(* IEC 61131-3 sources: IEC61131-3-CDSV3/Regular Expressions/src/20 Program Organization Units/Unicode, 1 file *)

(* ---- FuUnicodeCodepointCaseConvert.pou ---- *)
(*#-#-#-#-#-#-#-#-#-#---Declaration---#-#-#-#-#-#-#-#-#-#-#-#-#*)

// Converts the given Unicode odepoint to the lowercase or uppercase codepoint (the opposite casing).
// If there is no codepoint mapping, then it will return 0.
{attribute 'qualified_only'}
FUNCTION FuUnicodeCodepointCaseConvert : DWORD
VAR_INPUT
    dwCodepoint: DWORD;
END_VAR
(*#-#-#-#-#-#-#-#-#-#---Implementation---#-#-#-#-#-#-#-#-#-#-#-#-#*)

FuUnicodeCodepointCaseConvert := 0;

// The following code has been generated from Unicode's UnicodeData.txt file
CASE dwCodepoint OF
    65:
        FuUnicodeCodepointCaseConvert := 97;
        RETURN;
    66:
        FuUnicodeCodepointCaseConvert := 98;
        RETURN;
    67:
        FuUnicodeCodepointCaseConvert := 99;
        RETURN;
    68:
        FuUnicodeCodepointCaseConvert := 100;
        RETURN;
    69:
        FuUnicodeCodepointCaseConvert := 101;
        RETURN;
    70:
        FuUnicodeCodepointCaseConvert := 102;
        RETURN;
    71:
        FuUnicodeCodepointCaseConvert := 103;
        RETURN;
    72:
        FuUnicodeCodepointCaseConvert := 104;
        RETURN;
    73:
        FuUnicodeCodepointCaseConvert := 105;
        RETURN;
    74:
        FuUnicodeCodepointCaseConvert := 106;
        RETURN;
    75:
        FuUnicodeCodepointCaseConvert := 107;
        RETURN;
    76:
        FuUnicodeCodepointCaseConvert := 108;
        RETURN;
    77:
        FuUnicodeCodepointCaseConvert := 109;
        RETURN;
    78:
        FuUnicodeCodepointCaseConvert := 110;
        RETURN;
    79:
        FuUnicodeCodepointCaseConvert := 111;
        RETURN;
    80:
        FuUnicodeCodepointCaseConvert := 112;
        RETURN;
    81:
        FuUnicodeCodepointCaseConvert := 113;
        RETURN;
    82:
        FuUnicodeCodepointCaseConvert := 114;
        RETURN;
    83:
        FuUnicodeCodepointCaseConvert := 115;
        RETURN;
    84:
        FuUnicodeCodepointCaseConvert := 116;
        RETURN;
    85:
        FuUnicodeCodepointCaseConvert := 117;
        RETURN;
    86:
        FuUnicodeCodepointCaseConvert := 118;
        RETURN;
    87:
        FuUnicodeCodepointCaseConvert := 119;
        RETURN;
    88:
        FuUnicodeCodepointCaseConvert := 120;
        RETURN;
    89:
        FuUnicodeCodepointCaseConvert := 121;
        RETURN;
    90:
        FuUnicodeCodepointCaseConvert := 122;
        RETURN;
    97:
        FuUnicodeCodepointCaseConvert := 65;
        RETURN;
    98:
        FuUnicodeCodepointCaseConvert := 66;
        RETURN;
    99:
        FuUnicodeCodepointCaseConvert := 67;
        RETURN;
    100:
        FuUnicodeCodepointCaseConvert := 68;
        RETURN;
    101:
        FuUnicodeCodepointCaseConvert := 69;
        RETURN;
    102:
        FuUnicodeCodepointCaseConvert := 70;
        RETURN;
    103:
        FuUnicodeCodepointCaseConvert := 71;
        RETURN;
    104:
        FuUnicodeCodepointCaseConvert := 72;
        RETURN;
    105:
        FuUnicodeCodepointCaseConvert := 73;
        RETURN;
    106:
        FuUnicodeCodepointCaseConvert := 74;
        RETURN;
    107:
        FuUnicodeCodepointCaseConvert := 75;
        RETURN;
    108:
        FuUnicodeCodepointCaseConvert := 76;
        RETURN;
    109:
        FuUnicodeCodepointCaseConvert := 77;
        RETURN;
    110:
        FuUnicodeCodepointCaseConvert := 78;
        RETURN;
    111:
        FuUnicodeCodepointCaseConvert := 79;
        RETURN;
    112:
        FuUnicodeCodepointCaseConvert := 80;
        RETURN;
    113:
        FuUnicodeCodepointCaseConvert := 81;
        RETURN;
    114:
        FuUnicodeCodepointCaseConvert := 82;
        RETURN;
    115:
        FuUnicodeCodepointCaseConvert := 83;
        RETURN;
    116:
        FuUnicodeCodepointCaseConvert := 84;
        RETURN;
    117:
        FuUnicodeCodepointCaseConvert := 85;
        RETURN;
    118:
        FuUnicodeCodepointCaseConvert := 86;
        RETURN;
    119:
        FuUnicodeCodepointCaseConvert := 87;
        RETURN;
    120:
        FuUnicodeCodepointCaseConvert := 88;
        RETURN;
    121:
        FuUnicodeCodepointCaseConvert := 89;
        RETURN;
    122:
        FuUnicodeCodepointCaseConvert := 90;
        RETURN;
    181:
        FuUnicodeCodepointCaseConvert := 924;
        RETURN;
    192:
        FuUnicodeCodepointCaseConvert := 224;
        RETURN;
    193:
        FuUnicodeCodepointCaseConvert := 225;
        RETURN;
    194:
        FuUnicodeCodepointCaseConvert := 226;
        RETURN;
    195:
        FuUnicodeCodepointCaseConvert := 227;
        RETURN;
    196:
        FuUnicodeCodepointCaseConvert := 228;
        RETURN;
    197:
        FuUnicodeCodepointCaseConvert := 229;
        RETURN;
    198:
        FuUnicodeCodepointCaseConvert := 230;
        RETURN;
    199:
        FuUnicodeCodepointCaseConvert := 231;
        RETURN;
    200:
        FuUnicodeCodepointCaseConvert := 232;
        RETURN;
    201:
        FuUnicodeCodepointCaseConvert := 233;
        RETURN;
    202:
        FuUnicodeCodepointCaseConvert := 234;
        RETURN;
    203:
        FuUnicodeCodepointCaseConvert := 235;
        RETURN;
    204:
        FuUnicodeCodepointCaseConvert := 236;
        RETURN;
    205:
        FuUnicodeCodepointCaseConvert := 237;
        RETURN;
    206:
        FuUnicodeCodepointCaseConvert := 238;
        RETURN;
    207:
        FuUnicodeCodepointCaseConvert := 239;
        RETURN;
    208:
        FuUnicodeCodepointCaseConvert := 240;
        RETURN;
    209:
        FuUnicodeCodepointCaseConvert := 241;
        RETURN;
    210:
        FuUnicodeCodepointCaseConvert := 242;
        RETURN;
    211:
        FuUnicodeCodepointCaseConvert := 243;
        RETURN;
    212:
        FuUnicodeCodepointCaseConvert := 244;
        RETURN;
    213:
        FuUnicodeCodepointCaseConvert := 245;
        RETURN;
    214:
        FuUnicodeCodepointCaseConvert := 246;
        RETURN;
    216:
        FuUnicodeCodepointCaseConvert := 248;
        RETURN;
    217:
        FuUnicodeCodepointCaseConvert := 249;
        RETURN;
    218:
        FuUnicodeCodepointCaseConvert := 250;
        RETURN;
    219:
        FuUnicodeCodepointCaseConvert := 251;
        RETURN;
    220:
        FuUnicodeCodepointCaseConvert := 252;
        RETURN;
    221:
        FuUnicodeCodepointCaseConvert := 253;
        RETURN;
    222:
        FuUnicodeCodepointCaseConvert := 254;
        RETURN;
    224:
        FuUnicodeCodepointCaseConvert := 192;
        RETURN;
    225:
        FuUnicodeCodepointCaseConvert := 193;
        RETURN;
    226:
        FuUnicodeCodepointCaseConvert := 194;
        RETURN;
    227:
        FuUnicodeCodepointCaseConvert := 195;
        RETURN;
    228:
        FuUnicodeCodepointCaseConvert := 196;
        RETURN;
    229:
        FuUnicodeCodepointCaseConvert := 197;
        RETURN;
    230:
        FuUnicodeCodepointCaseConvert := 198;
        RETURN;
    231:
        FuUnicodeCodepointCaseConvert := 199;
        RETURN;
    232:
        FuUnicodeCodepointCaseConvert := 200;
        RETURN;
    233:
        FuUnicodeCodepointCaseConvert := 201;
        RETURN;
    234:
        FuUnicodeCodepointCaseConvert := 202;
        RETURN;
    235:
        FuUnicodeCodepointCaseConvert := 203;
        RETURN;
    236:
        FuUnicodeCodepointCaseConvert := 204;
        RETURN;
    237:
        FuUnicodeCodepointCaseConvert := 205;
        RETURN;
    238:
        FuUnicodeCodepointCaseConvert := 206;
        RETURN;
    239:
        FuUnicodeCodepointCaseConvert := 207;
        RETURN;
    240:
        FuUnicodeCodepointCaseConvert := 208;
        RETURN;
    241:
        FuUnicodeCodepointCaseConvert := 209;
        RETURN;
    242:
        FuUnicodeCodepointCaseConvert := 210;
        RETURN;
    243:
        FuUnicodeCodepointCaseConvert := 211;
        RETURN;
    244:
        FuUnicodeCodepointCaseConvert := 212;
        RETURN;
    245:
        FuUnicodeCodepointCaseConvert := 213;
        RETURN;
    246:
        FuUnicodeCodepointCaseConvert := 214;
        RETURN;
    248:
        FuUnicodeCodepointCaseConvert := 216;
        RETURN;
    249:
        FuUnicodeCodepointCaseConvert := 217;
        RETURN;
    250:
        FuUnicodeCodepointCaseConvert := 218;
        RETURN;
    251:
        FuUnicodeCodepointCaseConvert := 219;
        RETURN;
    252:
        FuUnicodeCodepointCaseConvert := 220;
        RETURN;
    253:
        FuUnicodeCodepointCaseConvert := 221;
        RETURN;
    254:
        FuUnicodeCodepointCaseConvert := 222;
        RETURN;
    255:
        FuUnicodeCodepointCaseConvert := 376;
        RETURN;
    256:
        FuUnicodeCodepointCaseConvert := 257;
        RETURN;
    257:
        FuUnicodeCodepointCaseConvert := 256;
        RETURN;
    258:
        FuUnicodeCodepointCaseConvert := 259;
        RETURN;
    259:
        FuUnicodeCodepointCaseConvert := 258;
        RETURN;
    260:
        FuUnicodeCodepointCaseConvert := 261;
        RETURN;
    261:
        FuUnicodeCodepointCaseConvert := 260;
        RETURN;
    262:
        FuUnicodeCodepointCaseConvert := 263;
        RETURN;
    263:
        FuUnicodeCodepointCaseConvert := 262;
        RETURN;
    264:
        FuUnicodeCodepointCaseConvert := 265;
        RETURN;
    265:
        FuUnicodeCodepointCaseConvert := 264;
        RETURN;
    266:
        FuUnicodeCodepointCaseConvert := 267;
        RETURN;
    267:
        FuUnicodeCodepointCaseConvert := 266;
        RETURN;
    268:
        FuUnicodeCodepointCaseConvert := 269;
        RETURN;
    269:
        FuUnicodeCodepointCaseConvert := 268;
        RETURN;
    270:
        FuUnicodeCodepointCaseConvert := 271;
        RETURN;
    271:
        FuUnicodeCodepointCaseConvert := 270;
        RETURN;
    272:
        FuUnicodeCodepointCaseConvert := 273;
        RETURN;
    273:
        FuUnicodeCodepointCaseConvert := 272;
        RETURN;
    274:
        FuUnicodeCodepointCaseConvert := 275;
        RETURN;
    275:
        FuUnicodeCodepointCaseConvert := 274;
        RETURN;
    276:
        FuUnicodeCodepointCaseConvert := 277;
        RETURN;
    277:
        FuUnicodeCodepointCaseConvert := 276;
        RETURN;
    278:
        FuUnicodeCodepointCaseConvert := 279;
        RETURN;
    279:
        FuUnicodeCodepointCaseConvert := 278;
        RETURN;
    280:
        FuUnicodeCodepointCaseConvert := 281;
        RETURN;
    281:
        FuUnicodeCodepointCaseConvert := 280;
        RETURN;
    282:
        FuUnicodeCodepointCaseConvert := 283;
        RETURN;
    283:
        FuUnicodeCodepointCaseConvert := 282;
        RETURN;
    284:
        FuUnicodeCodepointCaseConvert := 285;
        RETURN;
    285:
        FuUnicodeCodepointCaseConvert := 284;
        RETURN;
    286:
        FuUnicodeCodepointCaseConvert := 287;
        RETURN;
    287:
        FuUnicodeCodepointCaseConvert := 286;
        RETURN;
    288:
        FuUnicodeCodepointCaseConvert := 289;
        RETURN;
    289:
        FuUnicodeCodepointCaseConvert := 288;
        RETURN;
    290:
        FuUnicodeCodepointCaseConvert := 291;
        RETURN;
    291:
        FuUnicodeCodepointCaseConvert := 290;
        RETURN;
    292:
        FuUnicodeCodepointCaseConvert := 293;
        RETURN;
    293:
        FuUnicodeCodepointCaseConvert := 292;
        RETURN;
    294:
        FuUnicodeCodepointCaseConvert := 295;
        RETURN;
    295:
        FuUnicodeCodepointCaseConvert := 294;
        RETURN;
    296:
        FuUnicodeCodepointCaseConvert := 297;
        RETURN;
    297:
        FuUnicodeCodepointCaseConvert := 296;
        RETURN;
    298:
        FuUnicodeCodepointCaseConvert := 299;
        RETURN;
    299:
        FuUnicodeCodepointCaseConvert := 298;
        RETURN;
    300:
        FuUnicodeCodepointCaseConvert := 301;
        RETURN;
    301:
        FuUnicodeCodepointCaseConvert := 300;
        RETURN;
    302:
        FuUnicodeCodepointCaseConvert := 303;
        RETURN;
    303:
        FuUnicodeCodepointCaseConvert := 302;
        RETURN;
    304:
        FuUnicodeCodepointCaseConvert := 105;
        RETURN;
    305:
        FuUnicodeCodepointCaseConvert := 73;
        RETURN;
    306:
        FuUnicodeCodepointCaseConvert := 307;
        RETURN;
    307:
        FuUnicodeCodepointCaseConvert := 306;
        RETURN;
    308:
        FuUnicodeCodepointCaseConvert := 309;
        RETURN;
    309:
        FuUnicodeCodepointCaseConvert := 308;
        RETURN;
    310:
        FuUnicodeCodepointCaseConvert := 311;
        RETURN;
    311:
        FuUnicodeCodepointCaseConvert := 310;
        RETURN;
    313:
        FuUnicodeCodepointCaseConvert := 314;
        RETURN;
    314:
        FuUnicodeCodepointCaseConvert := 313;
        RETURN;
    315:
        FuUnicodeCodepointCaseConvert := 316;
        RETURN;
    316:
        FuUnicodeCodepointCaseConvert := 315;
        RETURN;
    317:
        FuUnicodeCodepointCaseConvert := 318;
        RETURN;
    318:
        FuUnicodeCodepointCaseConvert := 317;
        RETURN;
    319:
        FuUnicodeCodepointCaseConvert := 320;
        RETURN;
    320:
        FuUnicodeCodepointCaseConvert := 319;
        RETURN;
    321:
        FuUnicodeCodepointCaseConvert := 322;
        RETURN;
    322:
        FuUnicodeCodepointCaseConvert := 321;
        RETURN;
    323:
        FuUnicodeCodepointCaseConvert := 324;
        RETURN;
    324:
        FuUnicodeCodepointCaseConvert := 323;
        RETURN;
    325:
        FuUnicodeCodepointCaseConvert := 326;
        RETURN;
    326:
        FuUnicodeCodepointCaseConvert := 325;
        RETURN;
    327:
        FuUnicodeCodepointCaseConvert := 328;
        RETURN;
    328:
        FuUnicodeCodepointCaseConvert := 327;
        RETURN;
    330:
        FuUnicodeCodepointCaseConvert := 331;
        RETURN;
    331:
        FuUnicodeCodepointCaseConvert := 330;
        RETURN;
    332:
        FuUnicodeCodepointCaseConvert := 333;
        RETURN;
    333:
        FuUnicodeCodepointCaseConvert := 332;
        RETURN;
    334:
        FuUnicodeCodepointCaseConvert := 335;
        RETURN;
    335:
        FuUnicodeCodepointCaseConvert := 334;
        RETURN;
    336:
        FuUnicodeCodepointCaseConvert := 337;
        RETURN;
    337:
        FuUnicodeCodepointCaseConvert := 336;
        RETURN;
    338:
        FuUnicodeCodepointCaseConvert := 339;
        RETURN;
    339:
        FuUnicodeCodepointCaseConvert := 338;
        RETURN;
    340:
        FuUnicodeCodepointCaseConvert := 341;
        RETURN;
    341:
        FuUnicodeCodepointCaseConvert := 340;
        RETURN;
    342:
        FuUnicodeCodepointCaseConvert := 343;
        RETURN;
    343:
        FuUnicodeCodepointCaseConvert := 342;
        RETURN;
    344:
        FuUnicodeCodepointCaseConvert := 345;
        RETURN;
    345:
        FuUnicodeCodepointCaseConvert := 344;
        RETURN;
    346:
        FuUnicodeCodepointCaseConvert := 347;
        RETURN;
    347:
        FuUnicodeCodepointCaseConvert := 346;
        RETURN;
    348:
        FuUnicodeCodepointCaseConvert := 349;
        RETURN;
    349:
        FuUnicodeCodepointCaseConvert := 348;
        RETURN;
    350:
        FuUnicodeCodepointCaseConvert := 351;
        RETURN;
    351:
        FuUnicodeCodepointCaseConvert := 350;
        RETURN;
    352:
        FuUnicodeCodepointCaseConvert := 353;
        RETURN;
    353:
        FuUnicodeCodepointCaseConvert := 352;
        RETURN;
    354:
        FuUnicodeCodepointCaseConvert := 355;
        RETURN;
    355:
        FuUnicodeCodepointCaseConvert := 354;
        RETURN;
    356:
        FuUnicodeCodepointCaseConvert := 357;
        RETURN;
    357:
        FuUnicodeCodepointCaseConvert := 356;
        RETURN;
    358:
        FuUnicodeCodepointCaseConvert := 359;
        RETURN;
    359:
        FuUnicodeCodepointCaseConvert := 358;
        RETURN;
    360:
        FuUnicodeCodepointCaseConvert := 361;
        RETURN;
    361:
        FuUnicodeCodepointCaseConvert := 360;
        RETURN;
    362:
        FuUnicodeCodepointCaseConvert := 363;
        RETURN;
    363:
        FuUnicodeCodepointCaseConvert := 362;
        RETURN;
    364:
        FuUnicodeCodepointCaseConvert := 365;
        RETURN;
    365:
        FuUnicodeCodepointCaseConvert := 364;
        RETURN;
    366:
        FuUnicodeCodepointCaseConvert := 367;
        RETURN;
    367:
        FuUnicodeCodepointCaseConvert := 366;
        RETURN;
    368:
        FuUnicodeCodepointCaseConvert := 369;
        RETURN;
    369:
        FuUnicodeCodepointCaseConvert := 368;
        RETURN;
    370:
        FuUnicodeCodepointCaseConvert := 371;
        RETURN;
    371:
        FuUnicodeCodepointCaseConvert := 370;
        RETURN;
    372:
        FuUnicodeCodepointCaseConvert := 373;
        RETURN;
    373:
        FuUnicodeCodepointCaseConvert := 372;
        RETURN;
    374:
        FuUnicodeCodepointCaseConvert := 375;
        RETURN;
    375:
        FuUnicodeCodepointCaseConvert := 374;
        RETURN;
    376:
        FuUnicodeCodepointCaseConvert := 255;
        RETURN;
    377:
        FuUnicodeCodepointCaseConvert := 378;
        RETURN;
    378:
        FuUnicodeCodepointCaseConvert := 377;
        RETURN;
    379:
        FuUnicodeCodepointCaseConvert := 380;
        RETURN;
    380:
        FuUnicodeCodepointCaseConvert := 379;
        RETURN;
    381:
        FuUnicodeCodepointCaseConvert := 382;
        RETURN;
    382:
        FuUnicodeCodepointCaseConvert := 381;
        RETURN;
    383:
        FuUnicodeCodepointCaseConvert := 83;
        RETURN;
    384:
        FuUnicodeCodepointCaseConvert := 579;
        RETURN;
    385:
        FuUnicodeCodepointCaseConvert := 595;
        RETURN;
    386:
        FuUnicodeCodepointCaseConvert := 387;
        RETURN;
    387:
        FuUnicodeCodepointCaseConvert := 386;
        RETURN;
    388:
        FuUnicodeCodepointCaseConvert := 389;
        RETURN;
    389:
        FuUnicodeCodepointCaseConvert := 388;
        RETURN;
    390:
        FuUnicodeCodepointCaseConvert := 596;
        RETURN;
    391:
        FuUnicodeCodepointCaseConvert := 392;
        RETURN;
    392:
        FuUnicodeCodepointCaseConvert := 391;
        RETURN;
    393:
        FuUnicodeCodepointCaseConvert := 598;
        RETURN;
    394:
        FuUnicodeCodepointCaseConvert := 599;
        RETURN;
    395:
        FuUnicodeCodepointCaseConvert := 396;
        RETURN;
    396:
        FuUnicodeCodepointCaseConvert := 395;
        RETURN;
    398:
        FuUnicodeCodepointCaseConvert := 477;
        RETURN;
    399:
        FuUnicodeCodepointCaseConvert := 601;
        RETURN;
    400:
        FuUnicodeCodepointCaseConvert := 603;
        RETURN;
    401:
        FuUnicodeCodepointCaseConvert := 402;
        RETURN;
    402:
        FuUnicodeCodepointCaseConvert := 401;
        RETURN;
    403:
        FuUnicodeCodepointCaseConvert := 608;
        RETURN;
    404:
        FuUnicodeCodepointCaseConvert := 611;
        RETURN;
    405:
        FuUnicodeCodepointCaseConvert := 502;
        RETURN;
    406:
        FuUnicodeCodepointCaseConvert := 617;
        RETURN;
    407:
        FuUnicodeCodepointCaseConvert := 616;
        RETURN;
    408:
        FuUnicodeCodepointCaseConvert := 409;
        RETURN;
    409:
        FuUnicodeCodepointCaseConvert := 408;
        RETURN;
    410:
        FuUnicodeCodepointCaseConvert := 573;
        RETURN;
    412:
        FuUnicodeCodepointCaseConvert := 623;
        RETURN;
    413:
        FuUnicodeCodepointCaseConvert := 626;
        RETURN;
    414:
        FuUnicodeCodepointCaseConvert := 544;
        RETURN;
    415:
        FuUnicodeCodepointCaseConvert := 629;
        RETURN;
    416:
        FuUnicodeCodepointCaseConvert := 417;
        RETURN;
    417:
        FuUnicodeCodepointCaseConvert := 416;
        RETURN;
    418:
        FuUnicodeCodepointCaseConvert := 419;
        RETURN;
    419:
        FuUnicodeCodepointCaseConvert := 418;
        RETURN;
    420:
        FuUnicodeCodepointCaseConvert := 421;
        RETURN;
    421:
        FuUnicodeCodepointCaseConvert := 420;
        RETURN;
    422:
        FuUnicodeCodepointCaseConvert := 640;
        RETURN;
    423:
        FuUnicodeCodepointCaseConvert := 424;
        RETURN;
    424:
        FuUnicodeCodepointCaseConvert := 423;
        RETURN;
    425:
        FuUnicodeCodepointCaseConvert := 643;
        RETURN;
    428:
        FuUnicodeCodepointCaseConvert := 429;
        RETURN;
    429:
        FuUnicodeCodepointCaseConvert := 428;
        RETURN;
    430:
        FuUnicodeCodepointCaseConvert := 648;
        RETURN;
    431:
        FuUnicodeCodepointCaseConvert := 432;
        RETURN;
    432:
        FuUnicodeCodepointCaseConvert := 431;
        RETURN;
    433:
        FuUnicodeCodepointCaseConvert := 650;
        RETURN;
    434:
        FuUnicodeCodepointCaseConvert := 651;
        RETURN;
    435:
        FuUnicodeCodepointCaseConvert := 436;
        RETURN;
    436:
        FuUnicodeCodepointCaseConvert := 435;
        RETURN;
    437:
        FuUnicodeCodepointCaseConvert := 438;
        RETURN;
    438:
        FuUnicodeCodepointCaseConvert := 437;
        RETURN;
    439:
        FuUnicodeCodepointCaseConvert := 658;
        RETURN;
    440:
        FuUnicodeCodepointCaseConvert := 441;
        RETURN;
    441:
        FuUnicodeCodepointCaseConvert := 440;
        RETURN;
    444:
        FuUnicodeCodepointCaseConvert := 445;
        RETURN;
    445:
        FuUnicodeCodepointCaseConvert := 444;
        RETURN;
    447:
        FuUnicodeCodepointCaseConvert := 503;
        RETURN;
    452:
        FuUnicodeCodepointCaseConvert := 453;
        RETURN;
    453:
        FuUnicodeCodepointCaseConvert := 453;
        RETURN;
    454:
        FuUnicodeCodepointCaseConvert := 453;
        RETURN;
    455:
        FuUnicodeCodepointCaseConvert := 456;
        RETURN;
    456:
        FuUnicodeCodepointCaseConvert := 456;
        RETURN;
    457:
        FuUnicodeCodepointCaseConvert := 456;
        RETURN;
    458:
        FuUnicodeCodepointCaseConvert := 459;
        RETURN;
    459:
        FuUnicodeCodepointCaseConvert := 459;
        RETURN;
    460:
        FuUnicodeCodepointCaseConvert := 459;
        RETURN;
    461:
        FuUnicodeCodepointCaseConvert := 462;
        RETURN;
    462:
        FuUnicodeCodepointCaseConvert := 461;
        RETURN;
    463:
        FuUnicodeCodepointCaseConvert := 464;
        RETURN;
    464:
        FuUnicodeCodepointCaseConvert := 463;
        RETURN;
    465:
        FuUnicodeCodepointCaseConvert := 466;
        RETURN;
    466:
        FuUnicodeCodepointCaseConvert := 465;
        RETURN;
    467:
        FuUnicodeCodepointCaseConvert := 468;
        RETURN;
    468:
        FuUnicodeCodepointCaseConvert := 467;
        RETURN;
    469:
        FuUnicodeCodepointCaseConvert := 470;
        RETURN;
    470:
        FuUnicodeCodepointCaseConvert := 469;
        RETURN;
    471:
        FuUnicodeCodepointCaseConvert := 472;
        RETURN;
    472:
        FuUnicodeCodepointCaseConvert := 471;
        RETURN;
    473:
        FuUnicodeCodepointCaseConvert := 474;
        RETURN;
    474:
        FuUnicodeCodepointCaseConvert := 473;
        RETURN;
    475:
        FuUnicodeCodepointCaseConvert := 476;
        RETURN;
    476:
        FuUnicodeCodepointCaseConvert := 475;
        RETURN;
    477:
        FuUnicodeCodepointCaseConvert := 398;
        RETURN;
    478:
        FuUnicodeCodepointCaseConvert := 479;
        RETURN;
    479:
        FuUnicodeCodepointCaseConvert := 478;
        RETURN;
    480:
        FuUnicodeCodepointCaseConvert := 481;
        RETURN;
    481:
        FuUnicodeCodepointCaseConvert := 480;
        RETURN;
    482:
        FuUnicodeCodepointCaseConvert := 483;
        RETURN;
    483:
        FuUnicodeCodepointCaseConvert := 482;
        RETURN;
    484:
        FuUnicodeCodepointCaseConvert := 485;
        RETURN;
    485:
        FuUnicodeCodepointCaseConvert := 484;
        RETURN;
    486:
        FuUnicodeCodepointCaseConvert := 487;
        RETURN;
    487:
        FuUnicodeCodepointCaseConvert := 486;
        RETURN;
    488:
        FuUnicodeCodepointCaseConvert := 489;
        RETURN;
    489:
        FuUnicodeCodepointCaseConvert := 488;
        RETURN;
    490:
        FuUnicodeCodepointCaseConvert := 491;
        RETURN;
    491:
        FuUnicodeCodepointCaseConvert := 490;
        RETURN;
    492:
        FuUnicodeCodepointCaseConvert := 493;
        RETURN;
    493:
        FuUnicodeCodepointCaseConvert := 492;
        RETURN;
    494:
        FuUnicodeCodepointCaseConvert := 495;
        RETURN;
    495:
        FuUnicodeCodepointCaseConvert := 494;
        RETURN;
    497:
        FuUnicodeCodepointCaseConvert := 498;
        RETURN;
    498:
        FuUnicodeCodepointCaseConvert := 498;
        RETURN;
    499:
        FuUnicodeCodepointCaseConvert := 498;
        RETURN;
    500:
        FuUnicodeCodepointCaseConvert := 501;
        RETURN;
    501:
        FuUnicodeCodepointCaseConvert := 500;
        RETURN;
    502:
        FuUnicodeCodepointCaseConvert := 405;
        RETURN;
    503:
        FuUnicodeCodepointCaseConvert := 447;
        RETURN;
    504:
        FuUnicodeCodepointCaseConvert := 505;
        RETURN;
    505:
        FuUnicodeCodepointCaseConvert := 504;
        RETURN;
    506:
        FuUnicodeCodepointCaseConvert := 507;
        RETURN;
    507:
        FuUnicodeCodepointCaseConvert := 506;
        RETURN;
    508:
        FuUnicodeCodepointCaseConvert := 509;
        RETURN;
    509:
        FuUnicodeCodepointCaseConvert := 508;
        RETURN;
    510:
        FuUnicodeCodepointCaseConvert := 511;
        RETURN;
    511:
        FuUnicodeCodepointCaseConvert := 510;
        RETURN;
    512:
        FuUnicodeCodepointCaseConvert := 513;
        RETURN;
    513:
        FuUnicodeCodepointCaseConvert := 512;
        RETURN;
    514:
        FuUnicodeCodepointCaseConvert := 515;
        RETURN;
    515:
        FuUnicodeCodepointCaseConvert := 514;
        RETURN;
    516:
        FuUnicodeCodepointCaseConvert := 517;
        RETURN;
    517:
        FuUnicodeCodepointCaseConvert := 516;
        RETURN;
    518:
        FuUnicodeCodepointCaseConvert := 519;
        RETURN;
    519:
        FuUnicodeCodepointCaseConvert := 518;
        RETURN;
    520:
        FuUnicodeCodepointCaseConvert := 521;
        RETURN;
    521:
        FuUnicodeCodepointCaseConvert := 520;
        RETURN;
    522:
        FuUnicodeCodepointCaseConvert := 523;
        RETURN;
    523:
        FuUnicodeCodepointCaseConvert := 522;
        RETURN;
    524:
        FuUnicodeCodepointCaseConvert := 525;
        RETURN;
    525:
        FuUnicodeCodepointCaseConvert := 524;
        RETURN;
    526:
        FuUnicodeCodepointCaseConvert := 527;
        RETURN;
    527:
        FuUnicodeCodepointCaseConvert := 526;
        RETURN;
    528:
        FuUnicodeCodepointCaseConvert := 529;
        RETURN;
    529:
        FuUnicodeCodepointCaseConvert := 528;
        RETURN;
    530:
        FuUnicodeCodepointCaseConvert := 531;
        RETURN;
    531:
        FuUnicodeCodepointCaseConvert := 530;
        RETURN;
    532:
        FuUnicodeCodepointCaseConvert := 533;
        RETURN;
    533:
        FuUnicodeCodepointCaseConvert := 532;
        RETURN;
    534:
        FuUnicodeCodepointCaseConvert := 535;
        RETURN;
    535:
        FuUnicodeCodepointCaseConvert := 534;
        RETURN;
    536:
        FuUnicodeCodepointCaseConvert := 537;
        RETURN;
    537:
        FuUnicodeCodepointCaseConvert := 536;
        RETURN;
    538:
        FuUnicodeCodepointCaseConvert := 539;
        RETURN;
    539:
        FuUnicodeCodepointCaseConvert := 538;
        RETURN;
    540:
        FuUnicodeCodepointCaseConvert := 541;
        RETURN;
    541:
        FuUnicodeCodepointCaseConvert := 540;
        RETURN;
    542:
        FuUnicodeCodepointCaseConvert := 543;
        RETURN;
    543:
        FuUnicodeCodepointCaseConvert := 542;
        RETURN;
    544:
        FuUnicodeCodepointCaseConvert := 414;
        RETURN;
    546:
        FuUnicodeCodepointCaseConvert := 547;
        RETURN;
    547:
        FuUnicodeCodepointCaseConvert := 546;
        RETURN;
    548:
        FuUnicodeCodepointCaseConvert := 549;
        RETURN;
    549:
        FuUnicodeCodepointCaseConvert := 548;
        RETURN;
    550:
        FuUnicodeCodepointCaseConvert := 551;
        RETURN;
    551:
        FuUnicodeCodepointCaseConvert := 550;
        RETURN;
    552:
        FuUnicodeCodepointCaseConvert := 553;
        RETURN;
    553:
        FuUnicodeCodepointCaseConvert := 552;
        RETURN;
    554:
        FuUnicodeCodepointCaseConvert := 555;
        RETURN;
    555:
        FuUnicodeCodepointCaseConvert := 554;
        RETURN;
    556:
        FuUnicodeCodepointCaseConvert := 557;
        RETURN;
    557:
        FuUnicodeCodepointCaseConvert := 556;
        RETURN;
    558:
        FuUnicodeCodepointCaseConvert := 559;
        RETURN;
    559:
        FuUnicodeCodepointCaseConvert := 558;
        RETURN;
    560:
        FuUnicodeCodepointCaseConvert := 561;
        RETURN;
    561:
        FuUnicodeCodepointCaseConvert := 560;
        RETURN;
    562:
        FuUnicodeCodepointCaseConvert := 563;
        RETURN;
    563:
        FuUnicodeCodepointCaseConvert := 562;
        RETURN;
    570:
        FuUnicodeCodepointCaseConvert := 11365;
        RETURN;
    571:
        FuUnicodeCodepointCaseConvert := 572;
        RETURN;
    572:
        FuUnicodeCodepointCaseConvert := 571;
        RETURN;
    573:
        FuUnicodeCodepointCaseConvert := 410;
        RETURN;
    574:
        FuUnicodeCodepointCaseConvert := 11366;
        RETURN;
    575:
        FuUnicodeCodepointCaseConvert := 11390;
        RETURN;
    576:
        FuUnicodeCodepointCaseConvert := 11391;
        RETURN;
    577:
        FuUnicodeCodepointCaseConvert := 578;
        RETURN;
    578:
        FuUnicodeCodepointCaseConvert := 577;
        RETURN;
    579:
        FuUnicodeCodepointCaseConvert := 384;
        RETURN;
    580:
        FuUnicodeCodepointCaseConvert := 649;
        RETURN;
    581:
        FuUnicodeCodepointCaseConvert := 652;
        RETURN;
    582:
        FuUnicodeCodepointCaseConvert := 583;
        RETURN;
    583:
        FuUnicodeCodepointCaseConvert := 582;
        RETURN;
    584:
        FuUnicodeCodepointCaseConvert := 585;
        RETURN;
    585:
        FuUnicodeCodepointCaseConvert := 584;
        RETURN;
    586:
        FuUnicodeCodepointCaseConvert := 587;
        RETURN;
    587:
        FuUnicodeCodepointCaseConvert := 586;
        RETURN;
    588:
        FuUnicodeCodepointCaseConvert := 589;
        RETURN;
    589:
        FuUnicodeCodepointCaseConvert := 588;
        RETURN;
    590:
        FuUnicodeCodepointCaseConvert := 591;
        RETURN;
    591:
        FuUnicodeCodepointCaseConvert := 590;
        RETURN;
    592:
        FuUnicodeCodepointCaseConvert := 11375;
        RETURN;
    593:
        FuUnicodeCodepointCaseConvert := 11373;
        RETURN;
    594:
        FuUnicodeCodepointCaseConvert := 11376;
        RETURN;
    595:
        FuUnicodeCodepointCaseConvert := 385;
        RETURN;
    596:
        FuUnicodeCodepointCaseConvert := 390;
        RETURN;
    598:
        FuUnicodeCodepointCaseConvert := 393;
        RETURN;
    599:
        FuUnicodeCodepointCaseConvert := 394;
        RETURN;
    601:
        FuUnicodeCodepointCaseConvert := 399;
        RETURN;
    603:
        FuUnicodeCodepointCaseConvert := 400;
        RETURN;
    604:
        FuUnicodeCodepointCaseConvert := 42923;
        RETURN;
    608:
        FuUnicodeCodepointCaseConvert := 403;
        RETURN;
    609:
        FuUnicodeCodepointCaseConvert := 42924;
        RETURN;
    611:
        FuUnicodeCodepointCaseConvert := 404;
        RETURN;
    613:
        FuUnicodeCodepointCaseConvert := 42893;
        RETURN;
    614:
        FuUnicodeCodepointCaseConvert := 42922;
        RETURN;
    616:
        FuUnicodeCodepointCaseConvert := 407;
        RETURN;
    617:
        FuUnicodeCodepointCaseConvert := 406;
        RETURN;
    618:
        FuUnicodeCodepointCaseConvert := 42926;
        RETURN;
    619:
        FuUnicodeCodepointCaseConvert := 11362;
        RETURN;
    620:
        FuUnicodeCodepointCaseConvert := 42925;
        RETURN;
    623:
        FuUnicodeCodepointCaseConvert := 412;
        RETURN;
    625:
        FuUnicodeCodepointCaseConvert := 11374;
        RETURN;
    626:
        FuUnicodeCodepointCaseConvert := 413;
        RETURN;
    629:
        FuUnicodeCodepointCaseConvert := 415;
        RETURN;
    637:
        FuUnicodeCodepointCaseConvert := 11364;
        RETURN;
    640:
        FuUnicodeCodepointCaseConvert := 422;
        RETURN;
    642:
        FuUnicodeCodepointCaseConvert := 42949;
        RETURN;
    643:
        FuUnicodeCodepointCaseConvert := 425;
        RETURN;
    647:
        FuUnicodeCodepointCaseConvert := 42929;
        RETURN;
    648:
        FuUnicodeCodepointCaseConvert := 430;
        RETURN;
    649:
        FuUnicodeCodepointCaseConvert := 580;
        RETURN;
    650:
        FuUnicodeCodepointCaseConvert := 433;
        RETURN;
    651:
        FuUnicodeCodepointCaseConvert := 434;
        RETURN;
    652:
        FuUnicodeCodepointCaseConvert := 581;
        RETURN;
    658:
        FuUnicodeCodepointCaseConvert := 439;
        RETURN;
    669:
        FuUnicodeCodepointCaseConvert := 42930;
        RETURN;
    670:
        FuUnicodeCodepointCaseConvert := 42928;
        RETURN;
    837:
        FuUnicodeCodepointCaseConvert := 921;
        RETURN;
    880:
        FuUnicodeCodepointCaseConvert := 881;
        RETURN;
    881:
        FuUnicodeCodepointCaseConvert := 880;
        RETURN;
    882:
        FuUnicodeCodepointCaseConvert := 883;
        RETURN;
    883:
        FuUnicodeCodepointCaseConvert := 882;
        RETURN;
    886:
        FuUnicodeCodepointCaseConvert := 887;
        RETURN;
    887:
        FuUnicodeCodepointCaseConvert := 886;
        RETURN;
    891:
        FuUnicodeCodepointCaseConvert := 1021;
        RETURN;
    892:
        FuUnicodeCodepointCaseConvert := 1022;
        RETURN;
    893:
        FuUnicodeCodepointCaseConvert := 1023;
        RETURN;
    895:
        FuUnicodeCodepointCaseConvert := 1011;
        RETURN;
    902:
        FuUnicodeCodepointCaseConvert := 940;
        RETURN;
    904:
        FuUnicodeCodepointCaseConvert := 941;
        RETURN;
    905:
        FuUnicodeCodepointCaseConvert := 942;
        RETURN;
    906:
        FuUnicodeCodepointCaseConvert := 943;
        RETURN;
    908:
        FuUnicodeCodepointCaseConvert := 972;
        RETURN;
    910:
        FuUnicodeCodepointCaseConvert := 973;
        RETURN;
    911:
        FuUnicodeCodepointCaseConvert := 974;
        RETURN;
    913:
        FuUnicodeCodepointCaseConvert := 945;
        RETURN;
    914:
        FuUnicodeCodepointCaseConvert := 946;
        RETURN;
    915:
        FuUnicodeCodepointCaseConvert := 947;
        RETURN;
    916:
        FuUnicodeCodepointCaseConvert := 948;
        RETURN;
    917:
        FuUnicodeCodepointCaseConvert := 949;
        RETURN;
    918:
        FuUnicodeCodepointCaseConvert := 950;
        RETURN;
    919:
        FuUnicodeCodepointCaseConvert := 951;
        RETURN;
    920:
        FuUnicodeCodepointCaseConvert := 952;
        RETURN;
    921:
        FuUnicodeCodepointCaseConvert := 953;
        RETURN;
    922:
        FuUnicodeCodepointCaseConvert := 954;
        RETURN;
    923:
        FuUnicodeCodepointCaseConvert := 955;
        RETURN;
    924:
        FuUnicodeCodepointCaseConvert := 956;
        RETURN;
    925:
        FuUnicodeCodepointCaseConvert := 957;
        RETURN;
    926:
        FuUnicodeCodepointCaseConvert := 958;
        RETURN;
    927:
        FuUnicodeCodepointCaseConvert := 959;
        RETURN;
    928:
        FuUnicodeCodepointCaseConvert := 960;
        RETURN;
    929:
        FuUnicodeCodepointCaseConvert := 961;
        RETURN;
    931:
        FuUnicodeCodepointCaseConvert := 963;
        RETURN;
    932:
        FuUnicodeCodepointCaseConvert := 964;
        RETURN;
    933:
        FuUnicodeCodepointCaseConvert := 965;
        RETURN;
    934:
        FuUnicodeCodepointCaseConvert := 966;
        RETURN;
    935:
        FuUnicodeCodepointCaseConvert := 967;
        RETURN;
    936:
        FuUnicodeCodepointCaseConvert := 968;
        RETURN;
    937:
        FuUnicodeCodepointCaseConvert := 969;
        RETURN;
    938:
        FuUnicodeCodepointCaseConvert := 970;
        RETURN;
    939:
        FuUnicodeCodepointCaseConvert := 971;
        RETURN;
    940:
        FuUnicodeCodepointCaseConvert := 902;
        RETURN;
    941:
        FuUnicodeCodepointCaseConvert := 904;
        RETURN;
    942:
        FuUnicodeCodepointCaseConvert := 905;
        RETURN;
    943:
        FuUnicodeCodepointCaseConvert := 906;
        RETURN;
    945:
        FuUnicodeCodepointCaseConvert := 913;
        RETURN;
    946:
        FuUnicodeCodepointCaseConvert := 914;
        RETURN;
    947:
        FuUnicodeCodepointCaseConvert := 915;
        RETURN;
    948:
        FuUnicodeCodepointCaseConvert := 916;
        RETURN;
    949:
        FuUnicodeCodepointCaseConvert := 917;
        RETURN;
    950:
        FuUnicodeCodepointCaseConvert := 918;
        RETURN;
    951:
        FuUnicodeCodepointCaseConvert := 919;
        RETURN;
    952:
        FuUnicodeCodepointCaseConvert := 920;
        RETURN;
    953:
        FuUnicodeCodepointCaseConvert := 921;
        RETURN;
    954:
        FuUnicodeCodepointCaseConvert := 922;
        RETURN;
    955:
        FuUnicodeCodepointCaseConvert := 923;
        RETURN;
    956:
        FuUnicodeCodepointCaseConvert := 924;
        RETURN;
    957:
        FuUnicodeCodepointCaseConvert := 925;
        RETURN;
    958:
        FuUnicodeCodepointCaseConvert := 926;
        RETURN;
    959:
        FuUnicodeCodepointCaseConvert := 927;
        RETURN;
    960:
        FuUnicodeCodepointCaseConvert := 928;
        RETURN;
    961:
        FuUnicodeCodepointCaseConvert := 929;
        RETURN;
    962:
        FuUnicodeCodepointCaseConvert := 931;
        RETURN;
    963:
        FuUnicodeCodepointCaseConvert := 931;
        RETURN;
    964:
        FuUnicodeCodepointCaseConvert := 932;
        RETURN;
    965:
        FuUnicodeCodepointCaseConvert := 933;
        RETURN;
    966:
        FuUnicodeCodepointCaseConvert := 934;
        RETURN;
    967:
        FuUnicodeCodepointCaseConvert := 935;
        RETURN;
    968:
        FuUnicodeCodepointCaseConvert := 936;
        RETURN;
    969:
        FuUnicodeCodepointCaseConvert := 937;
        RETURN;
    970:
        FuUnicodeCodepointCaseConvert := 938;
        RETURN;
    971:
        FuUnicodeCodepointCaseConvert := 939;
        RETURN;
    972:
        FuUnicodeCodepointCaseConvert := 908;
        RETURN;
    973:
        FuUnicodeCodepointCaseConvert := 910;
        RETURN;
    974:
        FuUnicodeCodepointCaseConvert := 911;
        RETURN;
    975:
        FuUnicodeCodepointCaseConvert := 983;
        RETURN;
    976:
        FuUnicodeCodepointCaseConvert := 914;
        RETURN;
    977:
        FuUnicodeCodepointCaseConvert := 920;
        RETURN;
    981:
        FuUnicodeCodepointCaseConvert := 934;
        RETURN;
    982:
        FuUnicodeCodepointCaseConvert := 928;
        RETURN;
    983:
        FuUnicodeCodepointCaseConvert := 975;
        RETURN;
    984:
        FuUnicodeCodepointCaseConvert := 985;
        RETURN;
    985:
        FuUnicodeCodepointCaseConvert := 984;
        RETURN;
    986:
        FuUnicodeCodepointCaseConvert := 987;
        RETURN;
    987:
        FuUnicodeCodepointCaseConvert := 986;
        RETURN;
    988:
        FuUnicodeCodepointCaseConvert := 989;
        RETURN;
    989:
        FuUnicodeCodepointCaseConvert := 988;
        RETURN;
    990:
        FuUnicodeCodepointCaseConvert := 991;
        RETURN;
    991:
        FuUnicodeCodepointCaseConvert := 990;
        RETURN;
    992:
        FuUnicodeCodepointCaseConvert := 993;
        RETURN;
    993:
        FuUnicodeCodepointCaseConvert := 992;
        RETURN;
    994:
        FuUnicodeCodepointCaseConvert := 995;
        RETURN;
    995:
        FuUnicodeCodepointCaseConvert := 994;
        RETURN;
    996:
        FuUnicodeCodepointCaseConvert := 997;
        RETURN;
    997:
        FuUnicodeCodepointCaseConvert := 996;
        RETURN;
    998:
        FuUnicodeCodepointCaseConvert := 999;
        RETURN;
    999:
        FuUnicodeCodepointCaseConvert := 998;
        RETURN;
    1000:
        FuUnicodeCodepointCaseConvert := 1001;
        RETURN;
    1001:
        FuUnicodeCodepointCaseConvert := 1000;
        RETURN;
    1002:
        FuUnicodeCodepointCaseConvert := 1003;
        RETURN;
    1003:
        FuUnicodeCodepointCaseConvert := 1002;
        RETURN;
    1004:
        FuUnicodeCodepointCaseConvert := 1005;
        RETURN;
    1005:
        FuUnicodeCodepointCaseConvert := 1004;
        RETURN;
    1006:
        FuUnicodeCodepointCaseConvert := 1007;
        RETURN;
    1007:
        FuUnicodeCodepointCaseConvert := 1006;
        RETURN;
    1008:
        FuUnicodeCodepointCaseConvert := 922;
        RETURN;
    1009:
        FuUnicodeCodepointCaseConvert := 929;
        RETURN;
    1010:
        FuUnicodeCodepointCaseConvert := 1017;
        RETURN;
    1011:
        FuUnicodeCodepointCaseConvert := 895;
        RETURN;
    1012:
        FuUnicodeCodepointCaseConvert := 952;
        RETURN;
    1013:
        FuUnicodeCodepointCaseConvert := 917;
        RETURN;
    1015:
        FuUnicodeCodepointCaseConvert := 1016;
        RETURN;
    1016:
        FuUnicodeCodepointCaseConvert := 1015;
        RETURN;
    1017:
        FuUnicodeCodepointCaseConvert := 1010;
        RETURN;
    1018:
        FuUnicodeCodepointCaseConvert := 1019;
        RETURN;
    1019:
        FuUnicodeCodepointCaseConvert := 1018;
        RETURN;
    1021:
        FuUnicodeCodepointCaseConvert := 891;
        RETURN;
    1022:
        FuUnicodeCodepointCaseConvert := 892;
        RETURN;
    1023:
        FuUnicodeCodepointCaseConvert := 893;
        RETURN;
    1024:
        FuUnicodeCodepointCaseConvert := 1104;
        RETURN;
    1025:
        FuUnicodeCodepointCaseConvert := 1105;
        RETURN;
    1026:
        FuUnicodeCodepointCaseConvert := 1106;
        RETURN;
    1027:
        FuUnicodeCodepointCaseConvert := 1107;
        RETURN;
    1028:
        FuUnicodeCodepointCaseConvert := 1108;
        RETURN;
    1029:
        FuUnicodeCodepointCaseConvert := 1109;
        RETURN;
    1030:
        FuUnicodeCodepointCaseConvert := 1110;
        RETURN;
    1031:
        FuUnicodeCodepointCaseConvert := 1111;
        RETURN;
    1032:
        FuUnicodeCodepointCaseConvert := 1112;
        RETURN;
    1033:
        FuUnicodeCodepointCaseConvert := 1113;
        RETURN;
    1034:
        FuUnicodeCodepointCaseConvert := 1114;
        RETURN;
    1035:
        FuUnicodeCodepointCaseConvert := 1115;
        RETURN;
    1036:
        FuUnicodeCodepointCaseConvert := 1116;
        RETURN;
    1037:
        FuUnicodeCodepointCaseConvert := 1117;
        RETURN;
    1038:
        FuUnicodeCodepointCaseConvert := 1118;
        RETURN;
    1039:
        FuUnicodeCodepointCaseConvert := 1119;
        RETURN;
    1040:
        FuUnicodeCodepointCaseConvert := 1072;
        RETURN;
    1041:
        FuUnicodeCodepointCaseConvert := 1073;
        RETURN;
    1042:
        FuUnicodeCodepointCaseConvert := 1074;
        RETURN;
    1043:
        FuUnicodeCodepointCaseConvert := 1075;
        RETURN;
    1044:
        FuUnicodeCodepointCaseConvert := 1076;
        RETURN;
    1045:
        FuUnicodeCodepointCaseConvert := 1077;
        RETURN;
    1046:
        FuUnicodeCodepointCaseConvert := 1078;
        RETURN;
    1047:
        FuUnicodeCodepointCaseConvert := 1079;
        RETURN;
    1048:
        FuUnicodeCodepointCaseConvert := 1080;
        RETURN;
    1049:
        FuUnicodeCodepointCaseConvert := 1081;
        RETURN;
    1050:
        FuUnicodeCodepointCaseConvert := 1082;
        RETURN;
    1051:
        FuUnicodeCodepointCaseConvert := 1083;
        RETURN;
    1052:
        FuUnicodeCodepointCaseConvert := 1084;
        RETURN;
    1053:
        FuUnicodeCodepointCaseConvert := 1085;
        RETURN;
    1054:
        FuUnicodeCodepointCaseConvert := 1086;
        RETURN;
    1055:
        FuUnicodeCodepointCaseConvert := 1087;
        RETURN;
    1056:
        FuUnicodeCodepointCaseConvert := 1088;
        RETURN;
    1057:
        FuUnicodeCodepointCaseConvert := 1089;
        RETURN;
    1058:
        FuUnicodeCodepointCaseConvert := 1090;
        RETURN;
    1059:
        FuUnicodeCodepointCaseConvert := 1091;
        RETURN;
    1060:
        FuUnicodeCodepointCaseConvert := 1092;
        RETURN;
    1061:
        FuUnicodeCodepointCaseConvert := 1093;
        RETURN;
    1062:
        FuUnicodeCodepointCaseConvert := 1094;
        RETURN;
    1063:
        FuUnicodeCodepointCaseConvert := 1095;
        RETURN;
    1064:
        FuUnicodeCodepointCaseConvert := 1096;
        RETURN;
    1065:
        FuUnicodeCodepointCaseConvert := 1097;
        RETURN;
    1066:
        FuUnicodeCodepointCaseConvert := 1098;
        RETURN;
    1067:
        FuUnicodeCodepointCaseConvert := 1099;
        RETURN;
    1068:
        FuUnicodeCodepointCaseConvert := 1100;
        RETURN;
    1069:
        FuUnicodeCodepointCaseConvert := 1101;
        RETURN;
    1070:
        FuUnicodeCodepointCaseConvert := 1102;
        RETURN;
    1071:
        FuUnicodeCodepointCaseConvert := 1103;
        RETURN;
    1072:
        FuUnicodeCodepointCaseConvert := 1040;
        RETURN;
    1073:
        FuUnicodeCodepointCaseConvert := 1041;
        RETURN;
    1074:
        FuUnicodeCodepointCaseConvert := 1042;
        RETURN;
    1075:
        FuUnicodeCodepointCaseConvert := 1043;
        RETURN;
    1076:
        FuUnicodeCodepointCaseConvert := 1044;
        RETURN;
    1077:
        FuUnicodeCodepointCaseConvert := 1045;
        RETURN;
    1078:
        FuUnicodeCodepointCaseConvert := 1046;
        RETURN;
    1079:
        FuUnicodeCodepointCaseConvert := 1047;
        RETURN;
    1080:
        FuUnicodeCodepointCaseConvert := 1048;
        RETURN;
    1081:
        FuUnicodeCodepointCaseConvert := 1049;
        RETURN;
    1082:
        FuUnicodeCodepointCaseConvert := 1050;
        RETURN;
    1083:
        FuUnicodeCodepointCaseConvert := 1051;
        RETURN;
    1084:
        FuUnicodeCodepointCaseConvert := 1052;
        RETURN;
    1085:
        FuUnicodeCodepointCaseConvert := 1053;
        RETURN;
    1086:
        FuUnicodeCodepointCaseConvert := 1054;
        RETURN;
    1087:
        FuUnicodeCodepointCaseConvert := 1055;
        RETURN;
    1088:
        FuUnicodeCodepointCaseConvert := 1056;
        RETURN;
    1089:
        FuUnicodeCodepointCaseConvert := 1057;
        RETURN;
    1090:
        FuUnicodeCodepointCaseConvert := 1058;
        RETURN;
    1091:
        FuUnicodeCodepointCaseConvert := 1059;
        RETURN;
    1092:
        FuUnicodeCodepointCaseConvert := 1060;
        RETURN;
    1093:
        FuUnicodeCodepointCaseConvert := 1061;
        RETURN;
    1094:
        FuUnicodeCodepointCaseConvert := 1062;
        RETURN;
    1095:
        FuUnicodeCodepointCaseConvert := 1063;
        RETURN;
    1096:
        FuUnicodeCodepointCaseConvert := 1064;
        RETURN;
    1097:
        FuUnicodeCodepointCaseConvert := 1065;
        RETURN;
    1098:
        FuUnicodeCodepointCaseConvert := 1066;
        RETURN;
    1099:
        FuUnicodeCodepointCaseConvert := 1067;
        RETURN;
    1100:
        FuUnicodeCodepointCaseConvert := 1068;
        RETURN;
    1101:
        FuUnicodeCodepointCaseConvert := 1069;
        RETURN;
    1102:
        FuUnicodeCodepointCaseConvert := 1070;
        RETURN;
    1103:
        FuUnicodeCodepointCaseConvert := 1071;
        RETURN;
    1104:
        FuUnicodeCodepointCaseConvert := 1024;
        RETURN;
    1105:
        FuUnicodeCodepointCaseConvert := 1025;
        RETURN;
    1106:
        FuUnicodeCodepointCaseConvert := 1026;
        RETURN;
    1107:
        FuUnicodeCodepointCaseConvert := 1027;
        RETURN;
    1108:
        FuUnicodeCodepointCaseConvert := 1028;
        RETURN;
    1109:
        FuUnicodeCodepointCaseConvert := 1029;
        RETURN;
    1110:
        FuUnicodeCodepointCaseConvert := 1030;
        RETURN;
    1111:
        FuUnicodeCodepointCaseConvert := 1031;
        RETURN;
    1112:
        FuUnicodeCodepointCaseConvert := 1032;
        RETURN;
    1113:
        FuUnicodeCodepointCaseConvert := 1033;
        RETURN;
    1114:
        FuUnicodeCodepointCaseConvert := 1034;
        RETURN;
    1115:
        FuUnicodeCodepointCaseConvert := 1035;
        RETURN;
    1116:
        FuUnicodeCodepointCaseConvert := 1036;
        RETURN;
    1117:
        FuUnicodeCodepointCaseConvert := 1037;
        RETURN;
    1118:
        FuUnicodeCodepointCaseConvert := 1038;
        RETURN;
    1119:
        FuUnicodeCodepointCaseConvert := 1039;
        RETURN;
    1120:
        FuUnicodeCodepointCaseConvert := 1121;
        RETURN;
    1121:
        FuUnicodeCodepointCaseConvert := 1120;
        RETURN;
    1122:
        FuUnicodeCodepointCaseConvert := 1123;
        RETURN;
    1123:
        FuUnicodeCodepointCaseConvert := 1122;
        RETURN;
    1124:
        FuUnicodeCodepointCaseConvert := 1125;
        RETURN;
    1125:
        FuUnicodeCodepointCaseConvert := 1124;
        RETURN;
    1126:
        FuUnicodeCodepointCaseConvert := 1127;
        RETURN;
    1127:
        FuUnicodeCodepointCaseConvert := 1126;
        RETURN;
    1128:
        FuUnicodeCodepointCaseConvert := 1129;
        RETURN;
    1129:
        FuUnicodeCodepointCaseConvert := 1128;
        RETURN;
    1130:
        FuUnicodeCodepointCaseConvert := 1131;
        RETURN;
    1131:
        FuUnicodeCodepointCaseConvert := 1130;
        RETURN;
    1132:
        FuUnicodeCodepointCaseConvert := 1133;
        RETURN;
    1133:
        FuUnicodeCodepointCaseConvert := 1132;
        RETURN;
    1134:
        FuUnicodeCodepointCaseConvert := 1135;
        RETURN;
    1135:
        FuUnicodeCodepointCaseConvert := 1134;
        RETURN;
    1136:
        FuUnicodeCodepointCaseConvert := 1137;
        RETURN;
    1137:
        FuUnicodeCodepointCaseConvert := 1136;
        RETURN;
    1138:
        FuUnicodeCodepointCaseConvert := 1139;
        RETURN;
    1139:
        FuUnicodeCodepointCaseConvert := 1138;
        RETURN;
    1140:
        FuUnicodeCodepointCaseConvert := 1141;
        RETURN;
    1141:
        FuUnicodeCodepointCaseConvert := 1140;
        RETURN;
    1142:
        FuUnicodeCodepointCaseConvert := 1143;
        RETURN;
    1143:
        FuUnicodeCodepointCaseConvert := 1142;
        RETURN;
    1144:
        FuUnicodeCodepointCaseConvert := 1145;
        RETURN;
    1145:
        FuUnicodeCodepointCaseConvert := 1144;
        RETURN;
    1146:
        FuUnicodeCodepointCaseConvert := 1147;
        RETURN;
    1147:
        FuUnicodeCodepointCaseConvert := 1146;
        RETURN;
    1148:
        FuUnicodeCodepointCaseConvert := 1149;
        RETURN;
    1149:
        FuUnicodeCodepointCaseConvert := 1148;
        RETURN;
    1150:
        FuUnicodeCodepointCaseConvert := 1151;
        RETURN;
    1151:
        FuUnicodeCodepointCaseConvert := 1150;
        RETURN;
    1152:
        FuUnicodeCodepointCaseConvert := 1153;
        RETURN;
    1153:
        FuUnicodeCodepointCaseConvert := 1152;
        RETURN;
    1162:
        FuUnicodeCodepointCaseConvert := 1163;
        RETURN;
    1163:
        FuUnicodeCodepointCaseConvert := 1162;
        RETURN;
    1164:
        FuUnicodeCodepointCaseConvert := 1165;
        RETURN;
    1165:
        FuUnicodeCodepointCaseConvert := 1164;
        RETURN;
    1166:
        FuUnicodeCodepointCaseConvert := 1167;
        RETURN;
    1167:
        FuUnicodeCodepointCaseConvert := 1166;
        RETURN;
    1168:
        FuUnicodeCodepointCaseConvert := 1169;
        RETURN;
    1169:
        FuUnicodeCodepointCaseConvert := 1168;
        RETURN;
    1170:
        FuUnicodeCodepointCaseConvert := 1171;
        RETURN;
    1171:
        FuUnicodeCodepointCaseConvert := 1170;
        RETURN;
    1172:
        FuUnicodeCodepointCaseConvert := 1173;
        RETURN;
    1173:
        FuUnicodeCodepointCaseConvert := 1172;
        RETURN;
    1174:
        FuUnicodeCodepointCaseConvert := 1175;
        RETURN;
    1175:
        FuUnicodeCodepointCaseConvert := 1174;
        RETURN;
    1176:
        FuUnicodeCodepointCaseConvert := 1177;
        RETURN;
    1177:
        FuUnicodeCodepointCaseConvert := 1176;
        RETURN;
    1178:
        FuUnicodeCodepointCaseConvert := 1179;
        RETURN;
    1179:
        FuUnicodeCodepointCaseConvert := 1178;
        RETURN;
    1180:
        FuUnicodeCodepointCaseConvert := 1181;
        RETURN;
    1181:
        FuUnicodeCodepointCaseConvert := 1180;
        RETURN;
    1182:
        FuUnicodeCodepointCaseConvert := 1183;
        RETURN;
    1183:
        FuUnicodeCodepointCaseConvert := 1182;
        RETURN;
    1184:
        FuUnicodeCodepointCaseConvert := 1185;
        RETURN;
    1185:
        FuUnicodeCodepointCaseConvert := 1184;
        RETURN;
    1186:
        FuUnicodeCodepointCaseConvert := 1187;
        RETURN;
    1187:
        FuUnicodeCodepointCaseConvert := 1186;
        RETURN;
    1188:
        FuUnicodeCodepointCaseConvert := 1189;
        RETURN;
    1189:
        FuUnicodeCodepointCaseConvert := 1188;
        RETURN;
    1190:
        FuUnicodeCodepointCaseConvert := 1191;
        RETURN;
    1191:
        FuUnicodeCodepointCaseConvert := 1190;
        RETURN;
    1192:
        FuUnicodeCodepointCaseConvert := 1193;
        RETURN;
    1193:
        FuUnicodeCodepointCaseConvert := 1192;
        RETURN;
    1194:
        FuUnicodeCodepointCaseConvert := 1195;
        RETURN;
    1195:
        FuUnicodeCodepointCaseConvert := 1194;
        RETURN;
    1196:
        FuUnicodeCodepointCaseConvert := 1197;
        RETURN;
    1197:
        FuUnicodeCodepointCaseConvert := 1196;
        RETURN;
    1198:
        FuUnicodeCodepointCaseConvert := 1199;
        RETURN;
    1199:
        FuUnicodeCodepointCaseConvert := 1198;
        RETURN;
    1200:
        FuUnicodeCodepointCaseConvert := 1201;
        RETURN;
    1201:
        FuUnicodeCodepointCaseConvert := 1200;
        RETURN;
    1202:
        FuUnicodeCodepointCaseConvert := 1203;
        RETURN;
    1203:
        FuUnicodeCodepointCaseConvert := 1202;
        RETURN;
    1204:
        FuUnicodeCodepointCaseConvert := 1205;
        RETURN;
    1205:
        FuUnicodeCodepointCaseConvert := 1204;
        RETURN;
    1206:
        FuUnicodeCodepointCaseConvert := 1207;
        RETURN;
    1207:
        FuUnicodeCodepointCaseConvert := 1206;
        RETURN;
    1208:
        FuUnicodeCodepointCaseConvert := 1209;
        RETURN;
    1209:
        FuUnicodeCodepointCaseConvert := 1208;
        RETURN;
    1210:
        FuUnicodeCodepointCaseConvert := 1211;
        RETURN;
    1211:
        FuUnicodeCodepointCaseConvert := 1210;
        RETURN;
    1212:
        FuUnicodeCodepointCaseConvert := 1213;
        RETURN;
    1213:
        FuUnicodeCodepointCaseConvert := 1212;
        RETURN;
    1214:
        FuUnicodeCodepointCaseConvert := 1215;
        RETURN;
    1215:
        FuUnicodeCodepointCaseConvert := 1214;
        RETURN;
    1216:
        FuUnicodeCodepointCaseConvert := 1231;
        RETURN;
    1217:
        FuUnicodeCodepointCaseConvert := 1218;
        RETURN;
    1218:
        FuUnicodeCodepointCaseConvert := 1217;
        RETURN;
    1219:
        FuUnicodeCodepointCaseConvert := 1220;
        RETURN;
    1220:
        FuUnicodeCodepointCaseConvert := 1219;
        RETURN;
    1221:
        FuUnicodeCodepointCaseConvert := 1222;
        RETURN;
    1222:
        FuUnicodeCodepointCaseConvert := 1221;
        RETURN;
    1223:
        FuUnicodeCodepointCaseConvert := 1224;
        RETURN;
    1224:
        FuUnicodeCodepointCaseConvert := 1223;
        RETURN;
    1225:
        FuUnicodeCodepointCaseConvert := 1226;
        RETURN;
    1226:
        FuUnicodeCodepointCaseConvert := 1225;
        RETURN;
    1227:
        FuUnicodeCodepointCaseConvert := 1228;
        RETURN;
    1228:
        FuUnicodeCodepointCaseConvert := 1227;
        RETURN;
    1229:
        FuUnicodeCodepointCaseConvert := 1230;
        RETURN;
    1230:
        FuUnicodeCodepointCaseConvert := 1229;
        RETURN;
    1231:
        FuUnicodeCodepointCaseConvert := 1216;
        RETURN;
    1232:
        FuUnicodeCodepointCaseConvert := 1233;
        RETURN;
    1233:
        FuUnicodeCodepointCaseConvert := 1232;
        RETURN;
    1234:
        FuUnicodeCodepointCaseConvert := 1235;
        RETURN;
    1235:
        FuUnicodeCodepointCaseConvert := 1234;
        RETURN;
    1236:
        FuUnicodeCodepointCaseConvert := 1237;
        RETURN;
    1237:
        FuUnicodeCodepointCaseConvert := 1236;
        RETURN;
    1238:
        FuUnicodeCodepointCaseConvert := 1239;
        RETURN;
    1239:
        FuUnicodeCodepointCaseConvert := 1238;
        RETURN;
    1240:
        FuUnicodeCodepointCaseConvert := 1241;
        RETURN;
    1241:
        FuUnicodeCodepointCaseConvert := 1240;
        RETURN;
    1242:
        FuUnicodeCodepointCaseConvert := 1243;
        RETURN;
    1243:
        FuUnicodeCodepointCaseConvert := 1242;
        RETURN;
    1244:
        FuUnicodeCodepointCaseConvert := 1245;
        RETURN;
    1245:
        FuUnicodeCodepointCaseConvert := 1244;
        RETURN;
    1246:
        FuUnicodeCodepointCaseConvert := 1247;
        RETURN;
    1247:
        FuUnicodeCodepointCaseConvert := 1246;
        RETURN;
    1248:
        FuUnicodeCodepointCaseConvert := 1249;
        RETURN;
    1249:
        FuUnicodeCodepointCaseConvert := 1248;
        RETURN;
    1250:
        FuUnicodeCodepointCaseConvert := 1251;
        RETURN;
    1251:
        FuUnicodeCodepointCaseConvert := 1250;
        RETURN;
    1252:
        FuUnicodeCodepointCaseConvert := 1253;
        RETURN;
    1253:
        FuUnicodeCodepointCaseConvert := 1252;
        RETURN;
    1254:
        FuUnicodeCodepointCaseConvert := 1255;
        RETURN;
    1255:
        FuUnicodeCodepointCaseConvert := 1254;
        RETURN;
    1256:
        FuUnicodeCodepointCaseConvert := 1257;
        RETURN;
    1257:
        FuUnicodeCodepointCaseConvert := 1256;
        RETURN;
    1258:
        FuUnicodeCodepointCaseConvert := 1259;
        RETURN;
    1259:
        FuUnicodeCodepointCaseConvert := 1258;
        RETURN;
    1260:
        FuUnicodeCodepointCaseConvert := 1261;
        RETURN;
    1261:
        FuUnicodeCodepointCaseConvert := 1260;
        RETURN;
    1262:
        FuUnicodeCodepointCaseConvert := 1263;
        RETURN;
    1263:
        FuUnicodeCodepointCaseConvert := 1262;
        RETURN;
    1264:
        FuUnicodeCodepointCaseConvert := 1265;
        RETURN;
    1265:
        FuUnicodeCodepointCaseConvert := 1264;
        RETURN;
    1266:
        FuUnicodeCodepointCaseConvert := 1267;
        RETURN;
    1267:
        FuUnicodeCodepointCaseConvert := 1266;
        RETURN;
    1268:
        FuUnicodeCodepointCaseConvert := 1269;
        RETURN;
    1269:
        FuUnicodeCodepointCaseConvert := 1268;
        RETURN;
    1270:
        FuUnicodeCodepointCaseConvert := 1271;
        RETURN;
    1271:
        FuUnicodeCodepointCaseConvert := 1270;
        RETURN;
    1272:
        FuUnicodeCodepointCaseConvert := 1273;
        RETURN;
    1273:
        FuUnicodeCodepointCaseConvert := 1272;
        RETURN;
    1274:
        FuUnicodeCodepointCaseConvert := 1275;
        RETURN;
    1275:
        FuUnicodeCodepointCaseConvert := 1274;
        RETURN;
    1276:
        FuUnicodeCodepointCaseConvert := 1277;
        RETURN;
    1277:
        FuUnicodeCodepointCaseConvert := 1276;
        RETURN;
    1278:
        FuUnicodeCodepointCaseConvert := 1279;
        RETURN;
    1279:
        FuUnicodeCodepointCaseConvert := 1278;
        RETURN;
    1280:
        FuUnicodeCodepointCaseConvert := 1281;
        RETURN;
    1281:
        FuUnicodeCodepointCaseConvert := 1280;
        RETURN;
    1282:
        FuUnicodeCodepointCaseConvert := 1283;
        RETURN;
    1283:
        FuUnicodeCodepointCaseConvert := 1282;
        RETURN;
    1284:
        FuUnicodeCodepointCaseConvert := 1285;
        RETURN;
    1285:
        FuUnicodeCodepointCaseConvert := 1284;
        RETURN;
    1286:
        FuUnicodeCodepointCaseConvert := 1287;
        RETURN;
    1287:
        FuUnicodeCodepointCaseConvert := 1286;
        RETURN;
    1288:
        FuUnicodeCodepointCaseConvert := 1289;
        RETURN;
    1289:
        FuUnicodeCodepointCaseConvert := 1288;
        RETURN;
    1290:
        FuUnicodeCodepointCaseConvert := 1291;
        RETURN;
    1291:
        FuUnicodeCodepointCaseConvert := 1290;
        RETURN;
    1292:
        FuUnicodeCodepointCaseConvert := 1293;
        RETURN;
    1293:
        FuUnicodeCodepointCaseConvert := 1292;
        RETURN;
    1294:
        FuUnicodeCodepointCaseConvert := 1295;
        RETURN;
    1295:
        FuUnicodeCodepointCaseConvert := 1294;
        RETURN;
    1296:
        FuUnicodeCodepointCaseConvert := 1297;
        RETURN;
    1297:
        FuUnicodeCodepointCaseConvert := 1296;
        RETURN;
    1298:
        FuUnicodeCodepointCaseConvert := 1299;
        RETURN;
    1299:
        FuUnicodeCodepointCaseConvert := 1298;
        RETURN;
    1300:
        FuUnicodeCodepointCaseConvert := 1301;
        RETURN;
    1301:
        FuUnicodeCodepointCaseConvert := 1300;
        RETURN;
    1302:
        FuUnicodeCodepointCaseConvert := 1303;
        RETURN;
    1303:
        FuUnicodeCodepointCaseConvert := 1302;
        RETURN;
    1304:
        FuUnicodeCodepointCaseConvert := 1305;
        RETURN;
    1305:
        FuUnicodeCodepointCaseConvert := 1304;
        RETURN;
    1306:
        FuUnicodeCodepointCaseConvert := 1307;
        RETURN;
    1307:
        FuUnicodeCodepointCaseConvert := 1306;
        RETURN;
    1308:
        FuUnicodeCodepointCaseConvert := 1309;
        RETURN;
    1309:
        FuUnicodeCodepointCaseConvert := 1308;
        RETURN;
    1310:
        FuUnicodeCodepointCaseConvert := 1311;
        RETURN;
    1311:
        FuUnicodeCodepointCaseConvert := 1310;
        RETURN;
    1312:
        FuUnicodeCodepointCaseConvert := 1313;
        RETURN;
    1313:
        FuUnicodeCodepointCaseConvert := 1312;
        RETURN;
    1314:
        FuUnicodeCodepointCaseConvert := 1315;
        RETURN;
    1315:
        FuUnicodeCodepointCaseConvert := 1314;
        RETURN;
    1316:
        FuUnicodeCodepointCaseConvert := 1317;
        RETURN;
    1317:
        FuUnicodeCodepointCaseConvert := 1316;
        RETURN;
    1318:
        FuUnicodeCodepointCaseConvert := 1319;
        RETURN;
    1319:
        FuUnicodeCodepointCaseConvert := 1318;
        RETURN;
    1320:
        FuUnicodeCodepointCaseConvert := 1321;
        RETURN;
    1321:
        FuUnicodeCodepointCaseConvert := 1320;
        RETURN;
    1322:
        FuUnicodeCodepointCaseConvert := 1323;
        RETURN;
    1323:
        FuUnicodeCodepointCaseConvert := 1322;
        RETURN;
    1324:
        FuUnicodeCodepointCaseConvert := 1325;
        RETURN;
    1325:
        FuUnicodeCodepointCaseConvert := 1324;
        RETURN;
    1326:
        FuUnicodeCodepointCaseConvert := 1327;
        RETURN;
    1327:
        FuUnicodeCodepointCaseConvert := 1326;
        RETURN;
    1329:
        FuUnicodeCodepointCaseConvert := 1377;
        RETURN;
    1330:
        FuUnicodeCodepointCaseConvert := 1378;
        RETURN;
    1331:
        FuUnicodeCodepointCaseConvert := 1379;
        RETURN;
    1332:
        FuUnicodeCodepointCaseConvert := 1380;
        RETURN;
    1333:
        FuUnicodeCodepointCaseConvert := 1381;
        RETURN;
    1334:
        FuUnicodeCodepointCaseConvert := 1382;
        RETURN;
    1335:
        FuUnicodeCodepointCaseConvert := 1383;
        RETURN;
    1336:
        FuUnicodeCodepointCaseConvert := 1384;
        RETURN;
    1337:
        FuUnicodeCodepointCaseConvert := 1385;
        RETURN;
    1338:
        FuUnicodeCodepointCaseConvert := 1386;
        RETURN;
    1339:
        FuUnicodeCodepointCaseConvert := 1387;
        RETURN;
    1340:
        FuUnicodeCodepointCaseConvert := 1388;
        RETURN;
    1341:
        FuUnicodeCodepointCaseConvert := 1389;
        RETURN;
    1342:
        FuUnicodeCodepointCaseConvert := 1390;
        RETURN;
    1343:
        FuUnicodeCodepointCaseConvert := 1391;
        RETURN;
    1344:
        FuUnicodeCodepointCaseConvert := 1392;
        RETURN;
    1345:
        FuUnicodeCodepointCaseConvert := 1393;
        RETURN;
    1346:
        FuUnicodeCodepointCaseConvert := 1394;
        RETURN;
    1347:
        FuUnicodeCodepointCaseConvert := 1395;
        RETURN;
    1348:
        FuUnicodeCodepointCaseConvert := 1396;
        RETURN;
    1349:
        FuUnicodeCodepointCaseConvert := 1397;
        RETURN;
    1350:
        FuUnicodeCodepointCaseConvert := 1398;
        RETURN;
    1351:
        FuUnicodeCodepointCaseConvert := 1399;
        RETURN;
    1352:
        FuUnicodeCodepointCaseConvert := 1400;
        RETURN;
    1353:
        FuUnicodeCodepointCaseConvert := 1401;
        RETURN;
    1354:
        FuUnicodeCodepointCaseConvert := 1402;
        RETURN;
    1355:
        FuUnicodeCodepointCaseConvert := 1403;
        RETURN;
    1356:
        FuUnicodeCodepointCaseConvert := 1404;
        RETURN;
    1357:
        FuUnicodeCodepointCaseConvert := 1405;
        RETURN;
    1358:
        FuUnicodeCodepointCaseConvert := 1406;
        RETURN;
    1359:
        FuUnicodeCodepointCaseConvert := 1407;
        RETURN;
    1360:
        FuUnicodeCodepointCaseConvert := 1408;
        RETURN;
    1361:
        FuUnicodeCodepointCaseConvert := 1409;
        RETURN;
    1362:
        FuUnicodeCodepointCaseConvert := 1410;
        RETURN;
    1363:
        FuUnicodeCodepointCaseConvert := 1411;
        RETURN;
    1364:
        FuUnicodeCodepointCaseConvert := 1412;
        RETURN;
    1365:
        FuUnicodeCodepointCaseConvert := 1413;
        RETURN;
    1366:
        FuUnicodeCodepointCaseConvert := 1414;
        RETURN;
    1377:
        FuUnicodeCodepointCaseConvert := 1329;
        RETURN;
    1378:
        FuUnicodeCodepointCaseConvert := 1330;
        RETURN;
    1379:
        FuUnicodeCodepointCaseConvert := 1331;
        RETURN;
    1380:
        FuUnicodeCodepointCaseConvert := 1332;
        RETURN;
    1381:
        FuUnicodeCodepointCaseConvert := 1333;
        RETURN;
    1382:
        FuUnicodeCodepointCaseConvert := 1334;
        RETURN;
    1383:
        FuUnicodeCodepointCaseConvert := 1335;
        RETURN;
    1384:
        FuUnicodeCodepointCaseConvert := 1336;
        RETURN;
    1385:
        FuUnicodeCodepointCaseConvert := 1337;
        RETURN;
    1386:
        FuUnicodeCodepointCaseConvert := 1338;
        RETURN;
    1387:
        FuUnicodeCodepointCaseConvert := 1339;
        RETURN;
    1388:
        FuUnicodeCodepointCaseConvert := 1340;
        RETURN;
    1389:
        FuUnicodeCodepointCaseConvert := 1341;
        RETURN;
    1390:
        FuUnicodeCodepointCaseConvert := 1342;
        RETURN;
    1391:
        FuUnicodeCodepointCaseConvert := 1343;
        RETURN;
    1392:
        FuUnicodeCodepointCaseConvert := 1344;
        RETURN;
    1393:
        FuUnicodeCodepointCaseConvert := 1345;
        RETURN;
    1394:
        FuUnicodeCodepointCaseConvert := 1346;
        RETURN;
    1395:
        FuUnicodeCodepointCaseConvert := 1347;
        RETURN;
    1396:
        FuUnicodeCodepointCaseConvert := 1348;
        RETURN;
    1397:
        FuUnicodeCodepointCaseConvert := 1349;
        RETURN;
    1398:
        FuUnicodeCodepointCaseConvert := 1350;
        RETURN;
    1399:
        FuUnicodeCodepointCaseConvert := 1351;
        RETURN;
    1400:
        FuUnicodeCodepointCaseConvert := 1352;
        RETURN;
    1401:
        FuUnicodeCodepointCaseConvert := 1353;
        RETURN;
    1402:
        FuUnicodeCodepointCaseConvert := 1354;
        RETURN;
    1403:
        FuUnicodeCodepointCaseConvert := 1355;
        RETURN;
    1404:
        FuUnicodeCodepointCaseConvert := 1356;
        RETURN;
    1405:
        FuUnicodeCodepointCaseConvert := 1357;
        RETURN;
    1406:
        FuUnicodeCodepointCaseConvert := 1358;
        RETURN;
    1407:
        FuUnicodeCodepointCaseConvert := 1359;
        RETURN;
    1408:
        FuUnicodeCodepointCaseConvert := 1360;
        RETURN;
    1409:
        FuUnicodeCodepointCaseConvert := 1361;
        RETURN;
    1410:
        FuUnicodeCodepointCaseConvert := 1362;
        RETURN;
    1411:
        FuUnicodeCodepointCaseConvert := 1363;
        RETURN;
    1412:
        FuUnicodeCodepointCaseConvert := 1364;
        RETURN;
    1413:
        FuUnicodeCodepointCaseConvert := 1365;
        RETURN;
    1414:
        FuUnicodeCodepointCaseConvert := 1366;
        RETURN;
    4256:
        FuUnicodeCodepointCaseConvert := 11520;
        RETURN;
    4257:
        FuUnicodeCodepointCaseConvert := 11521;
        RETURN;
    4258:
        FuUnicodeCodepointCaseConvert := 11522;
        RETURN;
    4259:
        FuUnicodeCodepointCaseConvert := 11523;
        RETURN;
    4260:
        FuUnicodeCodepointCaseConvert := 11524;
        RETURN;
    4261:
        FuUnicodeCodepointCaseConvert := 11525;
        RETURN;
    4262:
        FuUnicodeCodepointCaseConvert := 11526;
        RETURN;
    4263:
        FuUnicodeCodepointCaseConvert := 11527;
        RETURN;
    4264:
        FuUnicodeCodepointCaseConvert := 11528;
        RETURN;
    4265:
        FuUnicodeCodepointCaseConvert := 11529;
        RETURN;
    4266:
        FuUnicodeCodepointCaseConvert := 11530;
        RETURN;
    4267:
        FuUnicodeCodepointCaseConvert := 11531;
        RETURN;
    4268:
        FuUnicodeCodepointCaseConvert := 11532;
        RETURN;
    4269:
        FuUnicodeCodepointCaseConvert := 11533;
        RETURN;
    4270:
        FuUnicodeCodepointCaseConvert := 11534;
        RETURN;
    4271:
        FuUnicodeCodepointCaseConvert := 11535;
        RETURN;
    4272:
        FuUnicodeCodepointCaseConvert := 11536;
        RETURN;
    4273:
        FuUnicodeCodepointCaseConvert := 11537;
        RETURN;
    4274:
        FuUnicodeCodepointCaseConvert := 11538;
        RETURN;
    4275:
        FuUnicodeCodepointCaseConvert := 11539;
        RETURN;
    4276:
        FuUnicodeCodepointCaseConvert := 11540;
        RETURN;
    4277:
        FuUnicodeCodepointCaseConvert := 11541;
        RETURN;
    4278:
        FuUnicodeCodepointCaseConvert := 11542;
        RETURN;
    4279:
        FuUnicodeCodepointCaseConvert := 11543;
        RETURN;
    4280:
        FuUnicodeCodepointCaseConvert := 11544;
        RETURN;
    4281:
        FuUnicodeCodepointCaseConvert := 11545;
        RETURN;
    4282:
        FuUnicodeCodepointCaseConvert := 11546;
        RETURN;
    4283:
        FuUnicodeCodepointCaseConvert := 11547;
        RETURN;
    4284:
        FuUnicodeCodepointCaseConvert := 11548;
        RETURN;
    4285:
        FuUnicodeCodepointCaseConvert := 11549;
        RETURN;
    4286:
        FuUnicodeCodepointCaseConvert := 11550;
        RETURN;
    4287:
        FuUnicodeCodepointCaseConvert := 11551;
        RETURN;
    4288:
        FuUnicodeCodepointCaseConvert := 11552;
        RETURN;
    4289:
        FuUnicodeCodepointCaseConvert := 11553;
        RETURN;
    4290:
        FuUnicodeCodepointCaseConvert := 11554;
        RETURN;
    4291:
        FuUnicodeCodepointCaseConvert := 11555;
        RETURN;
    4292:
        FuUnicodeCodepointCaseConvert := 11556;
        RETURN;
    4293:
        FuUnicodeCodepointCaseConvert := 11557;
        RETURN;
    4295:
        FuUnicodeCodepointCaseConvert := 11559;
        RETURN;
    4301:
        FuUnicodeCodepointCaseConvert := 11565;
        RETURN;
    4304:
        FuUnicodeCodepointCaseConvert := 4304;
        RETURN;
    4305:
        FuUnicodeCodepointCaseConvert := 4305;
        RETURN;
    4306:
        FuUnicodeCodepointCaseConvert := 4306;
        RETURN;
    4307:
        FuUnicodeCodepointCaseConvert := 4307;
        RETURN;
    4308:
        FuUnicodeCodepointCaseConvert := 4308;
        RETURN;
    4309:
        FuUnicodeCodepointCaseConvert := 4309;
        RETURN;
    4310:
        FuUnicodeCodepointCaseConvert := 4310;
        RETURN;
    4311:
        FuUnicodeCodepointCaseConvert := 4311;
        RETURN;
    4312:
        FuUnicodeCodepointCaseConvert := 4312;
        RETURN;
    4313:
        FuUnicodeCodepointCaseConvert := 4313;
        RETURN;
    4314:
        FuUnicodeCodepointCaseConvert := 4314;
        RETURN;
    4315:
        FuUnicodeCodepointCaseConvert := 4315;
        RETURN;
    4316:
        FuUnicodeCodepointCaseConvert := 4316;
        RETURN;
    4317:
        FuUnicodeCodepointCaseConvert := 4317;
        RETURN;
    4318:
        FuUnicodeCodepointCaseConvert := 4318;
        RETURN;
    4319:
        FuUnicodeCodepointCaseConvert := 4319;
        RETURN;
    4320:
        FuUnicodeCodepointCaseConvert := 4320;
        RETURN;
    4321:
        FuUnicodeCodepointCaseConvert := 4321;
        RETURN;
    4322:
        FuUnicodeCodepointCaseConvert := 4322;
        RETURN;
    4323:
        FuUnicodeCodepointCaseConvert := 4323;
        RETURN;
    4324:
        FuUnicodeCodepointCaseConvert := 4324;
        RETURN;
    4325:
        FuUnicodeCodepointCaseConvert := 4325;
        RETURN;
    4326:
        FuUnicodeCodepointCaseConvert := 4326;
        RETURN;
    4327:
        FuUnicodeCodepointCaseConvert := 4327;
        RETURN;
    4328:
        FuUnicodeCodepointCaseConvert := 4328;
        RETURN;
    4329:
        FuUnicodeCodepointCaseConvert := 4329;
        RETURN;
    4330:
        FuUnicodeCodepointCaseConvert := 4330;
        RETURN;
    4331:
        FuUnicodeCodepointCaseConvert := 4331;
        RETURN;
    4332:
        FuUnicodeCodepointCaseConvert := 4332;
        RETURN;
    4333:
        FuUnicodeCodepointCaseConvert := 4333;
        RETURN;
    4334:
        FuUnicodeCodepointCaseConvert := 4334;
        RETURN;
    4335:
        FuUnicodeCodepointCaseConvert := 4335;
        RETURN;
    4336:
        FuUnicodeCodepointCaseConvert := 4336;
        RETURN;
    4337:
        FuUnicodeCodepointCaseConvert := 4337;
        RETURN;
    4338:
        FuUnicodeCodepointCaseConvert := 4338;
        RETURN;
    4339:
        FuUnicodeCodepointCaseConvert := 4339;
        RETURN;
    4340:
        FuUnicodeCodepointCaseConvert := 4340;
        RETURN;
    4341:
        FuUnicodeCodepointCaseConvert := 4341;
        RETURN;
    4342:
        FuUnicodeCodepointCaseConvert := 4342;
        RETURN;
    4343:
        FuUnicodeCodepointCaseConvert := 4343;
        RETURN;
    4344:
        FuUnicodeCodepointCaseConvert := 4344;
        RETURN;
    4345:
        FuUnicodeCodepointCaseConvert := 4345;
        RETURN;
    4346:
        FuUnicodeCodepointCaseConvert := 4346;
        RETURN;
    4349:
        FuUnicodeCodepointCaseConvert := 4349;
        RETURN;
    4350:
        FuUnicodeCodepointCaseConvert := 4350;
        RETURN;
    4351:
        FuUnicodeCodepointCaseConvert := 4351;
        RETURN;
    5024:
        FuUnicodeCodepointCaseConvert := 43888;
        RETURN;
    5025:
        FuUnicodeCodepointCaseConvert := 43889;
        RETURN;
    5026:
        FuUnicodeCodepointCaseConvert := 43890;
        RETURN;
    5027:
        FuUnicodeCodepointCaseConvert := 43891;
        RETURN;
    5028:
        FuUnicodeCodepointCaseConvert := 43892;
        RETURN;
    5029:
        FuUnicodeCodepointCaseConvert := 43893;
        RETURN;
    5030:
        FuUnicodeCodepointCaseConvert := 43894;
        RETURN;
    5031:
        FuUnicodeCodepointCaseConvert := 43895;
        RETURN;
    5032:
        FuUnicodeCodepointCaseConvert := 43896;
        RETURN;
    5033:
        FuUnicodeCodepointCaseConvert := 43897;
        RETURN;
    5034:
        FuUnicodeCodepointCaseConvert := 43898;
        RETURN;
    5035:
        FuUnicodeCodepointCaseConvert := 43899;
        RETURN;
    5036:
        FuUnicodeCodepointCaseConvert := 43900;
        RETURN;
    5037:
        FuUnicodeCodepointCaseConvert := 43901;
        RETURN;
    5038:
        FuUnicodeCodepointCaseConvert := 43902;
        RETURN;
    5039:
        FuUnicodeCodepointCaseConvert := 43903;
        RETURN;
    5040:
        FuUnicodeCodepointCaseConvert := 43904;
        RETURN;
    5041:
        FuUnicodeCodepointCaseConvert := 43905;
        RETURN;
    5042:
        FuUnicodeCodepointCaseConvert := 43906;
        RETURN;
    5043:
        FuUnicodeCodepointCaseConvert := 43907;
        RETURN;
    5044:
        FuUnicodeCodepointCaseConvert := 43908;
        RETURN;
    5045:
        FuUnicodeCodepointCaseConvert := 43909;
        RETURN;
    5046:
        FuUnicodeCodepointCaseConvert := 43910;
        RETURN;
    5047:
        FuUnicodeCodepointCaseConvert := 43911;
        RETURN;
    5048:
        FuUnicodeCodepointCaseConvert := 43912;
        RETURN;
    5049:
        FuUnicodeCodepointCaseConvert := 43913;
        RETURN;
    5050:
        FuUnicodeCodepointCaseConvert := 43914;
        RETURN;
    5051:
        FuUnicodeCodepointCaseConvert := 43915;
        RETURN;
    5052:
        FuUnicodeCodepointCaseConvert := 43916;
        RETURN;
    5053:
        FuUnicodeCodepointCaseConvert := 43917;
        RETURN;
    5054:
        FuUnicodeCodepointCaseConvert := 43918;
        RETURN;
    5055:
        FuUnicodeCodepointCaseConvert := 43919;
        RETURN;
    5056:
        FuUnicodeCodepointCaseConvert := 43920;
        RETURN;
    5057:
        FuUnicodeCodepointCaseConvert := 43921;
        RETURN;
    5058:
        FuUnicodeCodepointCaseConvert := 43922;
        RETURN;
    5059:
        FuUnicodeCodepointCaseConvert := 43923;
        RETURN;
    5060:
        FuUnicodeCodepointCaseConvert := 43924;
        RETURN;
    5061:
        FuUnicodeCodepointCaseConvert := 43925;
        RETURN;
    5062:
        FuUnicodeCodepointCaseConvert := 43926;
        RETURN;
    5063:
        FuUnicodeCodepointCaseConvert := 43927;
        RETURN;
    5064:
        FuUnicodeCodepointCaseConvert := 43928;
        RETURN;
    5065:
        FuUnicodeCodepointCaseConvert := 43929;
        RETURN;
    5066:
        FuUnicodeCodepointCaseConvert := 43930;
        RETURN;
    5067:
        FuUnicodeCodepointCaseConvert := 43931;
        RETURN;
    5068:
        FuUnicodeCodepointCaseConvert := 43932;
        RETURN;
    5069:
        FuUnicodeCodepointCaseConvert := 43933;
        RETURN;
    5070:
        FuUnicodeCodepointCaseConvert := 43934;
        RETURN;
    5071:
        FuUnicodeCodepointCaseConvert := 43935;
        RETURN;
    5072:
        FuUnicodeCodepointCaseConvert := 43936;
        RETURN;
    5073:
        FuUnicodeCodepointCaseConvert := 43937;
        RETURN;
    5074:
        FuUnicodeCodepointCaseConvert := 43938;
        RETURN;
    5075:
        FuUnicodeCodepointCaseConvert := 43939;
        RETURN;
    5076:
        FuUnicodeCodepointCaseConvert := 43940;
        RETURN;
    5077:
        FuUnicodeCodepointCaseConvert := 43941;
        RETURN;
    5078:
        FuUnicodeCodepointCaseConvert := 43942;
        RETURN;
    5079:
        FuUnicodeCodepointCaseConvert := 43943;
        RETURN;
    5080:
        FuUnicodeCodepointCaseConvert := 43944;
        RETURN;
    5081:
        FuUnicodeCodepointCaseConvert := 43945;
        RETURN;
    5082:
        FuUnicodeCodepointCaseConvert := 43946;
        RETURN;
    5083:
        FuUnicodeCodepointCaseConvert := 43947;
        RETURN;
    5084:
        FuUnicodeCodepointCaseConvert := 43948;
        RETURN;
    5085:
        FuUnicodeCodepointCaseConvert := 43949;
        RETURN;
    5086:
        FuUnicodeCodepointCaseConvert := 43950;
        RETURN;
    5087:
        FuUnicodeCodepointCaseConvert := 43951;
        RETURN;
    5088:
        FuUnicodeCodepointCaseConvert := 43952;
        RETURN;
    5089:
        FuUnicodeCodepointCaseConvert := 43953;
        RETURN;
    5090:
        FuUnicodeCodepointCaseConvert := 43954;
        RETURN;
    5091:
        FuUnicodeCodepointCaseConvert := 43955;
        RETURN;
    5092:
        FuUnicodeCodepointCaseConvert := 43956;
        RETURN;
    5093:
        FuUnicodeCodepointCaseConvert := 43957;
        RETURN;
    5094:
        FuUnicodeCodepointCaseConvert := 43958;
        RETURN;
    5095:
        FuUnicodeCodepointCaseConvert := 43959;
        RETURN;
    5096:
        FuUnicodeCodepointCaseConvert := 43960;
        RETURN;
    5097:
        FuUnicodeCodepointCaseConvert := 43961;
        RETURN;
    5098:
        FuUnicodeCodepointCaseConvert := 43962;
        RETURN;
    5099:
        FuUnicodeCodepointCaseConvert := 43963;
        RETURN;
    5100:
        FuUnicodeCodepointCaseConvert := 43964;
        RETURN;
    5101:
        FuUnicodeCodepointCaseConvert := 43965;
        RETURN;
    5102:
        FuUnicodeCodepointCaseConvert := 43966;
        RETURN;
    5103:
        FuUnicodeCodepointCaseConvert := 43967;
        RETURN;
    5104:
        FuUnicodeCodepointCaseConvert := 5112;
        RETURN;
    5105:
        FuUnicodeCodepointCaseConvert := 5113;
        RETURN;
    5106:
        FuUnicodeCodepointCaseConvert := 5114;
        RETURN;
    5107:
        FuUnicodeCodepointCaseConvert := 5115;
        RETURN;
    5108:
        FuUnicodeCodepointCaseConvert := 5116;
        RETURN;
    5109:
        FuUnicodeCodepointCaseConvert := 5117;
        RETURN;
    5112:
        FuUnicodeCodepointCaseConvert := 5104;
        RETURN;
    5113:
        FuUnicodeCodepointCaseConvert := 5105;
        RETURN;
    5114:
        FuUnicodeCodepointCaseConvert := 5106;
        RETURN;
    5115:
        FuUnicodeCodepointCaseConvert := 5107;
        RETURN;
    5116:
        FuUnicodeCodepointCaseConvert := 5108;
        RETURN;
    5117:
        FuUnicodeCodepointCaseConvert := 5109;
        RETURN;
    7296:
        FuUnicodeCodepointCaseConvert := 1042;
        RETURN;
    7297:
        FuUnicodeCodepointCaseConvert := 1044;
        RETURN;
    7298:
        FuUnicodeCodepointCaseConvert := 1054;
        RETURN;
    7299:
        FuUnicodeCodepointCaseConvert := 1057;
        RETURN;
    7300:
        FuUnicodeCodepointCaseConvert := 1058;
        RETURN;
    7301:
        FuUnicodeCodepointCaseConvert := 1058;
        RETURN;
    7302:
        FuUnicodeCodepointCaseConvert := 1066;
        RETURN;
    7303:
        FuUnicodeCodepointCaseConvert := 1122;
        RETURN;
    7304:
        FuUnicodeCodepointCaseConvert := 42570;
        RETURN;
    7312:
        FuUnicodeCodepointCaseConvert := 4304;
        RETURN;
    7313:
        FuUnicodeCodepointCaseConvert := 4305;
        RETURN;
    7314:
        FuUnicodeCodepointCaseConvert := 4306;
        RETURN;
    7315:
        FuUnicodeCodepointCaseConvert := 4307;
        RETURN;
    7316:
        FuUnicodeCodepointCaseConvert := 4308;
        RETURN;
    7317:
        FuUnicodeCodepointCaseConvert := 4309;
        RETURN;
    7318:
        FuUnicodeCodepointCaseConvert := 4310;
        RETURN;
    7319:
        FuUnicodeCodepointCaseConvert := 4311;
        RETURN;
    7320:
        FuUnicodeCodepointCaseConvert := 4312;
        RETURN;
    7321:
        FuUnicodeCodepointCaseConvert := 4313;
        RETURN;
    7322:
        FuUnicodeCodepointCaseConvert := 4314;
        RETURN;
    7323:
        FuUnicodeCodepointCaseConvert := 4315;
        RETURN;
    7324:
        FuUnicodeCodepointCaseConvert := 4316;
        RETURN;
    7325:
        FuUnicodeCodepointCaseConvert := 4317;
        RETURN;
    7326:
        FuUnicodeCodepointCaseConvert := 4318;
        RETURN;
    7327:
        FuUnicodeCodepointCaseConvert := 4319;
        RETURN;
    7328:
        FuUnicodeCodepointCaseConvert := 4320;
        RETURN;
    7329:
        FuUnicodeCodepointCaseConvert := 4321;
        RETURN;
    7330:
        FuUnicodeCodepointCaseConvert := 4322;
        RETURN;
    7331:
        FuUnicodeCodepointCaseConvert := 4323;
        RETURN;
    7332:
        FuUnicodeCodepointCaseConvert := 4324;
        RETURN;
    7333:
        FuUnicodeCodepointCaseConvert := 4325;
        RETURN;
    7334:
        FuUnicodeCodepointCaseConvert := 4326;
        RETURN;
    7335:
        FuUnicodeCodepointCaseConvert := 4327;
        RETURN;
    7336:
        FuUnicodeCodepointCaseConvert := 4328;
        RETURN;
    7337:
        FuUnicodeCodepointCaseConvert := 4329;
        RETURN;
    7338:
        FuUnicodeCodepointCaseConvert := 4330;
        RETURN;
    7339:
        FuUnicodeCodepointCaseConvert := 4331;
        RETURN;
    7340:
        FuUnicodeCodepointCaseConvert := 4332;
        RETURN;
    7341:
        FuUnicodeCodepointCaseConvert := 4333;
        RETURN;
    7342:
        FuUnicodeCodepointCaseConvert := 4334;
        RETURN;
    7343:
        FuUnicodeCodepointCaseConvert := 4335;
        RETURN;
    7344:
        FuUnicodeCodepointCaseConvert := 4336;
        RETURN;
    7345:
        FuUnicodeCodepointCaseConvert := 4337;
        RETURN;
    7346:
        FuUnicodeCodepointCaseConvert := 4338;
        RETURN;
    7347:
        FuUnicodeCodepointCaseConvert := 4339;
        RETURN;
    7348:
        FuUnicodeCodepointCaseConvert := 4340;
        RETURN;
    7349:
        FuUnicodeCodepointCaseConvert := 4341;
        RETURN;
    7350:
        FuUnicodeCodepointCaseConvert := 4342;
        RETURN;
    7351:
        FuUnicodeCodepointCaseConvert := 4343;
        RETURN;
    7352:
        FuUnicodeCodepointCaseConvert := 4344;
        RETURN;
    7353:
        FuUnicodeCodepointCaseConvert := 4345;
        RETURN;
    7354:
        FuUnicodeCodepointCaseConvert := 4346;
        RETURN;
    7357:
        FuUnicodeCodepointCaseConvert := 4349;
        RETURN;
    7358:
        FuUnicodeCodepointCaseConvert := 4350;
        RETURN;
    7359:
        FuUnicodeCodepointCaseConvert := 4351;
        RETURN;
    7545:
        FuUnicodeCodepointCaseConvert := 42877;
        RETURN;
    7549:
        FuUnicodeCodepointCaseConvert := 11363;
        RETURN;
    7566:
        FuUnicodeCodepointCaseConvert := 42950;
        RETURN;
    7680:
        FuUnicodeCodepointCaseConvert := 7681;
        RETURN;
    7681:
        FuUnicodeCodepointCaseConvert := 7680;
        RETURN;
    7682:
        FuUnicodeCodepointCaseConvert := 7683;
        RETURN;
    7683:
        FuUnicodeCodepointCaseConvert := 7682;
        RETURN;
    7684:
        FuUnicodeCodepointCaseConvert := 7685;
        RETURN;
    7685:
        FuUnicodeCodepointCaseConvert := 7684;
        RETURN;
    7686:
        FuUnicodeCodepointCaseConvert := 7687;
        RETURN;
    7687:
        FuUnicodeCodepointCaseConvert := 7686;
        RETURN;
    7688:
        FuUnicodeCodepointCaseConvert := 7689;
        RETURN;
    7689:
        FuUnicodeCodepointCaseConvert := 7688;
        RETURN;
    7690:
        FuUnicodeCodepointCaseConvert := 7691;
        RETURN;
    7691:
        FuUnicodeCodepointCaseConvert := 7690;
        RETURN;
    7692:
        FuUnicodeCodepointCaseConvert := 7693;
        RETURN;
    7693:
        FuUnicodeCodepointCaseConvert := 7692;
        RETURN;
    7694:
        FuUnicodeCodepointCaseConvert := 7695;
        RETURN;
    7695:
        FuUnicodeCodepointCaseConvert := 7694;
        RETURN;
    7696:
        FuUnicodeCodepointCaseConvert := 7697;
        RETURN;
    7697:
        FuUnicodeCodepointCaseConvert := 7696;
        RETURN;
    7698:
        FuUnicodeCodepointCaseConvert := 7699;
        RETURN;
    7699:
        FuUnicodeCodepointCaseConvert := 7698;
        RETURN;
    7700:
        FuUnicodeCodepointCaseConvert := 7701;
        RETURN;
    7701:
        FuUnicodeCodepointCaseConvert := 7700;
        RETURN;
    7702:
        FuUnicodeCodepointCaseConvert := 7703;
        RETURN;
    7703:
        FuUnicodeCodepointCaseConvert := 7702;
        RETURN;
    7704:
        FuUnicodeCodepointCaseConvert := 7705;
        RETURN;
    7705:
        FuUnicodeCodepointCaseConvert := 7704;
        RETURN;
    7706:
        FuUnicodeCodepointCaseConvert := 7707;
        RETURN;
    7707:
        FuUnicodeCodepointCaseConvert := 7706;
        RETURN;
    7708:
        FuUnicodeCodepointCaseConvert := 7709;
        RETURN;
    7709:
        FuUnicodeCodepointCaseConvert := 7708;
        RETURN;
    7710:
        FuUnicodeCodepointCaseConvert := 7711;
        RETURN;
    7711:
        FuUnicodeCodepointCaseConvert := 7710;
        RETURN;
    7712:
        FuUnicodeCodepointCaseConvert := 7713;
        RETURN;
    7713:
        FuUnicodeCodepointCaseConvert := 7712;
        RETURN;
    7714:
        FuUnicodeCodepointCaseConvert := 7715;
        RETURN;
    7715:
        FuUnicodeCodepointCaseConvert := 7714;
        RETURN;
    7716:
        FuUnicodeCodepointCaseConvert := 7717;
        RETURN;
    7717:
        FuUnicodeCodepointCaseConvert := 7716;
        RETURN;
    7718:
        FuUnicodeCodepointCaseConvert := 7719;
        RETURN;
    7719:
        FuUnicodeCodepointCaseConvert := 7718;
        RETURN;
    7720:
        FuUnicodeCodepointCaseConvert := 7721;
        RETURN;
    7721:
        FuUnicodeCodepointCaseConvert := 7720;
        RETURN;
    7722:
        FuUnicodeCodepointCaseConvert := 7723;
        RETURN;
    7723:
        FuUnicodeCodepointCaseConvert := 7722;
        RETURN;
    7724:
        FuUnicodeCodepointCaseConvert := 7725;
        RETURN;
    7725:
        FuUnicodeCodepointCaseConvert := 7724;
        RETURN;
    7726:
        FuUnicodeCodepointCaseConvert := 7727;
        RETURN;
    7727:
        FuUnicodeCodepointCaseConvert := 7726;
        RETURN;
    7728:
        FuUnicodeCodepointCaseConvert := 7729;
        RETURN;
    7729:
        FuUnicodeCodepointCaseConvert := 7728;
        RETURN;
    7730:
        FuUnicodeCodepointCaseConvert := 7731;
        RETURN;
    7731:
        FuUnicodeCodepointCaseConvert := 7730;
        RETURN;
    7732:
        FuUnicodeCodepointCaseConvert := 7733;
        RETURN;
    7733:
        FuUnicodeCodepointCaseConvert := 7732;
        RETURN;
    7734:
        FuUnicodeCodepointCaseConvert := 7735;
        RETURN;
    7735:
        FuUnicodeCodepointCaseConvert := 7734;
        RETURN;
    7736:
        FuUnicodeCodepointCaseConvert := 7737;
        RETURN;
    7737:
        FuUnicodeCodepointCaseConvert := 7736;
        RETURN;
    7738:
        FuUnicodeCodepointCaseConvert := 7739;
        RETURN;
    7739:
        FuUnicodeCodepointCaseConvert := 7738;
        RETURN;
    7740:
        FuUnicodeCodepointCaseConvert := 7741;
        RETURN;
    7741:
        FuUnicodeCodepointCaseConvert := 7740;
        RETURN;
    7742:
        FuUnicodeCodepointCaseConvert := 7743;
        RETURN;
    7743:
        FuUnicodeCodepointCaseConvert := 7742;
        RETURN;
    7744:
        FuUnicodeCodepointCaseConvert := 7745;
        RETURN;
    7745:
        FuUnicodeCodepointCaseConvert := 7744;
        RETURN;
    7746:
        FuUnicodeCodepointCaseConvert := 7747;
        RETURN;
    7747:
        FuUnicodeCodepointCaseConvert := 7746;
        RETURN;
    7748:
        FuUnicodeCodepointCaseConvert := 7749;
        RETURN;
    7749:
        FuUnicodeCodepointCaseConvert := 7748;
        RETURN;
    7750:
        FuUnicodeCodepointCaseConvert := 7751;
        RETURN;
    7751:
        FuUnicodeCodepointCaseConvert := 7750;
        RETURN;
    7752:
        FuUnicodeCodepointCaseConvert := 7753;
        RETURN;
    7753:
        FuUnicodeCodepointCaseConvert := 7752;
        RETURN;
    7754:
        FuUnicodeCodepointCaseConvert := 7755;
        RETURN;
    7755:
        FuUnicodeCodepointCaseConvert := 7754;
        RETURN;
    7756:
        FuUnicodeCodepointCaseConvert := 7757;
        RETURN;
    7757:
        FuUnicodeCodepointCaseConvert := 7756;
        RETURN;
    7758:
        FuUnicodeCodepointCaseConvert := 7759;
        RETURN;
    7759:
        FuUnicodeCodepointCaseConvert := 7758;
        RETURN;
    7760:
        FuUnicodeCodepointCaseConvert := 7761;
        RETURN;
    7761:
        FuUnicodeCodepointCaseConvert := 7760;
        RETURN;
    7762:
        FuUnicodeCodepointCaseConvert := 7763;
        RETURN;
    7763:
        FuUnicodeCodepointCaseConvert := 7762;
        RETURN;
    7764:
        FuUnicodeCodepointCaseConvert := 7765;
        RETURN;
    7765:
        FuUnicodeCodepointCaseConvert := 7764;
        RETURN;
    7766:
        FuUnicodeCodepointCaseConvert := 7767;
        RETURN;
    7767:
        FuUnicodeCodepointCaseConvert := 7766;
        RETURN;
    7768:
        FuUnicodeCodepointCaseConvert := 7769;
        RETURN;
    7769:
        FuUnicodeCodepointCaseConvert := 7768;
        RETURN;
    7770:
        FuUnicodeCodepointCaseConvert := 7771;
        RETURN;
    7771:
        FuUnicodeCodepointCaseConvert := 7770;
        RETURN;
    7772:
        FuUnicodeCodepointCaseConvert := 7773;
        RETURN;
    7773:
        FuUnicodeCodepointCaseConvert := 7772;
        RETURN;
    7774:
        FuUnicodeCodepointCaseConvert := 7775;
        RETURN;
    7775:
        FuUnicodeCodepointCaseConvert := 7774;
        RETURN;
    7776:
        FuUnicodeCodepointCaseConvert := 7777;
        RETURN;
    7777:
        FuUnicodeCodepointCaseConvert := 7776;
        RETURN;
    7778:
        FuUnicodeCodepointCaseConvert := 7779;
        RETURN;
    7779:
        FuUnicodeCodepointCaseConvert := 7778;
        RETURN;
    7780:
        FuUnicodeCodepointCaseConvert := 7781;
        RETURN;
    7781:
        FuUnicodeCodepointCaseConvert := 7780;
        RETURN;
    7782:
        FuUnicodeCodepointCaseConvert := 7783;
        RETURN;
    7783:
        FuUnicodeCodepointCaseConvert := 7782;
        RETURN;
    7784:
        FuUnicodeCodepointCaseConvert := 7785;
        RETURN;
    7785:
        FuUnicodeCodepointCaseConvert := 7784;
        RETURN;
    7786:
        FuUnicodeCodepointCaseConvert := 7787;
        RETURN;
    7787:
        FuUnicodeCodepointCaseConvert := 7786;
        RETURN;
    7788:
        FuUnicodeCodepointCaseConvert := 7789;
        RETURN;
    7789:
        FuUnicodeCodepointCaseConvert := 7788;
        RETURN;
    7790:
        FuUnicodeCodepointCaseConvert := 7791;
        RETURN;
    7791:
        FuUnicodeCodepointCaseConvert := 7790;
        RETURN;
    7792:
        FuUnicodeCodepointCaseConvert := 7793;
        RETURN;
    7793:
        FuUnicodeCodepointCaseConvert := 7792;
        RETURN;
    7794:
        FuUnicodeCodepointCaseConvert := 7795;
        RETURN;
    7795:
        FuUnicodeCodepointCaseConvert := 7794;
        RETURN;
    7796:
        FuUnicodeCodepointCaseConvert := 7797;
        RETURN;
    7797:
        FuUnicodeCodepointCaseConvert := 7796;
        RETURN;
    7798:
        FuUnicodeCodepointCaseConvert := 7799;
        RETURN;
    7799:
        FuUnicodeCodepointCaseConvert := 7798;
        RETURN;
    7800:
        FuUnicodeCodepointCaseConvert := 7801;
        RETURN;
    7801:
        FuUnicodeCodepointCaseConvert := 7800;
        RETURN;
    7802:
        FuUnicodeCodepointCaseConvert := 7803;
        RETURN;
    7803:
        FuUnicodeCodepointCaseConvert := 7802;
        RETURN;
    7804:
        FuUnicodeCodepointCaseConvert := 7805;
        RETURN;
    7805:
        FuUnicodeCodepointCaseConvert := 7804;
        RETURN;
    7806:
        FuUnicodeCodepointCaseConvert := 7807;
        RETURN;
    7807:
        FuUnicodeCodepointCaseConvert := 7806;
        RETURN;
    7808:
        FuUnicodeCodepointCaseConvert := 7809;
        RETURN;
    7809:
        FuUnicodeCodepointCaseConvert := 7808;
        RETURN;
    7810:
        FuUnicodeCodepointCaseConvert := 7811;
        RETURN;
    7811:
        FuUnicodeCodepointCaseConvert := 7810;
        RETURN;
    7812:
        FuUnicodeCodepointCaseConvert := 7813;
        RETURN;
    7813:
        FuUnicodeCodepointCaseConvert := 7812;
        RETURN;
    7814:
        FuUnicodeCodepointCaseConvert := 7815;
        RETURN;
    7815:
        FuUnicodeCodepointCaseConvert := 7814;
        RETURN;
    7816:
        FuUnicodeCodepointCaseConvert := 7817;
        RETURN;
    7817:
        FuUnicodeCodepointCaseConvert := 7816;
        RETURN;
    7818:
        FuUnicodeCodepointCaseConvert := 7819;
        RETURN;
    7819:
        FuUnicodeCodepointCaseConvert := 7818;
        RETURN;
    7820:
        FuUnicodeCodepointCaseConvert := 7821;
        RETURN;
    7821:
        FuUnicodeCodepointCaseConvert := 7820;
        RETURN;
    7822:
        FuUnicodeCodepointCaseConvert := 7823;
        RETURN;
    7823:
        FuUnicodeCodepointCaseConvert := 7822;
        RETURN;
    7824:
        FuUnicodeCodepointCaseConvert := 7825;
        RETURN;
    7825:
        FuUnicodeCodepointCaseConvert := 7824;
        RETURN;
    7826:
        FuUnicodeCodepointCaseConvert := 7827;
        RETURN;
    7827:
        FuUnicodeCodepointCaseConvert := 7826;
        RETURN;
    7828:
        FuUnicodeCodepointCaseConvert := 7829;
        RETURN;
    7829:
        FuUnicodeCodepointCaseConvert := 7828;
        RETURN;
    7835:
        FuUnicodeCodepointCaseConvert := 7776;
        RETURN;
    7838:
        FuUnicodeCodepointCaseConvert := 223;
        RETURN;
    7840:
        FuUnicodeCodepointCaseConvert := 7841;
        RETURN;
    7841:
        FuUnicodeCodepointCaseConvert := 7840;
        RETURN;
    7842:
        FuUnicodeCodepointCaseConvert := 7843;
        RETURN;
    7843:
        FuUnicodeCodepointCaseConvert := 7842;
        RETURN;
    7844:
        FuUnicodeCodepointCaseConvert := 7845;
        RETURN;
    7845:
        FuUnicodeCodepointCaseConvert := 7844;
        RETURN;
    7846:
        FuUnicodeCodepointCaseConvert := 7847;
        RETURN;
    7847:
        FuUnicodeCodepointCaseConvert := 7846;
        RETURN;
    7848:
        FuUnicodeCodepointCaseConvert := 7849;
        RETURN;
    7849:
        FuUnicodeCodepointCaseConvert := 7848;
        RETURN;
    7850:
        FuUnicodeCodepointCaseConvert := 7851;
        RETURN;
    7851:
        FuUnicodeCodepointCaseConvert := 7850;
        RETURN;
    7852:
        FuUnicodeCodepointCaseConvert := 7853;
        RETURN;
    7853:
        FuUnicodeCodepointCaseConvert := 7852;
        RETURN;
    7854:
        FuUnicodeCodepointCaseConvert := 7855;
        RETURN;
    7855:
        FuUnicodeCodepointCaseConvert := 7854;
        RETURN;
    7856:
        FuUnicodeCodepointCaseConvert := 7857;
        RETURN;
    7857:
        FuUnicodeCodepointCaseConvert := 7856;
        RETURN;
    7858:
        FuUnicodeCodepointCaseConvert := 7859;
        RETURN;
    7859:
        FuUnicodeCodepointCaseConvert := 7858;
        RETURN;
    7860:
        FuUnicodeCodepointCaseConvert := 7861;
        RETURN;
    7861:
        FuUnicodeCodepointCaseConvert := 7860;
        RETURN;
    7862:
        FuUnicodeCodepointCaseConvert := 7863;
        RETURN;
    7863:
        FuUnicodeCodepointCaseConvert := 7862;
        RETURN;
    7864:
        FuUnicodeCodepointCaseConvert := 7865;
        RETURN;
    7865:
        FuUnicodeCodepointCaseConvert := 7864;
        RETURN;
    7866:
        FuUnicodeCodepointCaseConvert := 7867;
        RETURN;
    7867:
        FuUnicodeCodepointCaseConvert := 7866;
        RETURN;
    7868:
        FuUnicodeCodepointCaseConvert := 7869;
        RETURN;
    7869:
        FuUnicodeCodepointCaseConvert := 7868;
        RETURN;
    7870:
        FuUnicodeCodepointCaseConvert := 7871;
        RETURN;
    7871:
        FuUnicodeCodepointCaseConvert := 7870;
        RETURN;
    7872:
        FuUnicodeCodepointCaseConvert := 7873;
        RETURN;
    7873:
        FuUnicodeCodepointCaseConvert := 7872;
        RETURN;
    7874:
        FuUnicodeCodepointCaseConvert := 7875;
        RETURN;
    7875:
        FuUnicodeCodepointCaseConvert := 7874;
        RETURN;
    7876:
        FuUnicodeCodepointCaseConvert := 7877;
        RETURN;
    7877:
        FuUnicodeCodepointCaseConvert := 7876;
        RETURN;
    7878:
        FuUnicodeCodepointCaseConvert := 7879;
        RETURN;
    7879:
        FuUnicodeCodepointCaseConvert := 7878;
        RETURN;
    7880:
        FuUnicodeCodepointCaseConvert := 7881;
        RETURN;
    7881:
        FuUnicodeCodepointCaseConvert := 7880;
        RETURN;
    7882:
        FuUnicodeCodepointCaseConvert := 7883;
        RETURN;
    7883:
        FuUnicodeCodepointCaseConvert := 7882;
        RETURN;
    7884:
        FuUnicodeCodepointCaseConvert := 7885;
        RETURN;
    7885:
        FuUnicodeCodepointCaseConvert := 7884;
        RETURN;
    7886:
        FuUnicodeCodepointCaseConvert := 7887;
        RETURN;
    7887:
        FuUnicodeCodepointCaseConvert := 7886;
        RETURN;
    7888:
        FuUnicodeCodepointCaseConvert := 7889;
        RETURN;
    7889:
        FuUnicodeCodepointCaseConvert := 7888;
        RETURN;
    7890:
        FuUnicodeCodepointCaseConvert := 7891;
        RETURN;
    7891:
        FuUnicodeCodepointCaseConvert := 7890;
        RETURN;
    7892:
        FuUnicodeCodepointCaseConvert := 7893;
        RETURN;
    7893:
        FuUnicodeCodepointCaseConvert := 7892;
        RETURN;
    7894:
        FuUnicodeCodepointCaseConvert := 7895;
        RETURN;
    7895:
        FuUnicodeCodepointCaseConvert := 7894;
        RETURN;
    7896:
        FuUnicodeCodepointCaseConvert := 7897;
        RETURN;
    7897:
        FuUnicodeCodepointCaseConvert := 7896;
        RETURN;
    7898:
        FuUnicodeCodepointCaseConvert := 7899;
        RETURN;
    7899:
        FuUnicodeCodepointCaseConvert := 7898;
        RETURN;
    7900:
        FuUnicodeCodepointCaseConvert := 7901;
        RETURN;
    7901:
        FuUnicodeCodepointCaseConvert := 7900;
        RETURN;
    7902:
        FuUnicodeCodepointCaseConvert := 7903;
        RETURN;
    7903:
        FuUnicodeCodepointCaseConvert := 7902;
        RETURN;
    7904:
        FuUnicodeCodepointCaseConvert := 7905;
        RETURN;
    7905:
        FuUnicodeCodepointCaseConvert := 7904;
        RETURN;
    7906:
        FuUnicodeCodepointCaseConvert := 7907;
        RETURN;
    7907:
        FuUnicodeCodepointCaseConvert := 7906;
        RETURN;
    7908:
        FuUnicodeCodepointCaseConvert := 7909;
        RETURN;
    7909:
        FuUnicodeCodepointCaseConvert := 7908;
        RETURN;
    7910:
        FuUnicodeCodepointCaseConvert := 7911;
        RETURN;
    7911:
        FuUnicodeCodepointCaseConvert := 7910;
        RETURN;
    7912:
        FuUnicodeCodepointCaseConvert := 7913;
        RETURN;
    7913:
        FuUnicodeCodepointCaseConvert := 7912;
        RETURN;
    7914:
        FuUnicodeCodepointCaseConvert := 7915;
        RETURN;
    7915:
        FuUnicodeCodepointCaseConvert := 7914;
        RETURN;
    7916:
        FuUnicodeCodepointCaseConvert := 7917;
        RETURN;
    7917:
        FuUnicodeCodepointCaseConvert := 7916;
        RETURN;
    7918:
        FuUnicodeCodepointCaseConvert := 7919;
        RETURN;
    7919:
        FuUnicodeCodepointCaseConvert := 7918;
        RETURN;
    7920:
        FuUnicodeCodepointCaseConvert := 7921;
        RETURN;
    7921:
        FuUnicodeCodepointCaseConvert := 7920;
        RETURN;
    7922:
        FuUnicodeCodepointCaseConvert := 7923;
        RETURN;
    7923:
        FuUnicodeCodepointCaseConvert := 7922;
        RETURN;
    7924:
        FuUnicodeCodepointCaseConvert := 7925;
        RETURN;
    7925:
        FuUnicodeCodepointCaseConvert := 7924;
        RETURN;
    7926:
        FuUnicodeCodepointCaseConvert := 7927;
        RETURN;
    7927:
        FuUnicodeCodepointCaseConvert := 7926;
        RETURN;
    7928:
        FuUnicodeCodepointCaseConvert := 7929;
        RETURN;
    7929:
        FuUnicodeCodepointCaseConvert := 7928;
        RETURN;
    7930:
        FuUnicodeCodepointCaseConvert := 7931;
        RETURN;
    7931:
        FuUnicodeCodepointCaseConvert := 7930;
        RETURN;
    7932:
        FuUnicodeCodepointCaseConvert := 7933;
        RETURN;
    7933:
        FuUnicodeCodepointCaseConvert := 7932;
        RETURN;
    7934:
        FuUnicodeCodepointCaseConvert := 7935;
        RETURN;
    7935:
        FuUnicodeCodepointCaseConvert := 7934;
        RETURN;
    7936:
        FuUnicodeCodepointCaseConvert := 7944;
        RETURN;
    7937:
        FuUnicodeCodepointCaseConvert := 7945;
        RETURN;
    7938:
        FuUnicodeCodepointCaseConvert := 7946;
        RETURN;
    7939:
        FuUnicodeCodepointCaseConvert := 7947;
        RETURN;
    7940:
        FuUnicodeCodepointCaseConvert := 7948;
        RETURN;
    7941:
        FuUnicodeCodepointCaseConvert := 7949;
        RETURN;
    7942:
        FuUnicodeCodepointCaseConvert := 7950;
        RETURN;
    7943:
        FuUnicodeCodepointCaseConvert := 7951;
        RETURN;
    7944:
        FuUnicodeCodepointCaseConvert := 7936;
        RETURN;
    7945:
        FuUnicodeCodepointCaseConvert := 7937;
        RETURN;
    7946:
        FuUnicodeCodepointCaseConvert := 7938;
        RETURN;
    7947:
        FuUnicodeCodepointCaseConvert := 7939;
        RETURN;
    7948:
        FuUnicodeCodepointCaseConvert := 7940;
        RETURN;
    7949:
        FuUnicodeCodepointCaseConvert := 7941;
        RETURN;
    7950:
        FuUnicodeCodepointCaseConvert := 7942;
        RETURN;
    7951:
        FuUnicodeCodepointCaseConvert := 7943;
        RETURN;
    7952:
        FuUnicodeCodepointCaseConvert := 7960;
        RETURN;
    7953:
        FuUnicodeCodepointCaseConvert := 7961;
        RETURN;
    7954:
        FuUnicodeCodepointCaseConvert := 7962;
        RETURN;
    7955:
        FuUnicodeCodepointCaseConvert := 7963;
        RETURN;
    7956:
        FuUnicodeCodepointCaseConvert := 7964;
        RETURN;
    7957:
        FuUnicodeCodepointCaseConvert := 7965;
        RETURN;
    7960:
        FuUnicodeCodepointCaseConvert := 7952;
        RETURN;
    7961:
        FuUnicodeCodepointCaseConvert := 7953;
        RETURN;
    7962:
        FuUnicodeCodepointCaseConvert := 7954;
        RETURN;
    7963:
        FuUnicodeCodepointCaseConvert := 7955;
        RETURN;
    7964:
        FuUnicodeCodepointCaseConvert := 7956;
        RETURN;
    7965:
        FuUnicodeCodepointCaseConvert := 7957;
        RETURN;
    7968:
        FuUnicodeCodepointCaseConvert := 7976;
        RETURN;
    7969:
        FuUnicodeCodepointCaseConvert := 7977;
        RETURN;
    7970:
        FuUnicodeCodepointCaseConvert := 7978;
        RETURN;
    7971:
        FuUnicodeCodepointCaseConvert := 7979;
        RETURN;
    7972:
        FuUnicodeCodepointCaseConvert := 7980;
        RETURN;
    7973:
        FuUnicodeCodepointCaseConvert := 7981;
        RETURN;
    7974:
        FuUnicodeCodepointCaseConvert := 7982;
        RETURN;
    7975:
        FuUnicodeCodepointCaseConvert := 7983;
        RETURN;
    7976:
        FuUnicodeCodepointCaseConvert := 7968;
        RETURN;
    7977:
        FuUnicodeCodepointCaseConvert := 7969;
        RETURN;
    7978:
        FuUnicodeCodepointCaseConvert := 7970;
        RETURN;
    7979:
        FuUnicodeCodepointCaseConvert := 7971;
        RETURN;
    7980:
        FuUnicodeCodepointCaseConvert := 7972;
        RETURN;
    7981:
        FuUnicodeCodepointCaseConvert := 7973;
        RETURN;
    7982:
        FuUnicodeCodepointCaseConvert := 7974;
        RETURN;
    7983:
        FuUnicodeCodepointCaseConvert := 7975;
        RETURN;
    7984:
        FuUnicodeCodepointCaseConvert := 7992;
        RETURN;
    7985:
        FuUnicodeCodepointCaseConvert := 7993;
        RETURN;
    7986:
        FuUnicodeCodepointCaseConvert := 7994;
        RETURN;
    7987:
        FuUnicodeCodepointCaseConvert := 7995;
        RETURN;
    7988:
        FuUnicodeCodepointCaseConvert := 7996;
        RETURN;
    7989:
        FuUnicodeCodepointCaseConvert := 7997;
        RETURN;
    7990:
        FuUnicodeCodepointCaseConvert := 7998;
        RETURN;
    7991:
        FuUnicodeCodepointCaseConvert := 7999;
        RETURN;
    7992:
        FuUnicodeCodepointCaseConvert := 7984;
        RETURN;
    7993:
        FuUnicodeCodepointCaseConvert := 7985;
        RETURN;
    7994:
        FuUnicodeCodepointCaseConvert := 7986;
        RETURN;
    7995:
        FuUnicodeCodepointCaseConvert := 7987;
        RETURN;
    7996:
        FuUnicodeCodepointCaseConvert := 7988;
        RETURN;
    7997:
        FuUnicodeCodepointCaseConvert := 7989;
        RETURN;
    7998:
        FuUnicodeCodepointCaseConvert := 7990;
        RETURN;
    7999:
        FuUnicodeCodepointCaseConvert := 7991;
        RETURN;
    8000:
        FuUnicodeCodepointCaseConvert := 8008;
        RETURN;
    8001:
        FuUnicodeCodepointCaseConvert := 8009;
        RETURN;
    8002:
        FuUnicodeCodepointCaseConvert := 8010;
        RETURN;
    8003:
        FuUnicodeCodepointCaseConvert := 8011;
        RETURN;
    8004:
        FuUnicodeCodepointCaseConvert := 8012;
        RETURN;
    8005:
        FuUnicodeCodepointCaseConvert := 8013;
        RETURN;
    8008:
        FuUnicodeCodepointCaseConvert := 8000;
        RETURN;
    8009:
        FuUnicodeCodepointCaseConvert := 8001;
        RETURN;
    8010:
        FuUnicodeCodepointCaseConvert := 8002;
        RETURN;
    8011:
        FuUnicodeCodepointCaseConvert := 8003;
        RETURN;
    8012:
        FuUnicodeCodepointCaseConvert := 8004;
        RETURN;
    8013:
        FuUnicodeCodepointCaseConvert := 8005;
        RETURN;
    8017:
        FuUnicodeCodepointCaseConvert := 8025;
        RETURN;
    8019:
        FuUnicodeCodepointCaseConvert := 8027;
        RETURN;
    8021:
        FuUnicodeCodepointCaseConvert := 8029;
        RETURN;
    8023:
        FuUnicodeCodepointCaseConvert := 8031;
        RETURN;
    8025:
        FuUnicodeCodepointCaseConvert := 8017;
        RETURN;
    8027:
        FuUnicodeCodepointCaseConvert := 8019;
        RETURN;
    8029:
        FuUnicodeCodepointCaseConvert := 8021;
        RETURN;
    8031:
        FuUnicodeCodepointCaseConvert := 8023;
        RETURN;
    8032:
        FuUnicodeCodepointCaseConvert := 8040;
        RETURN;
    8033:
        FuUnicodeCodepointCaseConvert := 8041;
        RETURN;
    8034:
        FuUnicodeCodepointCaseConvert := 8042;
        RETURN;
    8035:
        FuUnicodeCodepointCaseConvert := 8043;
        RETURN;
    8036:
        FuUnicodeCodepointCaseConvert := 8044;
        RETURN;
    8037:
        FuUnicodeCodepointCaseConvert := 8045;
        RETURN;
    8038:
        FuUnicodeCodepointCaseConvert := 8046;
        RETURN;
    8039:
        FuUnicodeCodepointCaseConvert := 8047;
        RETURN;
    8040:
        FuUnicodeCodepointCaseConvert := 8032;
        RETURN;
    8041:
        FuUnicodeCodepointCaseConvert := 8033;
        RETURN;
    8042:
        FuUnicodeCodepointCaseConvert := 8034;
        RETURN;
    8043:
        FuUnicodeCodepointCaseConvert := 8035;
        RETURN;
    8044:
        FuUnicodeCodepointCaseConvert := 8036;
        RETURN;
    8045:
        FuUnicodeCodepointCaseConvert := 8037;
        RETURN;
    8046:
        FuUnicodeCodepointCaseConvert := 8038;
        RETURN;
    8047:
        FuUnicodeCodepointCaseConvert := 8039;
        RETURN;
    8048:
        FuUnicodeCodepointCaseConvert := 8122;
        RETURN;
    8049:
        FuUnicodeCodepointCaseConvert := 8123;
        RETURN;
    8050:
        FuUnicodeCodepointCaseConvert := 8136;
        RETURN;
    8051:
        FuUnicodeCodepointCaseConvert := 8137;
        RETURN;
    8052:
        FuUnicodeCodepointCaseConvert := 8138;
        RETURN;
    8053:
        FuUnicodeCodepointCaseConvert := 8139;
        RETURN;
    8054:
        FuUnicodeCodepointCaseConvert := 8154;
        RETURN;
    8055:
        FuUnicodeCodepointCaseConvert := 8155;
        RETURN;
    8056:
        FuUnicodeCodepointCaseConvert := 8184;
        RETURN;
    8057:
        FuUnicodeCodepointCaseConvert := 8185;
        RETURN;
    8058:
        FuUnicodeCodepointCaseConvert := 8170;
        RETURN;
    8059:
        FuUnicodeCodepointCaseConvert := 8171;
        RETURN;
    8060:
        FuUnicodeCodepointCaseConvert := 8186;
        RETURN;
    8061:
        FuUnicodeCodepointCaseConvert := 8187;
        RETURN;
    8064:
        FuUnicodeCodepointCaseConvert := 8072;
        RETURN;
    8065:
        FuUnicodeCodepointCaseConvert := 8073;
        RETURN;
    8066:
        FuUnicodeCodepointCaseConvert := 8074;
        RETURN;
    8067:
        FuUnicodeCodepointCaseConvert := 8075;
        RETURN;
    8068:
        FuUnicodeCodepointCaseConvert := 8076;
        RETURN;
    8069:
        FuUnicodeCodepointCaseConvert := 8077;
        RETURN;
    8070:
        FuUnicodeCodepointCaseConvert := 8078;
        RETURN;
    8071:
        FuUnicodeCodepointCaseConvert := 8079;
        RETURN;
    8072:
        FuUnicodeCodepointCaseConvert := 8064;
        RETURN;
    8073:
        FuUnicodeCodepointCaseConvert := 8065;
        RETURN;
    8074:
        FuUnicodeCodepointCaseConvert := 8066;
        RETURN;
    8075:
        FuUnicodeCodepointCaseConvert := 8067;
        RETURN;
    8076:
        FuUnicodeCodepointCaseConvert := 8068;
        RETURN;
    8077:
        FuUnicodeCodepointCaseConvert := 8069;
        RETURN;
    8078:
        FuUnicodeCodepointCaseConvert := 8070;
        RETURN;
    8079:
        FuUnicodeCodepointCaseConvert := 8071;
        RETURN;
    8080:
        FuUnicodeCodepointCaseConvert := 8088;
        RETURN;
    8081:
        FuUnicodeCodepointCaseConvert := 8089;
        RETURN;
    8082:
        FuUnicodeCodepointCaseConvert := 8090;
        RETURN;
    8083:
        FuUnicodeCodepointCaseConvert := 8091;
        RETURN;
    8084:
        FuUnicodeCodepointCaseConvert := 8092;
        RETURN;
    8085:
        FuUnicodeCodepointCaseConvert := 8093;
        RETURN;
    8086:
        FuUnicodeCodepointCaseConvert := 8094;
        RETURN;
    8087:
        FuUnicodeCodepointCaseConvert := 8095;
        RETURN;
    8088:
        FuUnicodeCodepointCaseConvert := 8080;
        RETURN;
    8089:
        FuUnicodeCodepointCaseConvert := 8081;
        RETURN;
    8090:
        FuUnicodeCodepointCaseConvert := 8082;
        RETURN;
    8091:
        FuUnicodeCodepointCaseConvert := 8083;
        RETURN;
    8092:
        FuUnicodeCodepointCaseConvert := 8084;
        RETURN;
    8093:
        FuUnicodeCodepointCaseConvert := 8085;
        RETURN;
    8094:
        FuUnicodeCodepointCaseConvert := 8086;
        RETURN;
    8095:
        FuUnicodeCodepointCaseConvert := 8087;
        RETURN;
    8096:
        FuUnicodeCodepointCaseConvert := 8104;
        RETURN;
    8097:
        FuUnicodeCodepointCaseConvert := 8105;
        RETURN;
    8098:
        FuUnicodeCodepointCaseConvert := 8106;
        RETURN;
    8099:
        FuUnicodeCodepointCaseConvert := 8107;
        RETURN;
    8100:
        FuUnicodeCodepointCaseConvert := 8108;
        RETURN;
    8101:
        FuUnicodeCodepointCaseConvert := 8109;
        RETURN;
    8102:
        FuUnicodeCodepointCaseConvert := 8110;
        RETURN;
    8103:
        FuUnicodeCodepointCaseConvert := 8111;
        RETURN;
    8104:
        FuUnicodeCodepointCaseConvert := 8096;
        RETURN;
    8105:
        FuUnicodeCodepointCaseConvert := 8097;
        RETURN;
    8106:
        FuUnicodeCodepointCaseConvert := 8098;
        RETURN;
    8107:
        FuUnicodeCodepointCaseConvert := 8099;
        RETURN;
    8108:
        FuUnicodeCodepointCaseConvert := 8100;
        RETURN;
    8109:
        FuUnicodeCodepointCaseConvert := 8101;
        RETURN;
    8110:
        FuUnicodeCodepointCaseConvert := 8102;
        RETURN;
    8111:
        FuUnicodeCodepointCaseConvert := 8103;
        RETURN;
    8112:
        FuUnicodeCodepointCaseConvert := 8120;
        RETURN;
    8113:
        FuUnicodeCodepointCaseConvert := 8121;
        RETURN;
    8115:
        FuUnicodeCodepointCaseConvert := 8124;
        RETURN;
    8120:
        FuUnicodeCodepointCaseConvert := 8112;
        RETURN;
    8121:
        FuUnicodeCodepointCaseConvert := 8113;
        RETURN;
    8122:
        FuUnicodeCodepointCaseConvert := 8048;
        RETURN;
    8123:
        FuUnicodeCodepointCaseConvert := 8049;
        RETURN;
    8124:
        FuUnicodeCodepointCaseConvert := 8115;
        RETURN;
    8126:
        FuUnicodeCodepointCaseConvert := 921;
        RETURN;
    8131:
        FuUnicodeCodepointCaseConvert := 8140;
        RETURN;
    8136:
        FuUnicodeCodepointCaseConvert := 8050;
        RETURN;
    8137:
        FuUnicodeCodepointCaseConvert := 8051;
        RETURN;
    8138:
        FuUnicodeCodepointCaseConvert := 8052;
        RETURN;
    8139:
        FuUnicodeCodepointCaseConvert := 8053;
        RETURN;
    8140:
        FuUnicodeCodepointCaseConvert := 8131;
        RETURN;
    8144:
        FuUnicodeCodepointCaseConvert := 8152;
        RETURN;
    8145:
        FuUnicodeCodepointCaseConvert := 8153;
        RETURN;
    8152:
        FuUnicodeCodepointCaseConvert := 8144;
        RETURN;
    8153:
        FuUnicodeCodepointCaseConvert := 8145;
        RETURN;
    8154:
        FuUnicodeCodepointCaseConvert := 8054;
        RETURN;
    8155:
        FuUnicodeCodepointCaseConvert := 8055;
        RETURN;
    8160:
        FuUnicodeCodepointCaseConvert := 8168;
        RETURN;
    8161:
        FuUnicodeCodepointCaseConvert := 8169;
        RETURN;
    8165:
        FuUnicodeCodepointCaseConvert := 8172;
        RETURN;
    8168:
        FuUnicodeCodepointCaseConvert := 8160;
        RETURN;
    8169:
        FuUnicodeCodepointCaseConvert := 8161;
        RETURN;
    8170:
        FuUnicodeCodepointCaseConvert := 8058;
        RETURN;
    8171:
        FuUnicodeCodepointCaseConvert := 8059;
        RETURN;
    8172:
        FuUnicodeCodepointCaseConvert := 8165;
        RETURN;
    8179:
        FuUnicodeCodepointCaseConvert := 8188;
        RETURN;
    8184:
        FuUnicodeCodepointCaseConvert := 8056;
        RETURN;
    8185:
        FuUnicodeCodepointCaseConvert := 8057;
        RETURN;
    8186:
        FuUnicodeCodepointCaseConvert := 8060;
        RETURN;
    8187:
        FuUnicodeCodepointCaseConvert := 8061;
        RETURN;
    8188:
        FuUnicodeCodepointCaseConvert := 8179;
        RETURN;
    8486:
        FuUnicodeCodepointCaseConvert := 969;
        RETURN;
    8490:
        FuUnicodeCodepointCaseConvert := 107;
        RETURN;
    8491:
        FuUnicodeCodepointCaseConvert := 229;
        RETURN;
    8498:
        FuUnicodeCodepointCaseConvert := 8526;
        RETURN;
    8526:
        FuUnicodeCodepointCaseConvert := 8498;
        RETURN;
    8544:
        FuUnicodeCodepointCaseConvert := 8560;
        RETURN;
    8545:
        FuUnicodeCodepointCaseConvert := 8561;
        RETURN;
    8546:
        FuUnicodeCodepointCaseConvert := 8562;
        RETURN;
    8547:
        FuUnicodeCodepointCaseConvert := 8563;
        RETURN;
    8548:
        FuUnicodeCodepointCaseConvert := 8564;
        RETURN;
    8549:
        FuUnicodeCodepointCaseConvert := 8565;
        RETURN;
    8550:
        FuUnicodeCodepointCaseConvert := 8566;
        RETURN;
    8551:
        FuUnicodeCodepointCaseConvert := 8567;
        RETURN;
    8552:
        FuUnicodeCodepointCaseConvert := 8568;
        RETURN;
    8553:
        FuUnicodeCodepointCaseConvert := 8569;
        RETURN;
    8554:
        FuUnicodeCodepointCaseConvert := 8570;
        RETURN;
    8555:
        FuUnicodeCodepointCaseConvert := 8571;
        RETURN;
    8556:
        FuUnicodeCodepointCaseConvert := 8572;
        RETURN;
    8557:
        FuUnicodeCodepointCaseConvert := 8573;
        RETURN;
    8558:
        FuUnicodeCodepointCaseConvert := 8574;
        RETURN;
    8559:
        FuUnicodeCodepointCaseConvert := 8575;
        RETURN;
    8560:
        FuUnicodeCodepointCaseConvert := 8544;
        RETURN;
    8561:
        FuUnicodeCodepointCaseConvert := 8545;
        RETURN;
    8562:
        FuUnicodeCodepointCaseConvert := 8546;
        RETURN;
    8563:
        FuUnicodeCodepointCaseConvert := 8547;
        RETURN;
    8564:
        FuUnicodeCodepointCaseConvert := 8548;
        RETURN;
    8565:
        FuUnicodeCodepointCaseConvert := 8549;
        RETURN;
    8566:
        FuUnicodeCodepointCaseConvert := 8550;
        RETURN;
    8567:
        FuUnicodeCodepointCaseConvert := 8551;
        RETURN;
    8568:
        FuUnicodeCodepointCaseConvert := 8552;
        RETURN;
    8569:
        FuUnicodeCodepointCaseConvert := 8553;
        RETURN;
    8570:
        FuUnicodeCodepointCaseConvert := 8554;
        RETURN;
    8571:
        FuUnicodeCodepointCaseConvert := 8555;
        RETURN;
    8572:
        FuUnicodeCodepointCaseConvert := 8556;
        RETURN;
    8573:
        FuUnicodeCodepointCaseConvert := 8557;
        RETURN;
    8574:
        FuUnicodeCodepointCaseConvert := 8558;
        RETURN;
    8575:
        FuUnicodeCodepointCaseConvert := 8559;
        RETURN;
    8579:
        FuUnicodeCodepointCaseConvert := 8580;
        RETURN;
    8580:
        FuUnicodeCodepointCaseConvert := 8579;
        RETURN;
    9398:
        FuUnicodeCodepointCaseConvert := 9424;
        RETURN;
    9399:
        FuUnicodeCodepointCaseConvert := 9425;
        RETURN;
    9400:
        FuUnicodeCodepointCaseConvert := 9426;
        RETURN;
    9401:
        FuUnicodeCodepointCaseConvert := 9427;
        RETURN;
    9402:
        FuUnicodeCodepointCaseConvert := 9428;
        RETURN;
    9403:
        FuUnicodeCodepointCaseConvert := 9429;
        RETURN;
    9404:
        FuUnicodeCodepointCaseConvert := 9430;
        RETURN;
    9405:
        FuUnicodeCodepointCaseConvert := 9431;
        RETURN;
    9406:
        FuUnicodeCodepointCaseConvert := 9432;
        RETURN;
    9407:
        FuUnicodeCodepointCaseConvert := 9433;
        RETURN;
    9408:
        FuUnicodeCodepointCaseConvert := 9434;
        RETURN;
    9409:
        FuUnicodeCodepointCaseConvert := 9435;
        RETURN;
    9410:
        FuUnicodeCodepointCaseConvert := 9436;
        RETURN;
    9411:
        FuUnicodeCodepointCaseConvert := 9437;
        RETURN;
    9412:
        FuUnicodeCodepointCaseConvert := 9438;
        RETURN;
    9413:
        FuUnicodeCodepointCaseConvert := 9439;
        RETURN;
    9414:
        FuUnicodeCodepointCaseConvert := 9440;
        RETURN;
    9415:
        FuUnicodeCodepointCaseConvert := 9441;
        RETURN;
    9416:
        FuUnicodeCodepointCaseConvert := 9442;
        RETURN;
    9417:
        FuUnicodeCodepointCaseConvert := 9443;
        RETURN;
    9418:
        FuUnicodeCodepointCaseConvert := 9444;
        RETURN;
    9419:
        FuUnicodeCodepointCaseConvert := 9445;
        RETURN;
    9420:
        FuUnicodeCodepointCaseConvert := 9446;
        RETURN;
    9421:
        FuUnicodeCodepointCaseConvert := 9447;
        RETURN;
    9422:
        FuUnicodeCodepointCaseConvert := 9448;
        RETURN;
    9423:
        FuUnicodeCodepointCaseConvert := 9449;
        RETURN;
    9424:
        FuUnicodeCodepointCaseConvert := 9398;
        RETURN;
    9425:
        FuUnicodeCodepointCaseConvert := 9399;
        RETURN;
    9426:
        FuUnicodeCodepointCaseConvert := 9400;
        RETURN;
    9427:
        FuUnicodeCodepointCaseConvert := 9401;
        RETURN;
    9428:
        FuUnicodeCodepointCaseConvert := 9402;
        RETURN;
    9429:
        FuUnicodeCodepointCaseConvert := 9403;
        RETURN;
    9430:
        FuUnicodeCodepointCaseConvert := 9404;
        RETURN;
    9431:
        FuUnicodeCodepointCaseConvert := 9405;
        RETURN;
    9432:
        FuUnicodeCodepointCaseConvert := 9406;
        RETURN;
    9433:
        FuUnicodeCodepointCaseConvert := 9407;
        RETURN;
    9434:
        FuUnicodeCodepointCaseConvert := 9408;
        RETURN;
    9435:
        FuUnicodeCodepointCaseConvert := 9409;
        RETURN;
    9436:
        FuUnicodeCodepointCaseConvert := 9410;
        RETURN;
    9437:
        FuUnicodeCodepointCaseConvert := 9411;
        RETURN;
    9438:
        FuUnicodeCodepointCaseConvert := 9412;
        RETURN;
    9439:
        FuUnicodeCodepointCaseConvert := 9413;
        RETURN;
    9440:
        FuUnicodeCodepointCaseConvert := 9414;
        RETURN;
    9441:
        FuUnicodeCodepointCaseConvert := 9415;
        RETURN;
    9442:
        FuUnicodeCodepointCaseConvert := 9416;
        RETURN;
    9443:
        FuUnicodeCodepointCaseConvert := 9417;
        RETURN;
    9444:
        FuUnicodeCodepointCaseConvert := 9418;
        RETURN;
    9445:
        FuUnicodeCodepointCaseConvert := 9419;
        RETURN;
    9446:
        FuUnicodeCodepointCaseConvert := 9420;
        RETURN;
    9447:
        FuUnicodeCodepointCaseConvert := 9421;
        RETURN;
    9448:
        FuUnicodeCodepointCaseConvert := 9422;
        RETURN;
    9449:
        FuUnicodeCodepointCaseConvert := 9423;
        RETURN;
    11264:
        FuUnicodeCodepointCaseConvert := 11312;
        RETURN;
    11265:
        FuUnicodeCodepointCaseConvert := 11313;
        RETURN;
    11266:
        FuUnicodeCodepointCaseConvert := 11314;
        RETURN;
    11267:
        FuUnicodeCodepointCaseConvert := 11315;
        RETURN;
    11268:
        FuUnicodeCodepointCaseConvert := 11316;
        RETURN;
    11269:
        FuUnicodeCodepointCaseConvert := 11317;
        RETURN;
    11270:
        FuUnicodeCodepointCaseConvert := 11318;
        RETURN;
    11271:
        FuUnicodeCodepointCaseConvert := 11319;
        RETURN;
    11272:
        FuUnicodeCodepointCaseConvert := 11320;
        RETURN;
    11273:
        FuUnicodeCodepointCaseConvert := 11321;
        RETURN;
    11274:
        FuUnicodeCodepointCaseConvert := 11322;
        RETURN;
    11275:
        FuUnicodeCodepointCaseConvert := 11323;
        RETURN;
    11276:
        FuUnicodeCodepointCaseConvert := 11324;
        RETURN;
    11277:
        FuUnicodeCodepointCaseConvert := 11325;
        RETURN;
    11278:
        FuUnicodeCodepointCaseConvert := 11326;
        RETURN;
    11279:
        FuUnicodeCodepointCaseConvert := 11327;
        RETURN;
    11280:
        FuUnicodeCodepointCaseConvert := 11328;
        RETURN;
    11281:
        FuUnicodeCodepointCaseConvert := 11329;
        RETURN;
    11282:
        FuUnicodeCodepointCaseConvert := 11330;
        RETURN;
    11283:
        FuUnicodeCodepointCaseConvert := 11331;
        RETURN;
    11284:
        FuUnicodeCodepointCaseConvert := 11332;
        RETURN;
    11285:
        FuUnicodeCodepointCaseConvert := 11333;
        RETURN;
    11286:
        FuUnicodeCodepointCaseConvert := 11334;
        RETURN;
    11287:
        FuUnicodeCodepointCaseConvert := 11335;
        RETURN;
    11288:
        FuUnicodeCodepointCaseConvert := 11336;
        RETURN;
    11289:
        FuUnicodeCodepointCaseConvert := 11337;
        RETURN;
    11290:
        FuUnicodeCodepointCaseConvert := 11338;
        RETURN;
    11291:
        FuUnicodeCodepointCaseConvert := 11339;
        RETURN;
    11292:
        FuUnicodeCodepointCaseConvert := 11340;
        RETURN;
    11293:
        FuUnicodeCodepointCaseConvert := 11341;
        RETURN;
    11294:
        FuUnicodeCodepointCaseConvert := 11342;
        RETURN;
    11295:
        FuUnicodeCodepointCaseConvert := 11343;
        RETURN;
    11296:
        FuUnicodeCodepointCaseConvert := 11344;
        RETURN;
    11297:
        FuUnicodeCodepointCaseConvert := 11345;
        RETURN;
    11298:
        FuUnicodeCodepointCaseConvert := 11346;
        RETURN;
    11299:
        FuUnicodeCodepointCaseConvert := 11347;
        RETURN;
    11300:
        FuUnicodeCodepointCaseConvert := 11348;
        RETURN;
    11301:
        FuUnicodeCodepointCaseConvert := 11349;
        RETURN;
    11302:
        FuUnicodeCodepointCaseConvert := 11350;
        RETURN;
    11303:
        FuUnicodeCodepointCaseConvert := 11351;
        RETURN;
    11304:
        FuUnicodeCodepointCaseConvert := 11352;
        RETURN;
    11305:
        FuUnicodeCodepointCaseConvert := 11353;
        RETURN;
    11306:
        FuUnicodeCodepointCaseConvert := 11354;
        RETURN;
    11307:
        FuUnicodeCodepointCaseConvert := 11355;
        RETURN;
    11308:
        FuUnicodeCodepointCaseConvert := 11356;
        RETURN;
    11309:
        FuUnicodeCodepointCaseConvert := 11357;
        RETURN;
    11310:
        FuUnicodeCodepointCaseConvert := 11358;
        RETURN;
    11311:
        FuUnicodeCodepointCaseConvert := 11359;
        RETURN;
    11312:
        FuUnicodeCodepointCaseConvert := 11264;
        RETURN;
    11313:
        FuUnicodeCodepointCaseConvert := 11265;
        RETURN;
    11314:
        FuUnicodeCodepointCaseConvert := 11266;
        RETURN;
    11315:
        FuUnicodeCodepointCaseConvert := 11267;
        RETURN;
    11316:
        FuUnicodeCodepointCaseConvert := 11268;
        RETURN;
    11317:
        FuUnicodeCodepointCaseConvert := 11269;
        RETURN;
    11318:
        FuUnicodeCodepointCaseConvert := 11270;
        RETURN;
    11319:
        FuUnicodeCodepointCaseConvert := 11271;
        RETURN;
    11320:
        FuUnicodeCodepointCaseConvert := 11272;
        RETURN;
    11321:
        FuUnicodeCodepointCaseConvert := 11273;
        RETURN;
    11322:
        FuUnicodeCodepointCaseConvert := 11274;
        RETURN;
    11323:
        FuUnicodeCodepointCaseConvert := 11275;
        RETURN;
    11324:
        FuUnicodeCodepointCaseConvert := 11276;
        RETURN;
    11325:
        FuUnicodeCodepointCaseConvert := 11277;
        RETURN;
    11326:
        FuUnicodeCodepointCaseConvert := 11278;
        RETURN;
    11327:
        FuUnicodeCodepointCaseConvert := 11279;
        RETURN;
    11328:
        FuUnicodeCodepointCaseConvert := 11280;
        RETURN;
    11329:
        FuUnicodeCodepointCaseConvert := 11281;
        RETURN;
    11330:
        FuUnicodeCodepointCaseConvert := 11282;
        RETURN;
    11331:
        FuUnicodeCodepointCaseConvert := 11283;
        RETURN;
    11332:
        FuUnicodeCodepointCaseConvert := 11284;
        RETURN;
    11333:
        FuUnicodeCodepointCaseConvert := 11285;
        RETURN;
    11334:
        FuUnicodeCodepointCaseConvert := 11286;
        RETURN;
    11335:
        FuUnicodeCodepointCaseConvert := 11287;
        RETURN;
    11336:
        FuUnicodeCodepointCaseConvert := 11288;
        RETURN;
    11337:
        FuUnicodeCodepointCaseConvert := 11289;
        RETURN;
    11338:
        FuUnicodeCodepointCaseConvert := 11290;
        RETURN;
    11339:
        FuUnicodeCodepointCaseConvert := 11291;
        RETURN;
    11340:
        FuUnicodeCodepointCaseConvert := 11292;
        RETURN;
    11341:
        FuUnicodeCodepointCaseConvert := 11293;
        RETURN;
    11342:
        FuUnicodeCodepointCaseConvert := 11294;
        RETURN;
    11343:
        FuUnicodeCodepointCaseConvert := 11295;
        RETURN;
    11344:
        FuUnicodeCodepointCaseConvert := 11296;
        RETURN;
    11345:
        FuUnicodeCodepointCaseConvert := 11297;
        RETURN;
    11346:
        FuUnicodeCodepointCaseConvert := 11298;
        RETURN;
    11347:
        FuUnicodeCodepointCaseConvert := 11299;
        RETURN;
    11348:
        FuUnicodeCodepointCaseConvert := 11300;
        RETURN;
    11349:
        FuUnicodeCodepointCaseConvert := 11301;
        RETURN;
    11350:
        FuUnicodeCodepointCaseConvert := 11302;
        RETURN;
    11351:
        FuUnicodeCodepointCaseConvert := 11303;
        RETURN;
    11352:
        FuUnicodeCodepointCaseConvert := 11304;
        RETURN;
    11353:
        FuUnicodeCodepointCaseConvert := 11305;
        RETURN;
    11354:
        FuUnicodeCodepointCaseConvert := 11306;
        RETURN;
    11355:
        FuUnicodeCodepointCaseConvert := 11307;
        RETURN;
    11356:
        FuUnicodeCodepointCaseConvert := 11308;
        RETURN;
    11357:
        FuUnicodeCodepointCaseConvert := 11309;
        RETURN;
    11358:
        FuUnicodeCodepointCaseConvert := 11310;
        RETURN;
    11359:
        FuUnicodeCodepointCaseConvert := 11311;
        RETURN;
    11360:
        FuUnicodeCodepointCaseConvert := 11361;
        RETURN;
    11361:
        FuUnicodeCodepointCaseConvert := 11360;
        RETURN;
    11362:
        FuUnicodeCodepointCaseConvert := 619;
        RETURN;
    11363:
        FuUnicodeCodepointCaseConvert := 7549;
        RETURN;
    11364:
        FuUnicodeCodepointCaseConvert := 637;
        RETURN;
    11365:
        FuUnicodeCodepointCaseConvert := 570;
        RETURN;
    11366:
        FuUnicodeCodepointCaseConvert := 574;
        RETURN;
    11367:
        FuUnicodeCodepointCaseConvert := 11368;
        RETURN;
    11368:
        FuUnicodeCodepointCaseConvert := 11367;
        RETURN;
    11369:
        FuUnicodeCodepointCaseConvert := 11370;
        RETURN;
    11370:
        FuUnicodeCodepointCaseConvert := 11369;
        RETURN;
    11371:
        FuUnicodeCodepointCaseConvert := 11372;
        RETURN;
    11372:
        FuUnicodeCodepointCaseConvert := 11371;
        RETURN;
    11373:
        FuUnicodeCodepointCaseConvert := 593;
        RETURN;
    11374:
        FuUnicodeCodepointCaseConvert := 625;
        RETURN;
    11375:
        FuUnicodeCodepointCaseConvert := 592;
        RETURN;
    11376:
        FuUnicodeCodepointCaseConvert := 594;
        RETURN;
    11378:
        FuUnicodeCodepointCaseConvert := 11379;
        RETURN;
    11379:
        FuUnicodeCodepointCaseConvert := 11378;
        RETURN;
    11381:
        FuUnicodeCodepointCaseConvert := 11382;
        RETURN;
    11382:
        FuUnicodeCodepointCaseConvert := 11381;
        RETURN;
    11390:
        FuUnicodeCodepointCaseConvert := 575;
        RETURN;
    11391:
        FuUnicodeCodepointCaseConvert := 576;
        RETURN;
    11392:
        FuUnicodeCodepointCaseConvert := 11393;
        RETURN;
    11393:
        FuUnicodeCodepointCaseConvert := 11392;
        RETURN;
    11394:
        FuUnicodeCodepointCaseConvert := 11395;
        RETURN;
    11395:
        FuUnicodeCodepointCaseConvert := 11394;
        RETURN;
    11396:
        FuUnicodeCodepointCaseConvert := 11397;
        RETURN;
    11397:
        FuUnicodeCodepointCaseConvert := 11396;
        RETURN;
    11398:
        FuUnicodeCodepointCaseConvert := 11399;
        RETURN;
    11399:
        FuUnicodeCodepointCaseConvert := 11398;
        RETURN;
    11400:
        FuUnicodeCodepointCaseConvert := 11401;
        RETURN;
    11401:
        FuUnicodeCodepointCaseConvert := 11400;
        RETURN;
    11402:
        FuUnicodeCodepointCaseConvert := 11403;
        RETURN;
    11403:
        FuUnicodeCodepointCaseConvert := 11402;
        RETURN;
    11404:
        FuUnicodeCodepointCaseConvert := 11405;
        RETURN;
    11405:
        FuUnicodeCodepointCaseConvert := 11404;
        RETURN;
    11406:
        FuUnicodeCodepointCaseConvert := 11407;
        RETURN;
    11407:
        FuUnicodeCodepointCaseConvert := 11406;
        RETURN;
    11408:
        FuUnicodeCodepointCaseConvert := 11409;
        RETURN;
    11409:
        FuUnicodeCodepointCaseConvert := 11408;
        RETURN;
    11410:
        FuUnicodeCodepointCaseConvert := 11411;
        RETURN;
    11411:
        FuUnicodeCodepointCaseConvert := 11410;
        RETURN;
    11412:
        FuUnicodeCodepointCaseConvert := 11413;
        RETURN;
    11413:
        FuUnicodeCodepointCaseConvert := 11412;
        RETURN;
    11414:
        FuUnicodeCodepointCaseConvert := 11415;
        RETURN;
    11415:
        FuUnicodeCodepointCaseConvert := 11414;
        RETURN;
    11416:
        FuUnicodeCodepointCaseConvert := 11417;
        RETURN;
    11417:
        FuUnicodeCodepointCaseConvert := 11416;
        RETURN;
    11418:
        FuUnicodeCodepointCaseConvert := 11419;
        RETURN;
    11419:
        FuUnicodeCodepointCaseConvert := 11418;
        RETURN;
    11420:
        FuUnicodeCodepointCaseConvert := 11421;
        RETURN;
    11421:
        FuUnicodeCodepointCaseConvert := 11420;
        RETURN;
    11422:
        FuUnicodeCodepointCaseConvert := 11423;
        RETURN;
    11423:
        FuUnicodeCodepointCaseConvert := 11422;
        RETURN;
    11424:
        FuUnicodeCodepointCaseConvert := 11425;
        RETURN;
    11425:
        FuUnicodeCodepointCaseConvert := 11424;
        RETURN;
    11426:
        FuUnicodeCodepointCaseConvert := 11427;
        RETURN;
    11427:
        FuUnicodeCodepointCaseConvert := 11426;
        RETURN;
    11428:
        FuUnicodeCodepointCaseConvert := 11429;
        RETURN;
    11429:
        FuUnicodeCodepointCaseConvert := 11428;
        RETURN;
    11430:
        FuUnicodeCodepointCaseConvert := 11431;
        RETURN;
    11431:
        FuUnicodeCodepointCaseConvert := 11430;
        RETURN;
    11432:
        FuUnicodeCodepointCaseConvert := 11433;
        RETURN;
    11433:
        FuUnicodeCodepointCaseConvert := 11432;
        RETURN;
    11434:
        FuUnicodeCodepointCaseConvert := 11435;
        RETURN;
    11435:
        FuUnicodeCodepointCaseConvert := 11434;
        RETURN;
    11436:
        FuUnicodeCodepointCaseConvert := 11437;
        RETURN;
    11437:
        FuUnicodeCodepointCaseConvert := 11436;
        RETURN;
    11438:
        FuUnicodeCodepointCaseConvert := 11439;
        RETURN;
    11439:
        FuUnicodeCodepointCaseConvert := 11438;
        RETURN;
    11440:
        FuUnicodeCodepointCaseConvert := 11441;
        RETURN;
    11441:
        FuUnicodeCodepointCaseConvert := 11440;
        RETURN;
    11442:
        FuUnicodeCodepointCaseConvert := 11443;
        RETURN;
    11443:
        FuUnicodeCodepointCaseConvert := 11442;
        RETURN;
    11444:
        FuUnicodeCodepointCaseConvert := 11445;
        RETURN;
    11445:
        FuUnicodeCodepointCaseConvert := 11444;
        RETURN;
    11446:
        FuUnicodeCodepointCaseConvert := 11447;
        RETURN;
    11447:
        FuUnicodeCodepointCaseConvert := 11446;
        RETURN;
    11448:
        FuUnicodeCodepointCaseConvert := 11449;
        RETURN;
    11449:
        FuUnicodeCodepointCaseConvert := 11448;
        RETURN;
    11450:
        FuUnicodeCodepointCaseConvert := 11451;
        RETURN;
    11451:
        FuUnicodeCodepointCaseConvert := 11450;
        RETURN;
    11452:
        FuUnicodeCodepointCaseConvert := 11453;
        RETURN;
    11453:
        FuUnicodeCodepointCaseConvert := 11452;
        RETURN;
    11454:
        FuUnicodeCodepointCaseConvert := 11455;
        RETURN;
    11455:
        FuUnicodeCodepointCaseConvert := 11454;
        RETURN;
    11456:
        FuUnicodeCodepointCaseConvert := 11457;
        RETURN;
    11457:
        FuUnicodeCodepointCaseConvert := 11456;
        RETURN;
    11458:
        FuUnicodeCodepointCaseConvert := 11459;
        RETURN;
    11459:
        FuUnicodeCodepointCaseConvert := 11458;
        RETURN;
    11460:
        FuUnicodeCodepointCaseConvert := 11461;
        RETURN;
    11461:
        FuUnicodeCodepointCaseConvert := 11460;
        RETURN;
    11462:
        FuUnicodeCodepointCaseConvert := 11463;
        RETURN;
    11463:
        FuUnicodeCodepointCaseConvert := 11462;
        RETURN;
    11464:
        FuUnicodeCodepointCaseConvert := 11465;
        RETURN;
    11465:
        FuUnicodeCodepointCaseConvert := 11464;
        RETURN;
    11466:
        FuUnicodeCodepointCaseConvert := 11467;
        RETURN;
    11467:
        FuUnicodeCodepointCaseConvert := 11466;
        RETURN;
    11468:
        FuUnicodeCodepointCaseConvert := 11469;
        RETURN;
    11469:
        FuUnicodeCodepointCaseConvert := 11468;
        RETURN;
    11470:
        FuUnicodeCodepointCaseConvert := 11471;
        RETURN;
    11471:
        FuUnicodeCodepointCaseConvert := 11470;
        RETURN;
    11472:
        FuUnicodeCodepointCaseConvert := 11473;
        RETURN;
    11473:
        FuUnicodeCodepointCaseConvert := 11472;
        RETURN;
    11474:
        FuUnicodeCodepointCaseConvert := 11475;
        RETURN;
    11475:
        FuUnicodeCodepointCaseConvert := 11474;
        RETURN;
    11476:
        FuUnicodeCodepointCaseConvert := 11477;
        RETURN;
    11477:
        FuUnicodeCodepointCaseConvert := 11476;
        RETURN;
    11478:
        FuUnicodeCodepointCaseConvert := 11479;
        RETURN;
    11479:
        FuUnicodeCodepointCaseConvert := 11478;
        RETURN;
    11480:
        FuUnicodeCodepointCaseConvert := 11481;
        RETURN;
    11481:
        FuUnicodeCodepointCaseConvert := 11480;
        RETURN;
    11482:
        FuUnicodeCodepointCaseConvert := 11483;
        RETURN;
    11483:
        FuUnicodeCodepointCaseConvert := 11482;
        RETURN;
    11484:
        FuUnicodeCodepointCaseConvert := 11485;
        RETURN;
    11485:
        FuUnicodeCodepointCaseConvert := 11484;
        RETURN;
    11486:
        FuUnicodeCodepointCaseConvert := 11487;
        RETURN;
    11487:
        FuUnicodeCodepointCaseConvert := 11486;
        RETURN;
    11488:
        FuUnicodeCodepointCaseConvert := 11489;
        RETURN;
    11489:
        FuUnicodeCodepointCaseConvert := 11488;
        RETURN;
    11490:
        FuUnicodeCodepointCaseConvert := 11491;
        RETURN;
    11491:
        FuUnicodeCodepointCaseConvert := 11490;
        RETURN;
    11499:
        FuUnicodeCodepointCaseConvert := 11500;
        RETURN;
    11500:
        FuUnicodeCodepointCaseConvert := 11499;
        RETURN;
    11501:
        FuUnicodeCodepointCaseConvert := 11502;
        RETURN;
    11502:
        FuUnicodeCodepointCaseConvert := 11501;
        RETURN;
    11506:
        FuUnicodeCodepointCaseConvert := 11507;
        RETURN;
    11507:
        FuUnicodeCodepointCaseConvert := 11506;
        RETURN;
    11520:
        FuUnicodeCodepointCaseConvert := 4256;
        RETURN;
    11521:
        FuUnicodeCodepointCaseConvert := 4257;
        RETURN;
    11522:
        FuUnicodeCodepointCaseConvert := 4258;
        RETURN;
    11523:
        FuUnicodeCodepointCaseConvert := 4259;
        RETURN;
    11524:
        FuUnicodeCodepointCaseConvert := 4260;
        RETURN;
    11525:
        FuUnicodeCodepointCaseConvert := 4261;
        RETURN;
    11526:
        FuUnicodeCodepointCaseConvert := 4262;
        RETURN;
    11527:
        FuUnicodeCodepointCaseConvert := 4263;
        RETURN;
    11528:
        FuUnicodeCodepointCaseConvert := 4264;
        RETURN;
    11529:
        FuUnicodeCodepointCaseConvert := 4265;
        RETURN;
    11530:
        FuUnicodeCodepointCaseConvert := 4266;
        RETURN;
    11531:
        FuUnicodeCodepointCaseConvert := 4267;
        RETURN;
    11532:
        FuUnicodeCodepointCaseConvert := 4268;
        RETURN;
    11533:
        FuUnicodeCodepointCaseConvert := 4269;
        RETURN;
    11534:
        FuUnicodeCodepointCaseConvert := 4270;
        RETURN;
    11535:
        FuUnicodeCodepointCaseConvert := 4271;
        RETURN;
    11536:
        FuUnicodeCodepointCaseConvert := 4272;
        RETURN;
    11537:
        FuUnicodeCodepointCaseConvert := 4273;
        RETURN;
    11538:
        FuUnicodeCodepointCaseConvert := 4274;
        RETURN;
    11539:
        FuUnicodeCodepointCaseConvert := 4275;
        RETURN;
    11540:
        FuUnicodeCodepointCaseConvert := 4276;
        RETURN;
    11541:
        FuUnicodeCodepointCaseConvert := 4277;
        RETURN;
    11542:
        FuUnicodeCodepointCaseConvert := 4278;
        RETURN;
    11543:
        FuUnicodeCodepointCaseConvert := 4279;
        RETURN;
    11544:
        FuUnicodeCodepointCaseConvert := 4280;
        RETURN;
    11545:
        FuUnicodeCodepointCaseConvert := 4281;
        RETURN;
    11546:
        FuUnicodeCodepointCaseConvert := 4282;
        RETURN;
    11547:
        FuUnicodeCodepointCaseConvert := 4283;
        RETURN;
    11548:
        FuUnicodeCodepointCaseConvert := 4284;
        RETURN;
    11549:
        FuUnicodeCodepointCaseConvert := 4285;
        RETURN;
    11550:
        FuUnicodeCodepointCaseConvert := 4286;
        RETURN;
    11551:
        FuUnicodeCodepointCaseConvert := 4287;
        RETURN;
    11552:
        FuUnicodeCodepointCaseConvert := 4288;
        RETURN;
    11553:
        FuUnicodeCodepointCaseConvert := 4289;
        RETURN;
    11554:
        FuUnicodeCodepointCaseConvert := 4290;
        RETURN;
    11555:
        FuUnicodeCodepointCaseConvert := 4291;
        RETURN;
    11556:
        FuUnicodeCodepointCaseConvert := 4292;
        RETURN;
    11557:
        FuUnicodeCodepointCaseConvert := 4293;
        RETURN;
    11559:
        FuUnicodeCodepointCaseConvert := 4295;
        RETURN;
    11565:
        FuUnicodeCodepointCaseConvert := 4301;
        RETURN;
    42560:
        FuUnicodeCodepointCaseConvert := 42561;
        RETURN;
    42561:
        FuUnicodeCodepointCaseConvert := 42560;
        RETURN;
    42562:
        FuUnicodeCodepointCaseConvert := 42563;
        RETURN;
    42563:
        FuUnicodeCodepointCaseConvert := 42562;
        RETURN;
    42564:
        FuUnicodeCodepointCaseConvert := 42565;
        RETURN;
    42565:
        FuUnicodeCodepointCaseConvert := 42564;
        RETURN;
    42566:
        FuUnicodeCodepointCaseConvert := 42567;
        RETURN;
    42567:
        FuUnicodeCodepointCaseConvert := 42566;
        RETURN;
    42568:
        FuUnicodeCodepointCaseConvert := 42569;
        RETURN;
    42569:
        FuUnicodeCodepointCaseConvert := 42568;
        RETURN;
    42570:
        FuUnicodeCodepointCaseConvert := 42571;
        RETURN;
    42571:
        FuUnicodeCodepointCaseConvert := 42570;
        RETURN;
    42572:
        FuUnicodeCodepointCaseConvert := 42573;
        RETURN;
    42573:
        FuUnicodeCodepointCaseConvert := 42572;
        RETURN;
    42574:
        FuUnicodeCodepointCaseConvert := 42575;
        RETURN;
    42575:
        FuUnicodeCodepointCaseConvert := 42574;
        RETURN;
    42576:
        FuUnicodeCodepointCaseConvert := 42577;
        RETURN;
    42577:
        FuUnicodeCodepointCaseConvert := 42576;
        RETURN;
    42578:
        FuUnicodeCodepointCaseConvert := 42579;
        RETURN;
    42579:
        FuUnicodeCodepointCaseConvert := 42578;
        RETURN;
    42580:
        FuUnicodeCodepointCaseConvert := 42581;
        RETURN;
    42581:
        FuUnicodeCodepointCaseConvert := 42580;
        RETURN;
    42582:
        FuUnicodeCodepointCaseConvert := 42583;
        RETURN;
    42583:
        FuUnicodeCodepointCaseConvert := 42582;
        RETURN;
    42584:
        FuUnicodeCodepointCaseConvert := 42585;
        RETURN;
    42585:
        FuUnicodeCodepointCaseConvert := 42584;
        RETURN;
    42586:
        FuUnicodeCodepointCaseConvert := 42587;
        RETURN;
    42587:
        FuUnicodeCodepointCaseConvert := 42586;
        RETURN;
    42588:
        FuUnicodeCodepointCaseConvert := 42589;
        RETURN;
    42589:
        FuUnicodeCodepointCaseConvert := 42588;
        RETURN;
    42590:
        FuUnicodeCodepointCaseConvert := 42591;
        RETURN;
    42591:
        FuUnicodeCodepointCaseConvert := 42590;
        RETURN;
    42592:
        FuUnicodeCodepointCaseConvert := 42593;
        RETURN;
    42593:
        FuUnicodeCodepointCaseConvert := 42592;
        RETURN;
    42594:
        FuUnicodeCodepointCaseConvert := 42595;
        RETURN;
    42595:
        FuUnicodeCodepointCaseConvert := 42594;
        RETURN;
    42596:
        FuUnicodeCodepointCaseConvert := 42597;
        RETURN;
    42597:
        FuUnicodeCodepointCaseConvert := 42596;
        RETURN;
    42598:
        FuUnicodeCodepointCaseConvert := 42599;
        RETURN;
    42599:
        FuUnicodeCodepointCaseConvert := 42598;
        RETURN;
    42600:
        FuUnicodeCodepointCaseConvert := 42601;
        RETURN;
    42601:
        FuUnicodeCodepointCaseConvert := 42600;
        RETURN;
    42602:
        FuUnicodeCodepointCaseConvert := 42603;
        RETURN;
    42603:
        FuUnicodeCodepointCaseConvert := 42602;
        RETURN;
    42604:
        FuUnicodeCodepointCaseConvert := 42605;
        RETURN;
    42605:
        FuUnicodeCodepointCaseConvert := 42604;
        RETURN;
    42624:
        FuUnicodeCodepointCaseConvert := 42625;
        RETURN;
    42625:
        FuUnicodeCodepointCaseConvert := 42624;
        RETURN;
    42626:
        FuUnicodeCodepointCaseConvert := 42627;
        RETURN;
    42627:
        FuUnicodeCodepointCaseConvert := 42626;
        RETURN;
    42628:
        FuUnicodeCodepointCaseConvert := 42629;
        RETURN;
    42629:
        FuUnicodeCodepointCaseConvert := 42628;
        RETURN;
    42630:
        FuUnicodeCodepointCaseConvert := 42631;
        RETURN;
    42631:
        FuUnicodeCodepointCaseConvert := 42630;
        RETURN;
    42632:
        FuUnicodeCodepointCaseConvert := 42633;
        RETURN;
    42633:
        FuUnicodeCodepointCaseConvert := 42632;
        RETURN;
    42634:
        FuUnicodeCodepointCaseConvert := 42635;
        RETURN;
    42635:
        FuUnicodeCodepointCaseConvert := 42634;
        RETURN;
    42636:
        FuUnicodeCodepointCaseConvert := 42637;
        RETURN;
    42637:
        FuUnicodeCodepointCaseConvert := 42636;
        RETURN;
    42638:
        FuUnicodeCodepointCaseConvert := 42639;
        RETURN;
    42639:
        FuUnicodeCodepointCaseConvert := 42638;
        RETURN;
    42640:
        FuUnicodeCodepointCaseConvert := 42641;
        RETURN;
    42641:
        FuUnicodeCodepointCaseConvert := 42640;
        RETURN;
    42642:
        FuUnicodeCodepointCaseConvert := 42643;
        RETURN;
    42643:
        FuUnicodeCodepointCaseConvert := 42642;
        RETURN;
    42644:
        FuUnicodeCodepointCaseConvert := 42645;
        RETURN;
    42645:
        FuUnicodeCodepointCaseConvert := 42644;
        RETURN;
    42646:
        FuUnicodeCodepointCaseConvert := 42647;
        RETURN;
    42647:
        FuUnicodeCodepointCaseConvert := 42646;
        RETURN;
    42648:
        FuUnicodeCodepointCaseConvert := 42649;
        RETURN;
    42649:
        FuUnicodeCodepointCaseConvert := 42648;
        RETURN;
    42650:
        FuUnicodeCodepointCaseConvert := 42651;
        RETURN;
    42651:
        FuUnicodeCodepointCaseConvert := 42650;
        RETURN;
    42786:
        FuUnicodeCodepointCaseConvert := 42787;
        RETURN;
    42787:
        FuUnicodeCodepointCaseConvert := 42786;
        RETURN;
    42788:
        FuUnicodeCodepointCaseConvert := 42789;
        RETURN;
    42789:
        FuUnicodeCodepointCaseConvert := 42788;
        RETURN;
    42790:
        FuUnicodeCodepointCaseConvert := 42791;
        RETURN;
    42791:
        FuUnicodeCodepointCaseConvert := 42790;
        RETURN;
    42792:
        FuUnicodeCodepointCaseConvert := 42793;
        RETURN;
    42793:
        FuUnicodeCodepointCaseConvert := 42792;
        RETURN;
    42794:
        FuUnicodeCodepointCaseConvert := 42795;
        RETURN;
    42795:
        FuUnicodeCodepointCaseConvert := 42794;
        RETURN;
    42796:
        FuUnicodeCodepointCaseConvert := 42797;
        RETURN;
    42797:
        FuUnicodeCodepointCaseConvert := 42796;
        RETURN;
    42798:
        FuUnicodeCodepointCaseConvert := 42799;
        RETURN;
    42799:
        FuUnicodeCodepointCaseConvert := 42798;
        RETURN;
    42802:
        FuUnicodeCodepointCaseConvert := 42803;
        RETURN;
    42803:
        FuUnicodeCodepointCaseConvert := 42802;
        RETURN;
    42804:
        FuUnicodeCodepointCaseConvert := 42805;
        RETURN;
    42805:
        FuUnicodeCodepointCaseConvert := 42804;
        RETURN;
    42806:
        FuUnicodeCodepointCaseConvert := 42807;
        RETURN;
    42807:
        FuUnicodeCodepointCaseConvert := 42806;
        RETURN;
    42808:
        FuUnicodeCodepointCaseConvert := 42809;
        RETURN;
    42809:
        FuUnicodeCodepointCaseConvert := 42808;
        RETURN;
    42810:
        FuUnicodeCodepointCaseConvert := 42811;
        RETURN;
    42811:
        FuUnicodeCodepointCaseConvert := 42810;
        RETURN;
    42812:
        FuUnicodeCodepointCaseConvert := 42813;
        RETURN;
    42813:
        FuUnicodeCodepointCaseConvert := 42812;
        RETURN;
    42814:
        FuUnicodeCodepointCaseConvert := 42815;
        RETURN;
    42815:
        FuUnicodeCodepointCaseConvert := 42814;
        RETURN;
    42816:
        FuUnicodeCodepointCaseConvert := 42817;
        RETURN;
    42817:
        FuUnicodeCodepointCaseConvert := 42816;
        RETURN;
    42818:
        FuUnicodeCodepointCaseConvert := 42819;
        RETURN;
    42819:
        FuUnicodeCodepointCaseConvert := 42818;
        RETURN;
    42820:
        FuUnicodeCodepointCaseConvert := 42821;
        RETURN;
    42821:
        FuUnicodeCodepointCaseConvert := 42820;
        RETURN;
    42822:
        FuUnicodeCodepointCaseConvert := 42823;
        RETURN;
    42823:
        FuUnicodeCodepointCaseConvert := 42822;
        RETURN;
    42824:
        FuUnicodeCodepointCaseConvert := 42825;
        RETURN;
    42825:
        FuUnicodeCodepointCaseConvert := 42824;
        RETURN;
    42826:
        FuUnicodeCodepointCaseConvert := 42827;
        RETURN;
    42827:
        FuUnicodeCodepointCaseConvert := 42826;
        RETURN;
    42828:
        FuUnicodeCodepointCaseConvert := 42829;
        RETURN;
    42829:
        FuUnicodeCodepointCaseConvert := 42828;
        RETURN;
    42830:
        FuUnicodeCodepointCaseConvert := 42831;
        RETURN;
    42831:
        FuUnicodeCodepointCaseConvert := 42830;
        RETURN;
    42832:
        FuUnicodeCodepointCaseConvert := 42833;
        RETURN;
    42833:
        FuUnicodeCodepointCaseConvert := 42832;
        RETURN;
    42834:
        FuUnicodeCodepointCaseConvert := 42835;
        RETURN;
    42835:
        FuUnicodeCodepointCaseConvert := 42834;
        RETURN;
    42836:
        FuUnicodeCodepointCaseConvert := 42837;
        RETURN;
    42837:
        FuUnicodeCodepointCaseConvert := 42836;
        RETURN;
    42838:
        FuUnicodeCodepointCaseConvert := 42839;
        RETURN;
    42839:
        FuUnicodeCodepointCaseConvert := 42838;
        RETURN;
    42840:
        FuUnicodeCodepointCaseConvert := 42841;
        RETURN;
    42841:
        FuUnicodeCodepointCaseConvert := 42840;
        RETURN;
    42842:
        FuUnicodeCodepointCaseConvert := 42843;
        RETURN;
    42843:
        FuUnicodeCodepointCaseConvert := 42842;
        RETURN;
    42844:
        FuUnicodeCodepointCaseConvert := 42845;
        RETURN;
    42845:
        FuUnicodeCodepointCaseConvert := 42844;
        RETURN;
    42846:
        FuUnicodeCodepointCaseConvert := 42847;
        RETURN;
    42847:
        FuUnicodeCodepointCaseConvert := 42846;
        RETURN;
    42848:
        FuUnicodeCodepointCaseConvert := 42849;
        RETURN;
    42849:
        FuUnicodeCodepointCaseConvert := 42848;
        RETURN;
    42850:
        FuUnicodeCodepointCaseConvert := 42851;
        RETURN;
    42851:
        FuUnicodeCodepointCaseConvert := 42850;
        RETURN;
    42852:
        FuUnicodeCodepointCaseConvert := 42853;
        RETURN;
    42853:
        FuUnicodeCodepointCaseConvert := 42852;
        RETURN;
    42854:
        FuUnicodeCodepointCaseConvert := 42855;
        RETURN;
    42855:
        FuUnicodeCodepointCaseConvert := 42854;
        RETURN;
    42856:
        FuUnicodeCodepointCaseConvert := 42857;
        RETURN;
    42857:
        FuUnicodeCodepointCaseConvert := 42856;
        RETURN;
    42858:
        FuUnicodeCodepointCaseConvert := 42859;
        RETURN;
    42859:
        FuUnicodeCodepointCaseConvert := 42858;
        RETURN;
    42860:
        FuUnicodeCodepointCaseConvert := 42861;
        RETURN;
    42861:
        FuUnicodeCodepointCaseConvert := 42860;
        RETURN;
    42862:
        FuUnicodeCodepointCaseConvert := 42863;
        RETURN;
    42863:
        FuUnicodeCodepointCaseConvert := 42862;
        RETURN;
    42873:
        FuUnicodeCodepointCaseConvert := 42874;
        RETURN;
    42874:
        FuUnicodeCodepointCaseConvert := 42873;
        RETURN;
    42875:
        FuUnicodeCodepointCaseConvert := 42876;
        RETURN;
    42876:
        FuUnicodeCodepointCaseConvert := 42875;
        RETURN;
    42877:
        FuUnicodeCodepointCaseConvert := 7545;
        RETURN;
    42878:
        FuUnicodeCodepointCaseConvert := 42879;
        RETURN;
    42879:
        FuUnicodeCodepointCaseConvert := 42878;
        RETURN;
    42880:
        FuUnicodeCodepointCaseConvert := 42881;
        RETURN;
    42881:
        FuUnicodeCodepointCaseConvert := 42880;
        RETURN;
    42882:
        FuUnicodeCodepointCaseConvert := 42883;
        RETURN;
    42883:
        FuUnicodeCodepointCaseConvert := 42882;
        RETURN;
    42884:
        FuUnicodeCodepointCaseConvert := 42885;
        RETURN;
    42885:
        FuUnicodeCodepointCaseConvert := 42884;
        RETURN;
    42886:
        FuUnicodeCodepointCaseConvert := 42887;
        RETURN;
    42887:
        FuUnicodeCodepointCaseConvert := 42886;
        RETURN;
    42891:
        FuUnicodeCodepointCaseConvert := 42892;
        RETURN;
    42892:
        FuUnicodeCodepointCaseConvert := 42891;
        RETURN;
    42893:
        FuUnicodeCodepointCaseConvert := 613;
        RETURN;
    42896:
        FuUnicodeCodepointCaseConvert := 42897;
        RETURN;
    42897:
        FuUnicodeCodepointCaseConvert := 42896;
        RETURN;
    42898:
        FuUnicodeCodepointCaseConvert := 42899;
        RETURN;
    42899:
        FuUnicodeCodepointCaseConvert := 42898;
        RETURN;
    42900:
        FuUnicodeCodepointCaseConvert := 42948;
        RETURN;
    42902:
        FuUnicodeCodepointCaseConvert := 42903;
        RETURN;
    42903:
        FuUnicodeCodepointCaseConvert := 42902;
        RETURN;
    42904:
        FuUnicodeCodepointCaseConvert := 42905;
        RETURN;
    42905:
        FuUnicodeCodepointCaseConvert := 42904;
        RETURN;
    42906:
        FuUnicodeCodepointCaseConvert := 42907;
        RETURN;
    42907:
        FuUnicodeCodepointCaseConvert := 42906;
        RETURN;
    42908:
        FuUnicodeCodepointCaseConvert := 42909;
        RETURN;
    42909:
        FuUnicodeCodepointCaseConvert := 42908;
        RETURN;
    42910:
        FuUnicodeCodepointCaseConvert := 42911;
        RETURN;
    42911:
        FuUnicodeCodepointCaseConvert := 42910;
        RETURN;
    42912:
        FuUnicodeCodepointCaseConvert := 42913;
        RETURN;
    42913:
        FuUnicodeCodepointCaseConvert := 42912;
        RETURN;
    42914:
        FuUnicodeCodepointCaseConvert := 42915;
        RETURN;
    42915:
        FuUnicodeCodepointCaseConvert := 42914;
        RETURN;
    42916:
        FuUnicodeCodepointCaseConvert := 42917;
        RETURN;
    42917:
        FuUnicodeCodepointCaseConvert := 42916;
        RETURN;
    42918:
        FuUnicodeCodepointCaseConvert := 42919;
        RETURN;
    42919:
        FuUnicodeCodepointCaseConvert := 42918;
        RETURN;
    42920:
        FuUnicodeCodepointCaseConvert := 42921;
        RETURN;
    42921:
        FuUnicodeCodepointCaseConvert := 42920;
        RETURN;
    42922:
        FuUnicodeCodepointCaseConvert := 614;
        RETURN;
    42923:
        FuUnicodeCodepointCaseConvert := 604;
        RETURN;
    42924:
        FuUnicodeCodepointCaseConvert := 609;
        RETURN;
    42925:
        FuUnicodeCodepointCaseConvert := 620;
        RETURN;
    42926:
        FuUnicodeCodepointCaseConvert := 618;
        RETURN;
    42928:
        FuUnicodeCodepointCaseConvert := 670;
        RETURN;
    42929:
        FuUnicodeCodepointCaseConvert := 647;
        RETURN;
    42930:
        FuUnicodeCodepointCaseConvert := 669;
        RETURN;
    42931:
        FuUnicodeCodepointCaseConvert := 43859;
        RETURN;
    42932:
        FuUnicodeCodepointCaseConvert := 42933;
        RETURN;
    42933:
        FuUnicodeCodepointCaseConvert := 42932;
        RETURN;
    42934:
        FuUnicodeCodepointCaseConvert := 42935;
        RETURN;
    42935:
        FuUnicodeCodepointCaseConvert := 42934;
        RETURN;
    42936:
        FuUnicodeCodepointCaseConvert := 42937;
        RETURN;
    42937:
        FuUnicodeCodepointCaseConvert := 42936;
        RETURN;
    42938:
        FuUnicodeCodepointCaseConvert := 42939;
        RETURN;
    42939:
        FuUnicodeCodepointCaseConvert := 42938;
        RETURN;
    42940:
        FuUnicodeCodepointCaseConvert := 42941;
        RETURN;
    42941:
        FuUnicodeCodepointCaseConvert := 42940;
        RETURN;
    42942:
        FuUnicodeCodepointCaseConvert := 42943;
        RETURN;
    42943:
        FuUnicodeCodepointCaseConvert := 42942;
        RETURN;
    42944:
        FuUnicodeCodepointCaseConvert := 42945;
        RETURN;
    42945:
        FuUnicodeCodepointCaseConvert := 42944;
        RETURN;
    42946:
        FuUnicodeCodepointCaseConvert := 42947;
        RETURN;
    42947:
        FuUnicodeCodepointCaseConvert := 42946;
        RETURN;
    42948:
        FuUnicodeCodepointCaseConvert := 42900;
        RETURN;
    42949:
        FuUnicodeCodepointCaseConvert := 642;
        RETURN;
    42950:
        FuUnicodeCodepointCaseConvert := 7566;
        RETURN;
    42951:
        FuUnicodeCodepointCaseConvert := 42952;
        RETURN;
    42952:
        FuUnicodeCodepointCaseConvert := 42951;
        RETURN;
    42953:
        FuUnicodeCodepointCaseConvert := 42954;
        RETURN;
    42954:
        FuUnicodeCodepointCaseConvert := 42953;
        RETURN;
    42960:
        FuUnicodeCodepointCaseConvert := 42961;
        RETURN;
    42961:
        FuUnicodeCodepointCaseConvert := 42960;
        RETURN;
    42966:
        FuUnicodeCodepointCaseConvert := 42967;
        RETURN;
    42967:
        FuUnicodeCodepointCaseConvert := 42966;
        RETURN;
    42968:
        FuUnicodeCodepointCaseConvert := 42969;
        RETURN;
    42969:
        FuUnicodeCodepointCaseConvert := 42968;
        RETURN;
    42997:
        FuUnicodeCodepointCaseConvert := 42998;
        RETURN;
    42998:
        FuUnicodeCodepointCaseConvert := 42997;
        RETURN;
    43859:
        FuUnicodeCodepointCaseConvert := 42931;
        RETURN;
    43888:
        FuUnicodeCodepointCaseConvert := 5024;
        RETURN;
    43889:
        FuUnicodeCodepointCaseConvert := 5025;
        RETURN;
    43890:
        FuUnicodeCodepointCaseConvert := 5026;
        RETURN;
    43891:
        FuUnicodeCodepointCaseConvert := 5027;
        RETURN;
    43892:
        FuUnicodeCodepointCaseConvert := 5028;
        RETURN;
    43893:
        FuUnicodeCodepointCaseConvert := 5029;
        RETURN;
    43894:
        FuUnicodeCodepointCaseConvert := 5030;
        RETURN;
    43895:
        FuUnicodeCodepointCaseConvert := 5031;
        RETURN;
    43896:
        FuUnicodeCodepointCaseConvert := 5032;
        RETURN;
    43897:
        FuUnicodeCodepointCaseConvert := 5033;
        RETURN;
    43898:
        FuUnicodeCodepointCaseConvert := 5034;
        RETURN;
    43899:
        FuUnicodeCodepointCaseConvert := 5035;
        RETURN;
    43900:
        FuUnicodeCodepointCaseConvert := 5036;
        RETURN;
    43901:
        FuUnicodeCodepointCaseConvert := 5037;
        RETURN;
    43902:
        FuUnicodeCodepointCaseConvert := 5038;
        RETURN;
    43903:
        FuUnicodeCodepointCaseConvert := 5039;
        RETURN;
    43904:
        FuUnicodeCodepointCaseConvert := 5040;
        RETURN;
    43905:
        FuUnicodeCodepointCaseConvert := 5041;
        RETURN;
    43906:
        FuUnicodeCodepointCaseConvert := 5042;
        RETURN;
    43907:
        FuUnicodeCodepointCaseConvert := 5043;
        RETURN;
    43908:
        FuUnicodeCodepointCaseConvert := 5044;
        RETURN;
    43909:
        FuUnicodeCodepointCaseConvert := 5045;
        RETURN;
    43910:
        FuUnicodeCodepointCaseConvert := 5046;
        RETURN;
    43911:
        FuUnicodeCodepointCaseConvert := 5047;
        RETURN;
    43912:
        FuUnicodeCodepointCaseConvert := 5048;
        RETURN;
    43913:
        FuUnicodeCodepointCaseConvert := 5049;
        RETURN;
    43914:
        FuUnicodeCodepointCaseConvert := 5050;
        RETURN;
    43915:
        FuUnicodeCodepointCaseConvert := 5051;
        RETURN;
    43916:
        FuUnicodeCodepointCaseConvert := 5052;
        RETURN;
    43917:
        FuUnicodeCodepointCaseConvert := 5053;
        RETURN;
    43918:
        FuUnicodeCodepointCaseConvert := 5054;
        RETURN;
    43919:
        FuUnicodeCodepointCaseConvert := 5055;
        RETURN;
    43920:
        FuUnicodeCodepointCaseConvert := 5056;
        RETURN;
    43921:
        FuUnicodeCodepointCaseConvert := 5057;
        RETURN;
    43922:
        FuUnicodeCodepointCaseConvert := 5058;
        RETURN;
    43923:
        FuUnicodeCodepointCaseConvert := 5059;
        RETURN;
    43924:
        FuUnicodeCodepointCaseConvert := 5060;
        RETURN;
    43925:
        FuUnicodeCodepointCaseConvert := 5061;
        RETURN;
    43926:
        FuUnicodeCodepointCaseConvert := 5062;
        RETURN;
    43927:
        FuUnicodeCodepointCaseConvert := 5063;
        RETURN;
    43928:
        FuUnicodeCodepointCaseConvert := 5064;
        RETURN;
    43929:
        FuUnicodeCodepointCaseConvert := 5065;
        RETURN;
    43930:
        FuUnicodeCodepointCaseConvert := 5066;
        RETURN;
    43931:
        FuUnicodeCodepointCaseConvert := 5067;
        RETURN;
    43932:
        FuUnicodeCodepointCaseConvert := 5068;
        RETURN;
    43933:
        FuUnicodeCodepointCaseConvert := 5069;
        RETURN;
    43934:
        FuUnicodeCodepointCaseConvert := 5070;
        RETURN;
    43935:
        FuUnicodeCodepointCaseConvert := 5071;
        RETURN;
    43936:
        FuUnicodeCodepointCaseConvert := 5072;
        RETURN;
    43937:
        FuUnicodeCodepointCaseConvert := 5073;
        RETURN;
    43938:
        FuUnicodeCodepointCaseConvert := 5074;
        RETURN;
    43939:
        FuUnicodeCodepointCaseConvert := 5075;
        RETURN;
    43940:
        FuUnicodeCodepointCaseConvert := 5076;
        RETURN;
    43941:
        FuUnicodeCodepointCaseConvert := 5077;
        RETURN;
    43942:
        FuUnicodeCodepointCaseConvert := 5078;
        RETURN;
    43943:
        FuUnicodeCodepointCaseConvert := 5079;
        RETURN;
    43944:
        FuUnicodeCodepointCaseConvert := 5080;
        RETURN;
    43945:
        FuUnicodeCodepointCaseConvert := 5081;
        RETURN;
    43946:
        FuUnicodeCodepointCaseConvert := 5082;
        RETURN;
    43947:
        FuUnicodeCodepointCaseConvert := 5083;
        RETURN;
    43948:
        FuUnicodeCodepointCaseConvert := 5084;
        RETURN;
    43949:
        FuUnicodeCodepointCaseConvert := 5085;
        RETURN;
    43950:
        FuUnicodeCodepointCaseConvert := 5086;
        RETURN;
    43951:
        FuUnicodeCodepointCaseConvert := 5087;
        RETURN;
    43952:
        FuUnicodeCodepointCaseConvert := 5088;
        RETURN;
    43953:
        FuUnicodeCodepointCaseConvert := 5089;
        RETURN;
    43954:
        FuUnicodeCodepointCaseConvert := 5090;
        RETURN;
    43955:
        FuUnicodeCodepointCaseConvert := 5091;
        RETURN;
    43956:
        FuUnicodeCodepointCaseConvert := 5092;
        RETURN;
    43957:
        FuUnicodeCodepointCaseConvert := 5093;
        RETURN;
    43958:
        FuUnicodeCodepointCaseConvert := 5094;
        RETURN;
    43959:
        FuUnicodeCodepointCaseConvert := 5095;
        RETURN;
    43960:
        FuUnicodeCodepointCaseConvert := 5096;
        RETURN;
    43961:
        FuUnicodeCodepointCaseConvert := 5097;
        RETURN;
    43962:
        FuUnicodeCodepointCaseConvert := 5098;
        RETURN;
    43963:
        FuUnicodeCodepointCaseConvert := 5099;
        RETURN;
    43964:
        FuUnicodeCodepointCaseConvert := 5100;
        RETURN;
    43965:
        FuUnicodeCodepointCaseConvert := 5101;
        RETURN;
    43966:
        FuUnicodeCodepointCaseConvert := 5102;
        RETURN;
    43967:
        FuUnicodeCodepointCaseConvert := 5103;
        RETURN;
    65313:
        FuUnicodeCodepointCaseConvert := 65345;
        RETURN;
    65314:
        FuUnicodeCodepointCaseConvert := 65346;
        RETURN;
    65315:
        FuUnicodeCodepointCaseConvert := 65347;
        RETURN;
    65316:
        FuUnicodeCodepointCaseConvert := 65348;
        RETURN;
    65317:
        FuUnicodeCodepointCaseConvert := 65349;
        RETURN;
    65318:
        FuUnicodeCodepointCaseConvert := 65350;
        RETURN;
    65319:
        FuUnicodeCodepointCaseConvert := 65351;
        RETURN;
    65320:
        FuUnicodeCodepointCaseConvert := 65352;
        RETURN;
    65321:
        FuUnicodeCodepointCaseConvert := 65353;
        RETURN;
    65322:
        FuUnicodeCodepointCaseConvert := 65354;
        RETURN;
    65323:
        FuUnicodeCodepointCaseConvert := 65355;
        RETURN;
    65324:
        FuUnicodeCodepointCaseConvert := 65356;
        RETURN;
    65325:
        FuUnicodeCodepointCaseConvert := 65357;
        RETURN;
    65326:
        FuUnicodeCodepointCaseConvert := 65358;
        RETURN;
    65327:
        FuUnicodeCodepointCaseConvert := 65359;
        RETURN;
    65328:
        FuUnicodeCodepointCaseConvert := 65360;
        RETURN;
    65329:
        FuUnicodeCodepointCaseConvert := 65361;
        RETURN;
    65330:
        FuUnicodeCodepointCaseConvert := 65362;
        RETURN;
    65331:
        FuUnicodeCodepointCaseConvert := 65363;
        RETURN;
    65332:
        FuUnicodeCodepointCaseConvert := 65364;
        RETURN;
    65333:
        FuUnicodeCodepointCaseConvert := 65365;
        RETURN;
    65334:
        FuUnicodeCodepointCaseConvert := 65366;
        RETURN;
    65335:
        FuUnicodeCodepointCaseConvert := 65367;
        RETURN;
    65336:
        FuUnicodeCodepointCaseConvert := 65368;
        RETURN;
    65337:
        FuUnicodeCodepointCaseConvert := 65369;
        RETURN;
    65338:
        FuUnicodeCodepointCaseConvert := 65370;
        RETURN;
    65345:
        FuUnicodeCodepointCaseConvert := 65313;
        RETURN;
    65346:
        FuUnicodeCodepointCaseConvert := 65314;
        RETURN;
    65347:
        FuUnicodeCodepointCaseConvert := 65315;
        RETURN;
    65348:
        FuUnicodeCodepointCaseConvert := 65316;
        RETURN;
    65349:
        FuUnicodeCodepointCaseConvert := 65317;
        RETURN;
    65350:
        FuUnicodeCodepointCaseConvert := 65318;
        RETURN;
    65351:
        FuUnicodeCodepointCaseConvert := 65319;
        RETURN;
    65352:
        FuUnicodeCodepointCaseConvert := 65320;
        RETURN;
    65353:
        FuUnicodeCodepointCaseConvert := 65321;
        RETURN;
    65354:
        FuUnicodeCodepointCaseConvert := 65322;
        RETURN;
    65355:
        FuUnicodeCodepointCaseConvert := 65323;
        RETURN;
    65356:
        FuUnicodeCodepointCaseConvert := 65324;
        RETURN;
    65357:
        FuUnicodeCodepointCaseConvert := 65325;
        RETURN;
    65358:
        FuUnicodeCodepointCaseConvert := 65326;
        RETURN;
    65359:
        FuUnicodeCodepointCaseConvert := 65327;
        RETURN;
    65360:
        FuUnicodeCodepointCaseConvert := 65328;
        RETURN;
    65361:
        FuUnicodeCodepointCaseConvert := 65329;
        RETURN;
    65362:
        FuUnicodeCodepointCaseConvert := 65330;
        RETURN;
    65363:
        FuUnicodeCodepointCaseConvert := 65331;
        RETURN;
    65364:
        FuUnicodeCodepointCaseConvert := 65332;
        RETURN;
    65365:
        FuUnicodeCodepointCaseConvert := 65333;
        RETURN;
    65366:
        FuUnicodeCodepointCaseConvert := 65334;
        RETURN;
    65367:
        FuUnicodeCodepointCaseConvert := 65335;
        RETURN;
    65368:
        FuUnicodeCodepointCaseConvert := 65336;
        RETURN;
    65369:
        FuUnicodeCodepointCaseConvert := 65337;
        RETURN;
    65370:
        FuUnicodeCodepointCaseConvert := 65338;
        RETURN;
    66560:
        FuUnicodeCodepointCaseConvert := 66600;
        RETURN;
    66561:
        FuUnicodeCodepointCaseConvert := 66601;
        RETURN;
    66562:
        FuUnicodeCodepointCaseConvert := 66602;
        RETURN;
    66563:
        FuUnicodeCodepointCaseConvert := 66603;
        RETURN;
    66564:
        FuUnicodeCodepointCaseConvert := 66604;
        RETURN;
    66565:
        FuUnicodeCodepointCaseConvert := 66605;
        RETURN;
    66566:
        FuUnicodeCodepointCaseConvert := 66606;
        RETURN;
    66567:
        FuUnicodeCodepointCaseConvert := 66607;
        RETURN;
    66568:
        FuUnicodeCodepointCaseConvert := 66608;
        RETURN;
    66569:
        FuUnicodeCodepointCaseConvert := 66609;
        RETURN;
    66570:
        FuUnicodeCodepointCaseConvert := 66610;
        RETURN;
    66571:
        FuUnicodeCodepointCaseConvert := 66611;
        RETURN;
    66572:
        FuUnicodeCodepointCaseConvert := 66612;
        RETURN;
    66573:
        FuUnicodeCodepointCaseConvert := 66613;
        RETURN;
    66574:
        FuUnicodeCodepointCaseConvert := 66614;
        RETURN;
    66575:
        FuUnicodeCodepointCaseConvert := 66615;
        RETURN;
    66576:
        FuUnicodeCodepointCaseConvert := 66616;
        RETURN;
    66577:
        FuUnicodeCodepointCaseConvert := 66617;
        RETURN;
    66578:
        FuUnicodeCodepointCaseConvert := 66618;
        RETURN;
    66579:
        FuUnicodeCodepointCaseConvert := 66619;
        RETURN;
    66580:
        FuUnicodeCodepointCaseConvert := 66620;
        RETURN;
    66581:
        FuUnicodeCodepointCaseConvert := 66621;
        RETURN;
    66582:
        FuUnicodeCodepointCaseConvert := 66622;
        RETURN;
    66583:
        FuUnicodeCodepointCaseConvert := 66623;
        RETURN;
    66584:
        FuUnicodeCodepointCaseConvert := 66624;
        RETURN;
    66585:
        FuUnicodeCodepointCaseConvert := 66625;
        RETURN;
    66586:
        FuUnicodeCodepointCaseConvert := 66626;
        RETURN;
    66587:
        FuUnicodeCodepointCaseConvert := 66627;
        RETURN;
    66588:
        FuUnicodeCodepointCaseConvert := 66628;
        RETURN;
    66589:
        FuUnicodeCodepointCaseConvert := 66629;
        RETURN;
    66590:
        FuUnicodeCodepointCaseConvert := 66630;
        RETURN;
    66591:
        FuUnicodeCodepointCaseConvert := 66631;
        RETURN;
    66592:
        FuUnicodeCodepointCaseConvert := 66632;
        RETURN;
    66593:
        FuUnicodeCodepointCaseConvert := 66633;
        RETURN;
    66594:
        FuUnicodeCodepointCaseConvert := 66634;
        RETURN;
    66595:
        FuUnicodeCodepointCaseConvert := 66635;
        RETURN;
    66596:
        FuUnicodeCodepointCaseConvert := 66636;
        RETURN;
    66597:
        FuUnicodeCodepointCaseConvert := 66637;
        RETURN;
    66598:
        FuUnicodeCodepointCaseConvert := 66638;
        RETURN;
    66599:
        FuUnicodeCodepointCaseConvert := 66639;
        RETURN;
    66600:
        FuUnicodeCodepointCaseConvert := 66560;
        RETURN;
    66601:
        FuUnicodeCodepointCaseConvert := 66561;
        RETURN;
    66602:
        FuUnicodeCodepointCaseConvert := 66562;
        RETURN;
    66603:
        FuUnicodeCodepointCaseConvert := 66563;
        RETURN;
    66604:
        FuUnicodeCodepointCaseConvert := 66564;
        RETURN;
    66605:
        FuUnicodeCodepointCaseConvert := 66565;
        RETURN;
    66606:
        FuUnicodeCodepointCaseConvert := 66566;
        RETURN;
    66607:
        FuUnicodeCodepointCaseConvert := 66567;
        RETURN;
    66608:
        FuUnicodeCodepointCaseConvert := 66568;
        RETURN;
    66609:
        FuUnicodeCodepointCaseConvert := 66569;
        RETURN;
    66610:
        FuUnicodeCodepointCaseConvert := 66570;
        RETURN;
    66611:
        FuUnicodeCodepointCaseConvert := 66571;
        RETURN;
    66612:
        FuUnicodeCodepointCaseConvert := 66572;
        RETURN;
    66613:
        FuUnicodeCodepointCaseConvert := 66573;
        RETURN;
    66614:
        FuUnicodeCodepointCaseConvert := 66574;
        RETURN;
    66615:
        FuUnicodeCodepointCaseConvert := 66575;
        RETURN;
    66616:
        FuUnicodeCodepointCaseConvert := 66576;
        RETURN;
    66617:
        FuUnicodeCodepointCaseConvert := 66577;
        RETURN;
    66618:
        FuUnicodeCodepointCaseConvert := 66578;
        RETURN;
    66619:
        FuUnicodeCodepointCaseConvert := 66579;
        RETURN;
    66620:
        FuUnicodeCodepointCaseConvert := 66580;
        RETURN;
    66621:
        FuUnicodeCodepointCaseConvert := 66581;
        RETURN;
    66622:
        FuUnicodeCodepointCaseConvert := 66582;
        RETURN;
    66623:
        FuUnicodeCodepointCaseConvert := 66583;
        RETURN;
    66624:
        FuUnicodeCodepointCaseConvert := 66584;
        RETURN;
    66625:
        FuUnicodeCodepointCaseConvert := 66585;
        RETURN;
    66626:
        FuUnicodeCodepointCaseConvert := 66586;
        RETURN;
    66627:
        FuUnicodeCodepointCaseConvert := 66587;
        RETURN;
    66628:
        FuUnicodeCodepointCaseConvert := 66588;
        RETURN;
    66629:
        FuUnicodeCodepointCaseConvert := 66589;
        RETURN;
    66630:
        FuUnicodeCodepointCaseConvert := 66590;
        RETURN;
    66631:
        FuUnicodeCodepointCaseConvert := 66591;
        RETURN;
    66632:
        FuUnicodeCodepointCaseConvert := 66592;
        RETURN;
    66633:
        FuUnicodeCodepointCaseConvert := 66593;
        RETURN;
    66634:
        FuUnicodeCodepointCaseConvert := 66594;
        RETURN;
    66635:
        FuUnicodeCodepointCaseConvert := 66595;
        RETURN;
    66636:
        FuUnicodeCodepointCaseConvert := 66596;
        RETURN;
    66637:
        FuUnicodeCodepointCaseConvert := 66597;
        RETURN;
    66638:
        FuUnicodeCodepointCaseConvert := 66598;
        RETURN;
    66639:
        FuUnicodeCodepointCaseConvert := 66599;
        RETURN;
    66736:
        FuUnicodeCodepointCaseConvert := 66776;
        RETURN;
    66737:
        FuUnicodeCodepointCaseConvert := 66777;
        RETURN;
    66738:
        FuUnicodeCodepointCaseConvert := 66778;
        RETURN;
    66739:
        FuUnicodeCodepointCaseConvert := 66779;
        RETURN;
    66740:
        FuUnicodeCodepointCaseConvert := 66780;
        RETURN;
    66741:
        FuUnicodeCodepointCaseConvert := 66781;
        RETURN;
    66742:
        FuUnicodeCodepointCaseConvert := 66782;
        RETURN;
    66743:
        FuUnicodeCodepointCaseConvert := 66783;
        RETURN;
    66744:
        FuUnicodeCodepointCaseConvert := 66784;
        RETURN;
    66745:
        FuUnicodeCodepointCaseConvert := 66785;
        RETURN;
    66746:
        FuUnicodeCodepointCaseConvert := 66786;
        RETURN;
    66747:
        FuUnicodeCodepointCaseConvert := 66787;
        RETURN;
    66748:
        FuUnicodeCodepointCaseConvert := 66788;
        RETURN;
    66749:
        FuUnicodeCodepointCaseConvert := 66789;
        RETURN;
    66750:
        FuUnicodeCodepointCaseConvert := 66790;
        RETURN;
    66751:
        FuUnicodeCodepointCaseConvert := 66791;
        RETURN;
    66752:
        FuUnicodeCodepointCaseConvert := 66792;
        RETURN;
    66753:
        FuUnicodeCodepointCaseConvert := 66793;
        RETURN;
    66754:
        FuUnicodeCodepointCaseConvert := 66794;
        RETURN;
    66755:
        FuUnicodeCodepointCaseConvert := 66795;
        RETURN;
    66756:
        FuUnicodeCodepointCaseConvert := 66796;
        RETURN;
    66757:
        FuUnicodeCodepointCaseConvert := 66797;
        RETURN;
    66758:
        FuUnicodeCodepointCaseConvert := 66798;
        RETURN;
    66759:
        FuUnicodeCodepointCaseConvert := 66799;
        RETURN;
    66760:
        FuUnicodeCodepointCaseConvert := 66800;
        RETURN;
    66761:
        FuUnicodeCodepointCaseConvert := 66801;
        RETURN;
    66762:
        FuUnicodeCodepointCaseConvert := 66802;
        RETURN;
    66763:
        FuUnicodeCodepointCaseConvert := 66803;
        RETURN;
    66764:
        FuUnicodeCodepointCaseConvert := 66804;
        RETURN;
    66765:
        FuUnicodeCodepointCaseConvert := 66805;
        RETURN;
    66766:
        FuUnicodeCodepointCaseConvert := 66806;
        RETURN;
    66767:
        FuUnicodeCodepointCaseConvert := 66807;
        RETURN;
    66768:
        FuUnicodeCodepointCaseConvert := 66808;
        RETURN;
    66769:
        FuUnicodeCodepointCaseConvert := 66809;
        RETURN;
    66770:
        FuUnicodeCodepointCaseConvert := 66810;
        RETURN;
    66771:
        FuUnicodeCodepointCaseConvert := 66811;
        RETURN;
    66776:
        FuUnicodeCodepointCaseConvert := 66736;
        RETURN;
    66777:
        FuUnicodeCodepointCaseConvert := 66737;
        RETURN;
    66778:
        FuUnicodeCodepointCaseConvert := 66738;
        RETURN;
    66779:
        FuUnicodeCodepointCaseConvert := 66739;
        RETURN;
    66780:
        FuUnicodeCodepointCaseConvert := 66740;
        RETURN;
    66781:
        FuUnicodeCodepointCaseConvert := 66741;
        RETURN;
    66782:
        FuUnicodeCodepointCaseConvert := 66742;
        RETURN;
    66783:
        FuUnicodeCodepointCaseConvert := 66743;
        RETURN;
    66784:
        FuUnicodeCodepointCaseConvert := 66744;
        RETURN;
    66785:
        FuUnicodeCodepointCaseConvert := 66745;
        RETURN;
    66786:
        FuUnicodeCodepointCaseConvert := 66746;
        RETURN;
    66787:
        FuUnicodeCodepointCaseConvert := 66747;
        RETURN;
    66788:
        FuUnicodeCodepointCaseConvert := 66748;
        RETURN;
    66789:
        FuUnicodeCodepointCaseConvert := 66749;
        RETURN;
    66790:
        FuUnicodeCodepointCaseConvert := 66750;
        RETURN;
    66791:
        FuUnicodeCodepointCaseConvert := 66751;
        RETURN;
    66792:
        FuUnicodeCodepointCaseConvert := 66752;
        RETURN;
    66793:
        FuUnicodeCodepointCaseConvert := 66753;
        RETURN;
    66794:
        FuUnicodeCodepointCaseConvert := 66754;
        RETURN;
    66795:
        FuUnicodeCodepointCaseConvert := 66755;
        RETURN;
    66796:
        FuUnicodeCodepointCaseConvert := 66756;
        RETURN;
    66797:
        FuUnicodeCodepointCaseConvert := 66757;
        RETURN;
    66798:
        FuUnicodeCodepointCaseConvert := 66758;
        RETURN;
    66799:
        FuUnicodeCodepointCaseConvert := 66759;
        RETURN;
    66800:
        FuUnicodeCodepointCaseConvert := 66760;
        RETURN;
    66801:
        FuUnicodeCodepointCaseConvert := 66761;
        RETURN;
    66802:
        FuUnicodeCodepointCaseConvert := 66762;
        RETURN;
    66803:
        FuUnicodeCodepointCaseConvert := 66763;
        RETURN;
    66804:
        FuUnicodeCodepointCaseConvert := 66764;
        RETURN;
    66805:
        FuUnicodeCodepointCaseConvert := 66765;
        RETURN;
    66806:
        FuUnicodeCodepointCaseConvert := 66766;
        RETURN;
    66807:
        FuUnicodeCodepointCaseConvert := 66767;
        RETURN;
    66808:
        FuUnicodeCodepointCaseConvert := 66768;
        RETURN;
    66809:
        FuUnicodeCodepointCaseConvert := 66769;
        RETURN;
    66810:
        FuUnicodeCodepointCaseConvert := 66770;
        RETURN;
    66811:
        FuUnicodeCodepointCaseConvert := 66771;
        RETURN;
    66928:
        FuUnicodeCodepointCaseConvert := 66967;
        RETURN;
    66929:
        FuUnicodeCodepointCaseConvert := 66968;
        RETURN;
    66930:
        FuUnicodeCodepointCaseConvert := 66969;
        RETURN;
    66931:
        FuUnicodeCodepointCaseConvert := 66970;
        RETURN;
    66932:
        FuUnicodeCodepointCaseConvert := 66971;
        RETURN;
    66933:
        FuUnicodeCodepointCaseConvert := 66972;
        RETURN;
    66934:
        FuUnicodeCodepointCaseConvert := 66973;
        RETURN;
    66935:
        FuUnicodeCodepointCaseConvert := 66974;
        RETURN;
    66936:
        FuUnicodeCodepointCaseConvert := 66975;
        RETURN;
    66937:
        FuUnicodeCodepointCaseConvert := 66976;
        RETURN;
    66938:
        FuUnicodeCodepointCaseConvert := 66977;
        RETURN;
    66940:
        FuUnicodeCodepointCaseConvert := 66979;
        RETURN;
    66941:
        FuUnicodeCodepointCaseConvert := 66980;
        RETURN;
    66942:
        FuUnicodeCodepointCaseConvert := 66981;
        RETURN;
    66943:
        FuUnicodeCodepointCaseConvert := 66982;
        RETURN;
    66944:
        FuUnicodeCodepointCaseConvert := 66983;
        RETURN;
    66945:
        FuUnicodeCodepointCaseConvert := 66984;
        RETURN;
    66946:
        FuUnicodeCodepointCaseConvert := 66985;
        RETURN;
    66947:
        FuUnicodeCodepointCaseConvert := 66986;
        RETURN;
    66948:
        FuUnicodeCodepointCaseConvert := 66987;
        RETURN;
    66949:
        FuUnicodeCodepointCaseConvert := 66988;
        RETURN;
    66950:
        FuUnicodeCodepointCaseConvert := 66989;
        RETURN;
    66951:
        FuUnicodeCodepointCaseConvert := 66990;
        RETURN;
    66952:
        FuUnicodeCodepointCaseConvert := 66991;
        RETURN;
    66953:
        FuUnicodeCodepointCaseConvert := 66992;
        RETURN;
    66954:
        FuUnicodeCodepointCaseConvert := 66993;
        RETURN;
    66956:
        FuUnicodeCodepointCaseConvert := 66995;
        RETURN;
    66957:
        FuUnicodeCodepointCaseConvert := 66996;
        RETURN;
    66958:
        FuUnicodeCodepointCaseConvert := 66997;
        RETURN;
    66959:
        FuUnicodeCodepointCaseConvert := 66998;
        RETURN;
    66960:
        FuUnicodeCodepointCaseConvert := 66999;
        RETURN;
    66961:
        FuUnicodeCodepointCaseConvert := 67000;
        RETURN;
    66962:
        FuUnicodeCodepointCaseConvert := 67001;
        RETURN;
    66964:
        FuUnicodeCodepointCaseConvert := 67003;
        RETURN;
    66965:
        FuUnicodeCodepointCaseConvert := 67004;
        RETURN;
    66967:
        FuUnicodeCodepointCaseConvert := 66928;
        RETURN;
    66968:
        FuUnicodeCodepointCaseConvert := 66929;
        RETURN;
    66969:
        FuUnicodeCodepointCaseConvert := 66930;
        RETURN;
    66970:
        FuUnicodeCodepointCaseConvert := 66931;
        RETURN;
    66971:
        FuUnicodeCodepointCaseConvert := 66932;
        RETURN;
    66972:
        FuUnicodeCodepointCaseConvert := 66933;
        RETURN;
    66973:
        FuUnicodeCodepointCaseConvert := 66934;
        RETURN;
    66974:
        FuUnicodeCodepointCaseConvert := 66935;
        RETURN;
    66975:
        FuUnicodeCodepointCaseConvert := 66936;
        RETURN;
    66976:
        FuUnicodeCodepointCaseConvert := 66937;
        RETURN;
    66977:
        FuUnicodeCodepointCaseConvert := 66938;
        RETURN;
    66979:
        FuUnicodeCodepointCaseConvert := 66940;
        RETURN;
    66980:
        FuUnicodeCodepointCaseConvert := 66941;
        RETURN;
    66981:
        FuUnicodeCodepointCaseConvert := 66942;
        RETURN;
    66982:
        FuUnicodeCodepointCaseConvert := 66943;
        RETURN;
    66983:
        FuUnicodeCodepointCaseConvert := 66944;
        RETURN;
    66984:
        FuUnicodeCodepointCaseConvert := 66945;
        RETURN;
    66985:
        FuUnicodeCodepointCaseConvert := 66946;
        RETURN;
    66986:
        FuUnicodeCodepointCaseConvert := 66947;
        RETURN;
    66987:
        FuUnicodeCodepointCaseConvert := 66948;
        RETURN;
    66988:
        FuUnicodeCodepointCaseConvert := 66949;
        RETURN;
    66989:
        FuUnicodeCodepointCaseConvert := 66950;
        RETURN;
    66990:
        FuUnicodeCodepointCaseConvert := 66951;
        RETURN;
    66991:
        FuUnicodeCodepointCaseConvert := 66952;
        RETURN;
    66992:
        FuUnicodeCodepointCaseConvert := 66953;
        RETURN;
    66993:
        FuUnicodeCodepointCaseConvert := 66954;
        RETURN;
    66995:
        FuUnicodeCodepointCaseConvert := 66956;
        RETURN;
    66996:
        FuUnicodeCodepointCaseConvert := 66957;
        RETURN;
    66997:
        FuUnicodeCodepointCaseConvert := 66958;
        RETURN;
    66998:
        FuUnicodeCodepointCaseConvert := 66959;
        RETURN;
    66999:
        FuUnicodeCodepointCaseConvert := 66960;
        RETURN;
    67000:
        FuUnicodeCodepointCaseConvert := 66961;
        RETURN;
    67001:
        FuUnicodeCodepointCaseConvert := 66962;
        RETURN;
    67003:
        FuUnicodeCodepointCaseConvert := 66964;
        RETURN;
    67004:
        FuUnicodeCodepointCaseConvert := 66965;
        RETURN;
    68736:
        FuUnicodeCodepointCaseConvert := 68800;
        RETURN;
    68737:
        FuUnicodeCodepointCaseConvert := 68801;
        RETURN;
    68738:
        FuUnicodeCodepointCaseConvert := 68802;
        RETURN;
    68739:
        FuUnicodeCodepointCaseConvert := 68803;
        RETURN;
    68740:
        FuUnicodeCodepointCaseConvert := 68804;
        RETURN;
    68741:
        FuUnicodeCodepointCaseConvert := 68805;
        RETURN;
    68742:
        FuUnicodeCodepointCaseConvert := 68806;
        RETURN;
    68743:
        FuUnicodeCodepointCaseConvert := 68807;
        RETURN;
    68744:
        FuUnicodeCodepointCaseConvert := 68808;
        RETURN;
    68745:
        FuUnicodeCodepointCaseConvert := 68809;
        RETURN;
    68746:
        FuUnicodeCodepointCaseConvert := 68810;
        RETURN;
    68747:
        FuUnicodeCodepointCaseConvert := 68811;
        RETURN;
    68748:
        FuUnicodeCodepointCaseConvert := 68812;
        RETURN;
    68749:
        FuUnicodeCodepointCaseConvert := 68813;
        RETURN;
    68750:
        FuUnicodeCodepointCaseConvert := 68814;
        RETURN;
    68751:
        FuUnicodeCodepointCaseConvert := 68815;
        RETURN;
    68752:
        FuUnicodeCodepointCaseConvert := 68816;
        RETURN;
    68753:
        FuUnicodeCodepointCaseConvert := 68817;
        RETURN;
    68754:
        FuUnicodeCodepointCaseConvert := 68818;
        RETURN;
    68755:
        FuUnicodeCodepointCaseConvert := 68819;
        RETURN;
    68756:
        FuUnicodeCodepointCaseConvert := 68820;
        RETURN;
    68757:
        FuUnicodeCodepointCaseConvert := 68821;
        RETURN;
    68758:
        FuUnicodeCodepointCaseConvert := 68822;
        RETURN;
    68759:
        FuUnicodeCodepointCaseConvert := 68823;
        RETURN;
    68760:
        FuUnicodeCodepointCaseConvert := 68824;
        RETURN;
    68761:
        FuUnicodeCodepointCaseConvert := 68825;
        RETURN;
    68762:
        FuUnicodeCodepointCaseConvert := 68826;
        RETURN;
    68763:
        FuUnicodeCodepointCaseConvert := 68827;
        RETURN;
    68764:
        FuUnicodeCodepointCaseConvert := 68828;
        RETURN;
    68765:
        FuUnicodeCodepointCaseConvert := 68829;
        RETURN;
    68766:
        FuUnicodeCodepointCaseConvert := 68830;
        RETURN;
    68767:
        FuUnicodeCodepointCaseConvert := 68831;
        RETURN;
    68768:
        FuUnicodeCodepointCaseConvert := 68832;
        RETURN;
    68769:
        FuUnicodeCodepointCaseConvert := 68833;
        RETURN;
    68770:
        FuUnicodeCodepointCaseConvert := 68834;
        RETURN;
    68771:
        FuUnicodeCodepointCaseConvert := 68835;
        RETURN;
    68772:
        FuUnicodeCodepointCaseConvert := 68836;
        RETURN;
    68773:
        FuUnicodeCodepointCaseConvert := 68837;
        RETURN;
    68774:
        FuUnicodeCodepointCaseConvert := 68838;
        RETURN;
    68775:
        FuUnicodeCodepointCaseConvert := 68839;
        RETURN;
    68776:
        FuUnicodeCodepointCaseConvert := 68840;
        RETURN;
    68777:
        FuUnicodeCodepointCaseConvert := 68841;
        RETURN;
    68778:
        FuUnicodeCodepointCaseConvert := 68842;
        RETURN;
    68779:
        FuUnicodeCodepointCaseConvert := 68843;
        RETURN;
    68780:
        FuUnicodeCodepointCaseConvert := 68844;
        RETURN;
    68781:
        FuUnicodeCodepointCaseConvert := 68845;
        RETURN;
    68782:
        FuUnicodeCodepointCaseConvert := 68846;
        RETURN;
    68783:
        FuUnicodeCodepointCaseConvert := 68847;
        RETURN;
    68784:
        FuUnicodeCodepointCaseConvert := 68848;
        RETURN;
    68785:
        FuUnicodeCodepointCaseConvert := 68849;
        RETURN;
    68786:
        FuUnicodeCodepointCaseConvert := 68850;
        RETURN;
    68800:
        FuUnicodeCodepointCaseConvert := 68736;
        RETURN;
    68801:
        FuUnicodeCodepointCaseConvert := 68737;
        RETURN;
    68802:
        FuUnicodeCodepointCaseConvert := 68738;
        RETURN;
    68803:
        FuUnicodeCodepointCaseConvert := 68739;
        RETURN;
    68804:
        FuUnicodeCodepointCaseConvert := 68740;
        RETURN;
    68805:
        FuUnicodeCodepointCaseConvert := 68741;
        RETURN;
    68806:
        FuUnicodeCodepointCaseConvert := 68742;
        RETURN;
    68807:
        FuUnicodeCodepointCaseConvert := 68743;
        RETURN;
    68808:
        FuUnicodeCodepointCaseConvert := 68744;
        RETURN;
    68809:
        FuUnicodeCodepointCaseConvert := 68745;
        RETURN;
    68810:
        FuUnicodeCodepointCaseConvert := 68746;
        RETURN;
    68811:
        FuUnicodeCodepointCaseConvert := 68747;
        RETURN;
    68812:
        FuUnicodeCodepointCaseConvert := 68748;
        RETURN;
    68813:
        FuUnicodeCodepointCaseConvert := 68749;
        RETURN;
    68814:
        FuUnicodeCodepointCaseConvert := 68750;
        RETURN;
    68815:
        FuUnicodeCodepointCaseConvert := 68751;
        RETURN;
    68816:
        FuUnicodeCodepointCaseConvert := 68752;
        RETURN;
    68817:
        FuUnicodeCodepointCaseConvert := 68753;
        RETURN;
    68818:
        FuUnicodeCodepointCaseConvert := 68754;
        RETURN;
    68819:
        FuUnicodeCodepointCaseConvert := 68755;
        RETURN;
    68820:
        FuUnicodeCodepointCaseConvert := 68756;
        RETURN;
    68821:
        FuUnicodeCodepointCaseConvert := 68757;
        RETURN;
    68822:
        FuUnicodeCodepointCaseConvert := 68758;
        RETURN;
    68823:
        FuUnicodeCodepointCaseConvert := 68759;
        RETURN;
    68824:
        FuUnicodeCodepointCaseConvert := 68760;
        RETURN;
    68825:
        FuUnicodeCodepointCaseConvert := 68761;
        RETURN;
    68826:
        FuUnicodeCodepointCaseConvert := 68762;
        RETURN;
    68827:
        FuUnicodeCodepointCaseConvert := 68763;
        RETURN;
    68828:
        FuUnicodeCodepointCaseConvert := 68764;
        RETURN;
    68829:
        FuUnicodeCodepointCaseConvert := 68765;
        RETURN;
    68830:
        FuUnicodeCodepointCaseConvert := 68766;
        RETURN;
    68831:
        FuUnicodeCodepointCaseConvert := 68767;
        RETURN;
    68832:
        FuUnicodeCodepointCaseConvert := 68768;
        RETURN;
    68833:
        FuUnicodeCodepointCaseConvert := 68769;
        RETURN;
    68834:
        FuUnicodeCodepointCaseConvert := 68770;
        RETURN;
    68835:
        FuUnicodeCodepointCaseConvert := 68771;
        RETURN;
    68836:
        FuUnicodeCodepointCaseConvert := 68772;
        RETURN;
    68837:
        FuUnicodeCodepointCaseConvert := 68773;
        RETURN;
    68838:
        FuUnicodeCodepointCaseConvert := 68774;
        RETURN;
    68839:
        FuUnicodeCodepointCaseConvert := 68775;
        RETURN;
    68840:
        FuUnicodeCodepointCaseConvert := 68776;
        RETURN;
    68841:
        FuUnicodeCodepointCaseConvert := 68777;
        RETURN;
    68842:
        FuUnicodeCodepointCaseConvert := 68778;
        RETURN;
    68843:
        FuUnicodeCodepointCaseConvert := 68779;
        RETURN;
    68844:
        FuUnicodeCodepointCaseConvert := 68780;
        RETURN;
    68845:
        FuUnicodeCodepointCaseConvert := 68781;
        RETURN;
    68846:
        FuUnicodeCodepointCaseConvert := 68782;
        RETURN;
    68847:
        FuUnicodeCodepointCaseConvert := 68783;
        RETURN;
    68848:
        FuUnicodeCodepointCaseConvert := 68784;
        RETURN;
    68849:
        FuUnicodeCodepointCaseConvert := 68785;
        RETURN;
    68850:
        FuUnicodeCodepointCaseConvert := 68786;
        RETURN;
    71840:
        FuUnicodeCodepointCaseConvert := 71872;
        RETURN;
    71841:
        FuUnicodeCodepointCaseConvert := 71873;
        RETURN;
    71842:
        FuUnicodeCodepointCaseConvert := 71874;
        RETURN;
    71843:
        FuUnicodeCodepointCaseConvert := 71875;
        RETURN;
    71844:
        FuUnicodeCodepointCaseConvert := 71876;
        RETURN;
    71845:
        FuUnicodeCodepointCaseConvert := 71877;
        RETURN;
    71846:
        FuUnicodeCodepointCaseConvert := 71878;
        RETURN;
    71847:
        FuUnicodeCodepointCaseConvert := 71879;
        RETURN;
    71848:
        FuUnicodeCodepointCaseConvert := 71880;
        RETURN;
    71849:
        FuUnicodeCodepointCaseConvert := 71881;
        RETURN;
    71850:
        FuUnicodeCodepointCaseConvert := 71882;
        RETURN;
    71851:
        FuUnicodeCodepointCaseConvert := 71883;
        RETURN;
    71852:
        FuUnicodeCodepointCaseConvert := 71884;
        RETURN;
    71853:
        FuUnicodeCodepointCaseConvert := 71885;
        RETURN;
    71854:
        FuUnicodeCodepointCaseConvert := 71886;
        RETURN;
    71855:
        FuUnicodeCodepointCaseConvert := 71887;
        RETURN;
    71856:
        FuUnicodeCodepointCaseConvert := 71888;
        RETURN;
    71857:
        FuUnicodeCodepointCaseConvert := 71889;
        RETURN;
    71858:
        FuUnicodeCodepointCaseConvert := 71890;
        RETURN;
    71859:
        FuUnicodeCodepointCaseConvert := 71891;
        RETURN;
    71860:
        FuUnicodeCodepointCaseConvert := 71892;
        RETURN;
    71861:
        FuUnicodeCodepointCaseConvert := 71893;
        RETURN;
    71862:
        FuUnicodeCodepointCaseConvert := 71894;
        RETURN;
    71863:
        FuUnicodeCodepointCaseConvert := 71895;
        RETURN;
    71864:
        FuUnicodeCodepointCaseConvert := 71896;
        RETURN;
    71865:
        FuUnicodeCodepointCaseConvert := 71897;
        RETURN;
    71866:
        FuUnicodeCodepointCaseConvert := 71898;
        RETURN;
    71867:
        FuUnicodeCodepointCaseConvert := 71899;
        RETURN;
    71868:
        FuUnicodeCodepointCaseConvert := 71900;
        RETURN;
    71869:
        FuUnicodeCodepointCaseConvert := 71901;
        RETURN;
    71870:
        FuUnicodeCodepointCaseConvert := 71902;
        RETURN;
    71871:
        FuUnicodeCodepointCaseConvert := 71903;
        RETURN;
    71872:
        FuUnicodeCodepointCaseConvert := 71840;
        RETURN;
    71873:
        FuUnicodeCodepointCaseConvert := 71841;
        RETURN;
    71874:
        FuUnicodeCodepointCaseConvert := 71842;
        RETURN;
    71875:
        FuUnicodeCodepointCaseConvert := 71843;
        RETURN;
    71876:
        FuUnicodeCodepointCaseConvert := 71844;
        RETURN;
    71877:
        FuUnicodeCodepointCaseConvert := 71845;
        RETURN;
    71878:
        FuUnicodeCodepointCaseConvert := 71846;
        RETURN;
    71879:
        FuUnicodeCodepointCaseConvert := 71847;
        RETURN;
    71880:
        FuUnicodeCodepointCaseConvert := 71848;
        RETURN;
    71881:
        FuUnicodeCodepointCaseConvert := 71849;
        RETURN;
    71882:
        FuUnicodeCodepointCaseConvert := 71850;
        RETURN;
    71883:
        FuUnicodeCodepointCaseConvert := 71851;
        RETURN;
    71884:
        FuUnicodeCodepointCaseConvert := 71852;
        RETURN;
    71885:
        FuUnicodeCodepointCaseConvert := 71853;
        RETURN;
    71886:
        FuUnicodeCodepointCaseConvert := 71854;
        RETURN;
    71887:
        FuUnicodeCodepointCaseConvert := 71855;
        RETURN;
    71888:
        FuUnicodeCodepointCaseConvert := 71856;
        RETURN;
    71889:
        FuUnicodeCodepointCaseConvert := 71857;
        RETURN;
    71890:
        FuUnicodeCodepointCaseConvert := 71858;
        RETURN;
    71891:
        FuUnicodeCodepointCaseConvert := 71859;
        RETURN;
    71892:
        FuUnicodeCodepointCaseConvert := 71860;
        RETURN;
    71893:
        FuUnicodeCodepointCaseConvert := 71861;
        RETURN;
    71894:
        FuUnicodeCodepointCaseConvert := 71862;
        RETURN;
    71895:
        FuUnicodeCodepointCaseConvert := 71863;
        RETURN;
    71896:
        FuUnicodeCodepointCaseConvert := 71864;
        RETURN;
    71897:
        FuUnicodeCodepointCaseConvert := 71865;
        RETURN;
    71898:
        FuUnicodeCodepointCaseConvert := 71866;
        RETURN;
    71899:
        FuUnicodeCodepointCaseConvert := 71867;
        RETURN;
    71900:
        FuUnicodeCodepointCaseConvert := 71868;
        RETURN;
    71901:
        FuUnicodeCodepointCaseConvert := 71869;
        RETURN;
    71902:
        FuUnicodeCodepointCaseConvert := 71870;
        RETURN;
    71903:
        FuUnicodeCodepointCaseConvert := 71871;
        RETURN;
    93760:
        FuUnicodeCodepointCaseConvert := 93792;
        RETURN;
    93761:
        FuUnicodeCodepointCaseConvert := 93793;
        RETURN;
    93762:
        FuUnicodeCodepointCaseConvert := 93794;
        RETURN;
    93763:
        FuUnicodeCodepointCaseConvert := 93795;
        RETURN;
    93764:
        FuUnicodeCodepointCaseConvert := 93796;
        RETURN;
    93765:
        FuUnicodeCodepointCaseConvert := 93797;
        RETURN;
    93766:
        FuUnicodeCodepointCaseConvert := 93798;
        RETURN;
    93767:
        FuUnicodeCodepointCaseConvert := 93799;
        RETURN;
    93768:
        FuUnicodeCodepointCaseConvert := 93800;
        RETURN;
    93769:
        FuUnicodeCodepointCaseConvert := 93801;
        RETURN;
    93770:
        FuUnicodeCodepointCaseConvert := 93802;
        RETURN;
    93771:
        FuUnicodeCodepointCaseConvert := 93803;
        RETURN;
    93772:
        FuUnicodeCodepointCaseConvert := 93804;
        RETURN;
    93773:
        FuUnicodeCodepointCaseConvert := 93805;
        RETURN;
    93774:
        FuUnicodeCodepointCaseConvert := 93806;
        RETURN;
    93775:
        FuUnicodeCodepointCaseConvert := 93807;
        RETURN;
    93776:
        FuUnicodeCodepointCaseConvert := 93808;
        RETURN;
    93777:
        FuUnicodeCodepointCaseConvert := 93809;
        RETURN;
    93778:
        FuUnicodeCodepointCaseConvert := 93810;
        RETURN;
    93779:
        FuUnicodeCodepointCaseConvert := 93811;
        RETURN;
    93780:
        FuUnicodeCodepointCaseConvert := 93812;
        RETURN;
    93781:
        FuUnicodeCodepointCaseConvert := 93813;
        RETURN;
    93782:
        FuUnicodeCodepointCaseConvert := 93814;
        RETURN;
    93783:
        FuUnicodeCodepointCaseConvert := 93815;
        RETURN;
    93784:
        FuUnicodeCodepointCaseConvert := 93816;
        RETURN;
    93785:
        FuUnicodeCodepointCaseConvert := 93817;
        RETURN;
    93786:
        FuUnicodeCodepointCaseConvert := 93818;
        RETURN;
    93787:
        FuUnicodeCodepointCaseConvert := 93819;
        RETURN;
    93788:
        FuUnicodeCodepointCaseConvert := 93820;
        RETURN;
    93789:
        FuUnicodeCodepointCaseConvert := 93821;
        RETURN;
    93790:
        FuUnicodeCodepointCaseConvert := 93822;
        RETURN;
    93791:
        FuUnicodeCodepointCaseConvert := 93823;
        RETURN;
    93792:
        FuUnicodeCodepointCaseConvert := 93760;
        RETURN;
    93793:
        FuUnicodeCodepointCaseConvert := 93761;
        RETURN;
    93794:
        FuUnicodeCodepointCaseConvert := 93762;
        RETURN;
    93795:
        FuUnicodeCodepointCaseConvert := 93763;
        RETURN;
    93796:
        FuUnicodeCodepointCaseConvert := 93764;
        RETURN;
    93797:
        FuUnicodeCodepointCaseConvert := 93765;
        RETURN;
    93798:
        FuUnicodeCodepointCaseConvert := 93766;
        RETURN;
    93799:
        FuUnicodeCodepointCaseConvert := 93767;
        RETURN;
    93800:
        FuUnicodeCodepointCaseConvert := 93768;
        RETURN;
    93801:
        FuUnicodeCodepointCaseConvert := 93769;
        RETURN;
    93802:
        FuUnicodeCodepointCaseConvert := 93770;
        RETURN;
    93803:
        FuUnicodeCodepointCaseConvert := 93771;
        RETURN;
    93804:
        FuUnicodeCodepointCaseConvert := 93772;
        RETURN;
    93805:
        FuUnicodeCodepointCaseConvert := 93773;
        RETURN;
    93806:
        FuUnicodeCodepointCaseConvert := 93774;
        RETURN;
    93807:
        FuUnicodeCodepointCaseConvert := 93775;
        RETURN;
    93808:
        FuUnicodeCodepointCaseConvert := 93776;
        RETURN;
    93809:
        FuUnicodeCodepointCaseConvert := 93777;
        RETURN;
    93810:
        FuUnicodeCodepointCaseConvert := 93778;
        RETURN;
    93811:
        FuUnicodeCodepointCaseConvert := 93779;
        RETURN;
    93812:
        FuUnicodeCodepointCaseConvert := 93780;
        RETURN;
    93813:
        FuUnicodeCodepointCaseConvert := 93781;
        RETURN;
    93814:
        FuUnicodeCodepointCaseConvert := 93782;
        RETURN;
    93815:
        FuUnicodeCodepointCaseConvert := 93783;
        RETURN;
    93816:
        FuUnicodeCodepointCaseConvert := 93784;
        RETURN;
    93817:
        FuUnicodeCodepointCaseConvert := 93785;
        RETURN;
    93818:
        FuUnicodeCodepointCaseConvert := 93786;
        RETURN;
    93819:
        FuUnicodeCodepointCaseConvert := 93787;
        RETURN;
    93820:
        FuUnicodeCodepointCaseConvert := 93788;
        RETURN;
    93821:
        FuUnicodeCodepointCaseConvert := 93789;
        RETURN;
    93822:
        FuUnicodeCodepointCaseConvert := 93790;
        RETURN;
    93823:
        FuUnicodeCodepointCaseConvert := 93791;
        RETURN;
    125184:
        FuUnicodeCodepointCaseConvert := 125218;
        RETURN;
    125185:
        FuUnicodeCodepointCaseConvert := 125219;
        RETURN;
    125186:
        FuUnicodeCodepointCaseConvert := 125220;
        RETURN;
    125187:
        FuUnicodeCodepointCaseConvert := 125221;
        RETURN;
    125188:
        FuUnicodeCodepointCaseConvert := 125222;
        RETURN;
    125189:
        FuUnicodeCodepointCaseConvert := 125223;
        RETURN;
    125190:
        FuUnicodeCodepointCaseConvert := 125224;
        RETURN;
    125191:
        FuUnicodeCodepointCaseConvert := 125225;
        RETURN;
    125192:
        FuUnicodeCodepointCaseConvert := 125226;
        RETURN;
    125193:
        FuUnicodeCodepointCaseConvert := 125227;
        RETURN;
    125194:
        FuUnicodeCodepointCaseConvert := 125228;
        RETURN;
    125195:
        FuUnicodeCodepointCaseConvert := 125229;
        RETURN;
    125196:
        FuUnicodeCodepointCaseConvert := 125230;
        RETURN;
    125197:
        FuUnicodeCodepointCaseConvert := 125231;
        RETURN;
    125198:
        FuUnicodeCodepointCaseConvert := 125232;
        RETURN;
    125199:
        FuUnicodeCodepointCaseConvert := 125233;
        RETURN;
    125200:
        FuUnicodeCodepointCaseConvert := 125234;
        RETURN;
    125201:
        FuUnicodeCodepointCaseConvert := 125235;
        RETURN;
    125202:
        FuUnicodeCodepointCaseConvert := 125236;
        RETURN;
    125203:
        FuUnicodeCodepointCaseConvert := 125237;
        RETURN;
    125204:
        FuUnicodeCodepointCaseConvert := 125238;
        RETURN;
    125205:
        FuUnicodeCodepointCaseConvert := 125239;
        RETURN;
    125206:
        FuUnicodeCodepointCaseConvert := 125240;
        RETURN;
    125207:
        FuUnicodeCodepointCaseConvert := 125241;
        RETURN;
    125208:
        FuUnicodeCodepointCaseConvert := 125242;
        RETURN;
    125209:
        FuUnicodeCodepointCaseConvert := 125243;
        RETURN;
    125210:
        FuUnicodeCodepointCaseConvert := 125244;
        RETURN;
    125211:
        FuUnicodeCodepointCaseConvert := 125245;
        RETURN;
    125212:
        FuUnicodeCodepointCaseConvert := 125246;
        RETURN;
    125213:
        FuUnicodeCodepointCaseConvert := 125247;
        RETURN;
    125214:
        FuUnicodeCodepointCaseConvert := 125248;
        RETURN;
    125215:
        FuUnicodeCodepointCaseConvert := 125249;
        RETURN;
    125216:
        FuUnicodeCodepointCaseConvert := 125250;
        RETURN;
    125217:
        FuUnicodeCodepointCaseConvert := 125251;
        RETURN;
    125218:
        FuUnicodeCodepointCaseConvert := 125184;
        RETURN;
    125219:
        FuUnicodeCodepointCaseConvert := 125185;
        RETURN;
    125220:
        FuUnicodeCodepointCaseConvert := 125186;
        RETURN;
    125221:
        FuUnicodeCodepointCaseConvert := 125187;
        RETURN;
    125222:
        FuUnicodeCodepointCaseConvert := 125188;
        RETURN;
    125223:
        FuUnicodeCodepointCaseConvert := 125189;
        RETURN;
    125224:
        FuUnicodeCodepointCaseConvert := 125190;
        RETURN;
    125225:
        FuUnicodeCodepointCaseConvert := 125191;
        RETURN;
    125226:
        FuUnicodeCodepointCaseConvert := 125192;
        RETURN;
    125227:
        FuUnicodeCodepointCaseConvert := 125193;
        RETURN;
    125228:
        FuUnicodeCodepointCaseConvert := 125194;
        RETURN;
    125229:
        FuUnicodeCodepointCaseConvert := 125195;
        RETURN;
    125230:
        FuUnicodeCodepointCaseConvert := 125196;
        RETURN;
    125231:
        FuUnicodeCodepointCaseConvert := 125197;
        RETURN;
    125232:
        FuUnicodeCodepointCaseConvert := 125198;
        RETURN;
    125233:
        FuUnicodeCodepointCaseConvert := 125199;
        RETURN;
    125234:
        FuUnicodeCodepointCaseConvert := 125200;
        RETURN;
    125235:
        FuUnicodeCodepointCaseConvert := 125201;
        RETURN;
    125236:
        FuUnicodeCodepointCaseConvert := 125202;
        RETURN;
    125237:
        FuUnicodeCodepointCaseConvert := 125203;
        RETURN;
    125238:
        FuUnicodeCodepointCaseConvert := 125204;
        RETURN;
    125239:
        FuUnicodeCodepointCaseConvert := 125205;
        RETURN;
    125240:
        FuUnicodeCodepointCaseConvert := 125206;
        RETURN;
    125241:
        FuUnicodeCodepointCaseConvert := 125207;
        RETURN;
    125242:
        FuUnicodeCodepointCaseConvert := 125208;
        RETURN;
    125243:
        FuUnicodeCodepointCaseConvert := 125209;
        RETURN;
    125244:
        FuUnicodeCodepointCaseConvert := 125210;
        RETURN;
    125245:
        FuUnicodeCodepointCaseConvert := 125211;
        RETURN;
    125246:
        FuUnicodeCodepointCaseConvert := 125212;
        RETURN;
    125247:
        FuUnicodeCodepointCaseConvert := 125213;
        RETURN;
    125248:
        FuUnicodeCodepointCaseConvert := 125214;
        RETURN;
    125249:
        FuUnicodeCodepointCaseConvert := 125215;
        RETURN;
    125250:
        FuUnicodeCodepointCaseConvert := 125216;
        RETURN;
    125251:
        FuUnicodeCodepointCaseConvert := 125217;
        RETURN;
END_CASE
